2126.13 BOOL  ; NC433_6_U 7ST接料伺服偏差计数器复位输出/ 原点调整命令输出
2126.14 BOOL  ; NC433_6_U 7ST接料伺服激活Override
2126.15 BOOL  ; NC433_6_U 7ST接料伺服停止
2127.00 BOOL  ; NC433_6_U 7ST接料伺服预留
2127.01 BOOL  ; NC433_6_U 7ST接料伺服预留
2127.02 BOOL  ; NC433_6_U 7ST接料伺服预留
2127.03 BOOL  ; NC433_6_U 7ST接料伺服预留
2127.04 BOOL  ; NC433_6_U 7ST接料伺服预留
2127.05 BOOL  ; NC433_6_U 7ST接料伺服预留
2127.06 BOOL  ; NC433_6_U 7ST接料伺服预留
2127.07 BOOL  ; NC433_6_U 7ST接料伺服预留
2127.08 BOOL  ; NC433_6_U 7ST接料伺服强制中断
2127.09 BOOL  ; NC433_6_U 7ST接料伺服预留
2127.10 BOOL  ; NC433_6_U 7ST接料伺服预留
2127.11 BOOL  ; NC433_6_U 7ST接料伺服预留
2127.12 BOOL  ; NC433_6_U 7ST接料伺服数据写入
2127.13 BOOL  ; NC433_6_U 7ST接料伺服数据读出
2127.14 BOOL  ; NC433_6_U 7ST接料伺服数据保存
2127.15 BOOL  ; NC433_6_U 7ST接料伺服预留
2128.00 BOOL  ; NC433_6_X1#预留
2128.01 BOOL  ; NC433_6_X1#预留
2128.02 BOOL  ; NC433_6_X1#预留
2128.03 BOOL  ; NC433_6_X1#预留
2128.04 BOOL  ; NC433_6_X1#等待存储器操作
2128.05 BOOL  ; NC433_6_X1#定位完成标志位
2128.06 BOOL  ; NC433_6_X1#无原点标志位
2128.07 BOOL  ; NC433_6_X1#原点停止标志位
2128.08 BOOL  ; NC433_6_X1#0 区监测标志位
2128.09 BOOL  ; NC433_6_X1#1 区监测标志位
2128.10 BOOL  ; NC433_6_X1#2 区监测标志位
2128.11 BOOL  ; NC433_6_X1#示教完成
2128.12 BOOL  ; NC433_6_X1#错误标志
2128.13 BOOL  ; NC433_6_X1#忙标志
2128.14 BOOL  ; NC433_6_X1#数据传送标志位
2128.15 BOOL  ; NC433_6_X1#减速停止执行标志位
2129.00 BOOL  ; NC433_6_X1#预留
2129.01 BOOL  ; NC433_6_X1#预留
2129.02 BOOL  ; NC433_6_X1#预留
2129.03 BOOL  ; NC433_6_X1#预留
2129.04 BOOL  ; NC433_6_X1#预留
2129.05 BOOL  ; NC433_6_X1#预留
2129.06 BOOL  ; NC433_6_X1#预留
2129.07 BOOL  ; NC433_6_X1#预留
2129.08 BOOL  ; NC433_6_X1#CW极限输入信号
2129.09 BOOL  ; NC433_6_X1#CCW极限输入信号
2129.10 BOOL  ; NC433_6_X1#原点接近输入信号
2129.11 BOOL  ; NC433_6_X1#原点输入信号
2129.12 BOOL  ; NC433_6_X1#中断输入信号
2129.13 BOOL  ; NC433_6_X1#紧急输入信号
2129.14 BOOL  ; NC433_6_X1#定位完成输入信号
2129.15 BOOL  ; NC433_6_X1#偏差计数器复位输出/ 原点调整命令输出
2130.00 BOOL  ; NC433_6_X1#错误代码
2130.01 BOOL  ; NC433_6_X1#错误代码
2130.02 BOOL  ; NC433_6_X1#错误代码
2130.03 BOOL  ; NC433_6_X1#错误代码
2130.04 BOOL  ; NC433_6_X1#错误代码
2130.05 BOOL  ; NC433_6_X1#错误代码
2130.06 BOOL  ; NC433_6_X1#错误代码
2130.07 BOOL  ; NC433_6_X1#错误代码
2130.08 BOOL  ; NC433_6_X1#错误代码
2130.09 BOOL  ; NC433_6_X1#错误代码
2130.10 BOOL  ; NC433_6_X1#错误代码
2130.11 BOOL  ; NC433_6_X1#错误代码
2130.12 BOOL  ; NC433_6_X1#错误代码
2130.13 BOOL  ; NC433_6_X1#错误代码
2130.14 BOOL  ; NC433_6_X1#错误代码
2130.15 BOOL  ; NC433_6_X1#错误代码
2131.00 BOOL  ; NC433_6_Y 2#预留
2131.01 BOOL  ; NC433_6_Y 2#预留
2131.02 BOOL  ; NC433_6_Y 2#预留
2131.03 BOOL  ; NC433_6_Y 2#预留
2131.04 BOOL  ; NC433_6_Y 2#等待存储器操作
2131.05 BOOL  ; NC433_6_Y 2#定位完成标志位
2131.06 BOOL  ; NC433_6_Y 2#无原点标志位
2131.07 BOOL  ; NC433_6_Y 2#原点停止标志位
2131.08 BOOL  ; NC433_6_Y 2#0 区监测标志位
2131.09 BOOL  ; NC433_6_Y 2#1 区监测标志位
2131.10 BOOL  ; NC433_6_Y 2#2 区监测标志位
2131.11 BOOL  ; NC433_6_Y 2#示教完成
2131.12 BOOL  ; NC433_6_Y 2#错误标志
2131.13 BOOL  ; NC433_6_Y 2#忙标志
2131.14 BOOL  ; NC433_6_Y 2#数据传送标志位
2131.15 BOOL  ; NC433_6_Y 2#减速停止执行标志位
2132.00 BOOL  ; NC433_6_Y 2#预留
2132.01 BOOL  ; NC433_6_Y 2#预留
2132.02 BOOL  ; NC433_6_Y 2#预留
2132.03 BOOL  ; NC433_6_Y 2#预留
2132.04 BOOL  ; NC433_6_Y 2#预留
2132.05 BOOL  ; NC433_6_Y 2#预留
2132.06 BOOL  ; NC433_6_Y 2#预留
2132.07 BOOL  ; NC433_6_Y 2#预留
2132.08 BOOL  ; NC433_6_Y 2#CW极限输入信号
2132.09 BOOL  ; NC433_6_Y 2#CCW极限输入信号
2132.10 BOOL  ; NC433_6_Y 2#原点接近输入信号
2132.11 BOOL  ; NC433_6_Y 2#原点输入信号
2132.12 BOOL  ; NC433_6_Y 2#中断输入信号
2132.13 BOOL  ; NC433_6_Y 2#紧急输入信号
2132.14 BOOL  ; NC433_6_Y 2#定位完成输入信号
2132.15 BOOL  ; NC433_6_Y 2#偏差计数器复位输出/ 原点调整命令输出
2133.00 BOOL  ; NC433_6_Y 2#错误代码
2133.01 BOOL  ; NC433_6_Y 2#错误代码
2133.02 BOOL  ; NC433_6_Y 2#错误代码
2133.03 BOOL  ; NC433_6_Y 2#错误代码
2133.04 BOOL  ; NC433_6_Y 2#错误代码
2133.05 BOOL  ; NC433_6_Y 2#错误代码
2133.06 BOOL  ; NC433_6_Y 2#错误代码
2133.07 BOOL  ; NC433_6_Y 2#错误代码
2133.08 BOOL  ; NC433_6_Y 2#错误代码
2133.09 BOOL  ; NC433_6_Y 2#错误代码
2133.10 BOOL  ; NC433_6_Y 2#错误代码
2133.11 BOOL  ; NC433_6_Y 2#错误代码
2133.12 BOOL  ; NC433_6_Y 2#错误代码
2133.13 BOOL  ; NC433_6_Y 2#错误代码
2133.14 BOOL  ; NC433_6_Y 2#错误代码
2133.15 BOOL  ; NC433_6_Y 2#错误代码
2134.00 BOOL  ; NC433_6_Z 3#预留
2134.01 BOOL  ; NC433_6_Z 3#预留
2134.02 BOOL  ; NC433_6_Z 3#预留
2134.03 BOOL  ; NC433_6_Z 3#预留
2134.04 BOOL  ; NC433_6_Z 3#等待存储器操作
2134.05 BOOL  ; NC433_6_Z 3#定位完成标志位
2134.06 BOOL  ; NC433_6_Z 3#无原点标志位
2134.07 BOOL  ; NC433_6_Z 3#原点停止标志位
2134.08 BOOL  ; NC433_6_Z 3#0 区监测标志位
2134.09 BOOL  ; NC433_6_Z 3#1 区监测标志位
2134.10 BOOL  ; NC433_6_Z 3#2 区监测标志位
2134.11 BOOL  ; NC433_6_Z 3#示教完成
2134.12 BOOL  ; NC433_6_Z 3#错误标志
2134.13 BOOL  ; NC433_6_Z 3#忙标志
2134.14 BOOL  ; NC433_6_Z 3#数据传送标志位
2134.15 BOOL  ; NC433_6_Z 3#减速停止执行标志位
2135.00 BOOL  ; NC433_6_Z 3#预留
2135.01 BOOL  ; NC433_6_Z 3#预留
2135.02 BOOL  ; NC433_6_Z 3#预留
2135.03 BOOL  ; NC433_6_Z 3#预留
2135.04 BOOL  ; NC433_6_Z 3#预留
2135.05 BOOL  ; NC433_6_Z 3#预留
2135.06 BOOL  ; NC433_6_Z 3#预留
2135.07 BOOL  ; NC433_6_Z 3#预留
2135.08 BOOL  ; NC433_6_Z 3#CW极限输入信号
2135.09 BOOL  ; NC433_6_Z 3#CCW极限输入信号
2135.10 BOOL  ; NC433_6_Z 3#原点接近输入信号
2135.11 BOOL  ; NC433_6_Z 3#原点输入信号
2135.12 BOOL  ; NC433_6_Z 3#中断输入信号
2135.13 BOOL  ; NC433_6_Z 3#紧急输入信号
2135.14 BOOL  ; NC433_6_Z 3#定位完成输入信号
2135.15 BOOL  ; NC433_6_Z 3#偏差计数器复位输出/ 原点调整命令输出
2136.00 BOOL  ; NC433_6_Z 3#错误代码
2136.01 BOOL  ; NC433_6_Z 3#错误代码
2136.02 BOOL  ; NC433_6_Z 3#错误代码
2136.03 BOOL  ; NC433_6_Z 3#错误代码
2136.04 BOOL  ; NC433_6_Z 3#错误代码
2136.05 BOOL  ; NC433_6_Z 3#错误代码
2136.06 BOOL  ; NC433_6_Z 3#错误代码
2136.07 BOOL  ; NC433_6_Z 3#错误代码
2136.08 BOOL  ; NC433_6_Z 3#错误代码
2136.09 BOOL  ; NC433_6_Z 3#错误代码
2136.10 BOOL  ; NC433_6_Z 3#错误代码
2136.11 BOOL  ; NC433_6_Z 3#错误代码
2136.12 BOOL  ; NC433_6_Z 3#错误代码
2136.13 BOOL  ; NC433_6_Z 3#错误代码
2136.14 BOOL  ; NC433_6_Z 3#错误代码
2136.15 BOOL  ; NC433_6_Z 3#错误代码
2137.00 BOOL  ; NC433_6_U 7ST接料伺服预留
2137.01 BOOL  ; NC433_6_U 7ST接料伺服预留
2137.02 BOOL  ; NC433_6_U 7ST接料伺服预留
2137.03 BOOL  ; NC433_6_U 7ST接料伺服预留
2137.04 BOOL  ; NC433_6_U 7ST接料伺服等待存储器操作
2137.05 BOOL  ; NC433_6_U 7ST接料伺服定位完成标志位
2137.06 BOOL  ; NC433_6_U 7ST接料伺服无原点标志位
2137.07 BOOL  ; NC433_6_U 7ST接料伺服原点停止标志位
2137.08 BOOL  ; NC433_6_U 7ST接料伺服0 区监测标志位
2137.09 BOOL  ; NC433_6_U 7ST接料伺服1 区监测标志位
2137.10 BOOL  ; NC433_6_U 7ST接料伺服2 区监测标志位
2137.11 BOOL  ; NC433_6_U 7ST接料伺服示教完成
2137.12 BOOL  ; NC433_6_U 7ST接料伺服错误标志
2137.13 BOOL  ; NC433_6_U 7ST接料伺服忙标志
2137.14 BOOL  ; NC433_6_U 7ST接料伺服数据传送标志位
2137.15 BOOL  ; NC433_6_U 7ST接料伺服减速停止执行标志位
2138.00 BOOL  ; NC433_6_U 7ST接料伺服预留
2138.01 BOOL  ; NC433_6_U 7ST接料伺服预留
2138.02 BOOL  ; NC433_6_U 7ST接料伺服预留
2138.03 BOOL  ; NC433_6_U 7ST接料伺服预留
2138.04 BOOL  ; NC433_6_U 7ST接料伺服预留
2138.05 BOOL  ; NC433_6_U 7ST接料伺服预留
2138.06 BOOL  ; NC433_6_U 7ST接料伺服预留
2138.07 BOOL  ; NC433_6_U 7ST接料伺服预留
2138.08 BOOL  ; NC433_6_U 7ST接料伺服CW极限输入信号
2138.09 BOOL  ; NC433_6_U 7ST接料伺服CCW极限输入信号
2138.10 BOOL  ; NC433_6_U 7ST接料伺服原点接近输入信号
2138.11 BOOL  ; NC433_6_U 7ST接料伺服原点输入信号
2138.12 BOOL  ; NC433_6_U 7ST接料伺服中断输入信号
2138.13 BOOL  ; NC433_6_U 7ST接料伺服紧急输入信号
2138.14 BOOL  ; NC433_6_U 7ST接料伺服定位完成输入信号
2138.15 BOOL  ; NC433_6_U 7ST接料伺服偏差计数器复位输出/ 原点调整命令输出
2139.00 BOOL  ; NC433_6_U 7ST接料伺服错误代码
2139.01 BOOL  ; NC433_6_U 7ST接料伺服错误代码
2139.02 BOOL  ; NC433_6_U 7ST接料伺服错误代码
2139.03 BOOL  ; NC433_6_U 7ST接料伺服错误代码
2139.04 BOOL  ; NC433_6_U 7ST接料伺服错误代码
2139.05 BOOL  ; NC433_6_U 7ST接料伺服错误代码
2139.06 BOOL  ; NC433_6_U 7ST接料伺服错误代码
2139.07 BOOL  ; NC433_6_U 7ST接料伺服错误代码
2139.08 BOOL  ; NC433_6_U 7ST接料伺服错误代码
2139.09 BOOL  ; NC433_6_U 7ST接料伺服错误代码
2139.10 BOOL  ; NC433_6_U 7ST接料伺服错误代码
2139.11 BOOL  ; NC433_6_U 7ST接料伺服错误代码
2139.12 BOOL  ; NC433_6_U 7ST接料伺服错误代码
2139.13 BOOL  ; NC433_6_U 7ST接料伺服错误代码
2139.14 BOOL  ; NC433_6_U 7ST接料伺服错误代码
2139.15 BOOL  ; NC433_6_U 7ST接料伺服错误代码
2170 CHANNEL  ; DA08V_1 通道使能
2171 CHANNEL  ; DA08V_1 通道1 A1比例阀 转换值
2172 CHANNEL  ; DA08V_1 通道2 A2比例阀 转换值
2173 CHANNEL  ; DA08V_1 通道3 A3比例阀 转换值
2174 CHANNEL  ; DA08V_1 通道4 A4比例阀 转换值
2175 CHANNEL  ; DA08V_1 通道5 B1比例阀 转换值
2176 CHANNEL  ; DA08V_1 通道6 B2比例阀 转换值
2177 CHANNEL  ; DA08V_1 通道7 B3比例阀 转换值
2178 CHANNEL  ; DA08V_1 通道8 B4比例阀 转换值
2180 CHANNEL  ; DA08V_2 通道使能
2181 CHANNEL  ; DA08V_2 通道1DA 转换值
2182 CHANNEL  ; DA08V_2 通道2DA 转换值
2183 CHANNEL  ; DA08V_2 通道3DA 转换值
2184 CHANNEL  ; DA08V_2 通道4DA 转换值
2185 CHANNEL  ; DA08V_2 通道5DA 转换值
2186 CHANNEL  ; DA08V_2 通道6DA 转换值
2187 CHANNEL  ; DA08V_2 通道7DA 转换值
2188 CHANNEL  ; DA08V_2 通道8DA 转换值
2190 CHANNEL  ; DA08V_3 通道使能
2191 CHANNEL  ; DA08V_3 通道1DA 转换值
2192 CHANNEL  ; DA08V_3 通道2DA 转换值
2193 CHANNEL  ; DA08V_3 通道3DA 转换值
2194 CHANNEL  ; DA08V_3 通道4DA 转换值
2195 CHANNEL  ; DA08V_3 通道5DA 转换值
2196 CHANNEL  ; DA08V_3 通道6DA 转换值
2197 CHANNEL  ; DA08V_3 通道7DA 转换值
2198 CHANNEL  ; DA08V_3 通道8DA 转换值
21.00 BOOL  ; 热压C下层上板左加热启动
21.01 BOOL  ; 热压C下层上板中加热启动
21.02 BOOL  ; 热压C下层上板右加热启动
21.03 BOOL  ; 热压C下层下板左加热启动
21.04 BOOL  ; 热压C下层下板中加热启动
21.05 BOOL  ; 热压C下层下板右加热启动
2200 CHANNEL  ; DA08V_4 通道使能
2201 CHANNEL  ; DA08V_4 通道1DA 转换值
2202 CHANNEL  ; DA08V_4 通道2DA 转换值
2203 CHANNEL  ; DA08V_4 通道3DA 转换值
2204 CHANNEL  ; DA08V_4 通道4DA 转换值
2205 CHANNEL  ; DA08V_4 通道5DA 转换值
2206 CHANNEL  ; DA08V_4 通道6DA 转换值
2207 CHANNEL  ; DA08V_4 通道7DA 转换值
2208 CHANNEL  ; DA08V_4 通道8DA 转换值
221.00 BOOL  ; 进出料横移伺服A进料位手动(M)
221.01 BOOL  ; 进出料横移伺服热压A放料位手动(M)
221.02 BOOL  ; 进出料横移伺服热压A取料位手动(M)
221.03 BOOL  ; 进出料横移伺服热压B放料位手动(M)
221.04 BOOL  ; 横移伺服热压B取料位手动(M)
221.05 BOOL  ; 横移伺服热压C放料位手动(M)
221.06 BOOL  ; 横移伺服热压C取料位手动(M)
221.07 BOOL  ; 进出料横移伺服出料位手动(M)
222.00 BOOL  ; 进出料横移伺服A进料位(A)
222.01 BOOL  ; 进出料横移伺服热压A放料位(A)
222.02 BOOL  ; 进出料横移伺服热压A取料位(A)
222.03 BOOL  ; 进出料横移伺服热压B放料位(A)
222.04 BOOL  ; 横移伺服热压B取料位(A)
222.05 BOOL  ; 横移伺服热压C放料位(A)
222.06 BOOL  ; 横移伺服热压C取料位(A)
222.07 BOOL  ; 进出料横移伺服出料位(A)
223.00 BOOL  ; 进出料伸缩伺服等待位手动(M)
223.01 BOOL  ; 进出料伸缩伺服平台取料位手动(M)
223.02 BOOL  ; 进出料伸缩伺服A热压取放位手动(M)
224.00 BOOL  ; 进出料伸缩伺服等待位(A)
224.01 BOOL  ; 进出料伸缩伺服平台取料位(A)
224.02 BOOL  ; 进出料伸缩伺服A热压取放位(A)
2.00 BOOL  ; 进料定位下层有料感应
2.01 BOOL  ; 出料定位上层前后松开位
2.02 BOOL  ; 出料定位上层前后夹紧位
2.03 BOOL  ; 出料定位下层前后松开位
2.04 BOOL  ; 出料定位下层前后夹紧位
2.05 BOOL  ; 出料定位上层左右松开位
2.06 BOOL  ; 出料定位上层左右夹紧位
2.07 BOOL  ; 出料定位下层左右松开位
2.08 BOOL  ; 出料定位下层左右夹紧位
2.09 BOOL  ; 出料定位平台上层接料位
2.10 BOOL  ; 出料定位平台上层出料位
2.11 BOOL  ; 出料定位平台下层接料位
2.12 BOOL  ; 出料定位平台下层出料位
2.13 BOOL  ; 出料定位上层有料感应
2.14 BOOL  ; 出料定位下层有料感应
2.15 BOOL  ; 备用5
321.00 BOOL  ; 进出料横移伺服A进料位
321.01 BOOL  ; 进出料横移伺服热压A放料位
321.02 BOOL  ; 进出料横移伺服热压A取料位
321.03 BOOL  ; 进出料横移伺服热压B放料位
321.04 BOOL  ; 横移伺服热压B取料位
321.05 BOOL  ; 横移伺服热压C放料位
321.06 BOOL  ; 横移伺服热压C取料位
321.07 BOOL  ; 进出料横移伺服出料位
323.00 BOOL  ; 进出料伸缩伺服等待位
323.01 BOOL  ; 进出料伸缩伺服平台取料位
323.02 BOOL  ; 进出料伸缩伺服A热压取放位
3.00 BOOL  ; 进料夹爪张开位
3.01 BOOL  ; 进料夹爪夹紧位
3.02 BOOL  ; 进料爪上层左压紧上升位
3.03 BOOL  ; 进料爪上层右压紧上升位
3.04 BOOL  ; 进料爪下层左压紧上升位
3.05 BOOL  ; 进料爪下层右压紧上升位
3.06 BOOL  ; 进料爪上层中间压紧上升位
3.07 BOOL  ; 进料爪下层中间压紧上升位
3.08 BOOL  ; 进料夹爪上升位
3.09 BOOL  ; 进料夹爪下降位
3.10 BOOL  ; 进料爪上层有料感应
3.11 BOOL  ; 进料爪下层有料感应
3.12 BOOL  ; 出料夹爪张开位
3.13 BOOL  ; 出料夹爪夹紧位
3.14 BOOL  ; 出料爪上层左压紧上升位
3.15 BOOL  ; 出料爪上层右压紧上升位
42.04 BOOL  ; $?St$Bk?_#[5] / 上料定位A0度翻转 / $?St$Bk?_#[5]
42.05 BOOL  ; 上料定位A90度翻转
42.06 BOOL  ; 上料定位A1前后左右松开
42.07 BOOL  ; 上料定位A1前后左右夹紧
42.08 BOOL  ; 上料定位A2前后左右松开
42.09 BOOL  ; 上料定位A2前后左右夹紧
42.10 BOOL  ; 上料定位A3前后左右松开
42.11 BOOL  ; 上料定位A3前后左右夹紧
42.12 BOOL  ; 上料定位A4前后左右松开
42.13 BOOL  ; 上料定位A4前后左右夹紧
47.02 BOOL  ; 热压A上预压平移气缸缩回
47.03 BOOL  ; 热压A上预压平移气缸预压
47.06 BOOL  ; 热压A垫高气缸移出
47.07 BOOL  ; 热压A垫高气缸热压
47.08 BOOL  ; 热压A1HIP测试上升
47.09 BOOL  ; 热压A1HIP测试下降
48.00 BOOL  ; 热压A1顶升气缸缩回
48.01 BOOL  ; 热压A1顶升气缸伸出
48.02 BOOL  ; 热压A2顶升气缸左右缩回
48.03 BOOL  ; 热压A2顶升气缸左右伸出
48.04 BOOL  ; 热压A3顶升气缸左右缩回
48.05 BOOL  ; 热压A3顶升气缸左右伸出
48.06 BOOL  ; 热压A4顶升气缸左右缩回
48.07 BOOL  ; 热压A4顶升气缸左右伸出
48.14 BOOL  ; 热压A上吹气
48.15 BOOL  ; 热压A下板A吹气
49.00 BOOL  ; 热压A下板B吹气
49.01 BOOL  ; 热压B上预压平移气缸缩回
49.02 BOOL  ; 热压B上预压平移气缸预压
49.03 BOOL  ; 热压B下预压平移气缸缩回
49.04 BOOL  ; 热压B下预压平移气缸预压
49.05 BOOL  ; 热压B垫高气缸移出
49.06 BOOL  ; 热压B垫高气缸热压
49.07 BOOL  ; 热压B1HIP测试上升
49.08 BOOL  ; 热压B1HIP测试下降
49.15 BOOL  ; 热压B1顶升气缸缩回
4.00 BOOL  ; 出料爪下层左压紧上升位
4.01 BOOL  ; 出料爪下层右压紧上升位
4.02 BOOL  ; 出料夹爪上升位
4.03 BOOL  ; 出料夹爪下降位
4.04 BOOL  ; 出料爪上层有料感应
4.05 BOOL  ; 出料爪下层有料感应
4.06 BOOL  ; 备用6
4.07 BOOL  ; 备用7
4.08 BOOL  ; 热压A增压缸上升位
4.09 BOOL  ; 热压A增压缸下降位
4.10 BOOL  ; 热压A上层顶升气缸上升位
4.11 BOOL  ; 热压A上层顶升气缸下降位
4.12 BOOL  ; 热压A下层顶升气缸上升位
4.13 BOOL  ; 热压A下层顶升气缸下降位
4.14 BOOL  ; 热压A垫高气缸移出位
4.15 BOOL  ; 热压A垫高气缸热压位
50.00 BOOL  ; 热压B1顶升气缸伸出
50.01 BOOL  ; 热压B2顶升气缸左缩回
50.02 BOOL  ; 热压B2顶升气缸左伸出
50.03 BOOL  ; 热压B3顶升气缸左缩回
50.04 BOOL  ; 热压B3顶升气缸左伸出
50.05 BOOL  ; 热压B4顶升气缸左缩回
50.06 BOOL  ; 热压B4顶升气缸左伸出
50.13 BOOL  ; 热压B上吹气
50.14 BOOL  ; 热压B下板A吹气
50.15 BOOL  ; 热压B下板B吹气
5.00 BOOL  ; 热压A上层Hip测试气缸上升位
5.01 BOOL  ; 热压A上层Hip测试气缸下降位
5.02 BOOL  ; 热压A下层Hip测试气缸上升位
5.03 BOOL  ; 热压A下层Hip测试气缸下降位
5.04 BOOL  ; 热压A上层有料感应
5.05 BOOL  ; 热压A下层有料感应
5.06 BOOL  ; 热压A上层极耳检查输入
5.07 BOOL  ; 热压A下层极耳检查输入
5.08 BOOL  ; 备用8
5.09 BOOL  ; 热压B增压缸上升位
5.10 BOOL  ; 热压B增压缸下降位
5.11 BOOL  ; 热压B上层顶升气缸上升位
5.12 BOOL  ; 热压B上层顶升气缸下降位
5.13 BOOL  ; 热压B下层顶升气缸上升位
5.14 BOOL  ; 热压B下层顶升气缸下降位
5.15 BOOL  ; 热压B垫高气缸移出位
6.00 BOOL  ; 热压B垫高气缸热压位
6.01 BOOL  ; 热压B上层Hip测试气缸上升位
6.02 BOOL  ; 热压B上层Hip测试气缸下降位
6.03 BOOL  ; 热压B下层Hip测试气缸上升位
6.04 BOOL  ; 热压B下层Hip测试气缸下降位
6.05 BOOL  ; 热压B上层有料感应
6.06 BOOL  ; 热压B下层有料感应
6.07 BOOL  ; 热压B上层极耳检查输入
6.08 BOOL  ; 热压B下层极耳检查输入
6.09 BOOL  ; 备用9
6.10 BOOL  ; 热压C增压缸上升位
6.11 BOOL  ; 热压C增压缸下降位
6.12 BOOL  ; 热压C上层顶升气缸上升位
6.13 BOOL  ; 热压C上层顶升气缸下降位
6.14 BOOL  ; 热压C下层顶升气缸上升位
6.15 BOOL  ; 热压C下层顶升气缸下降位
711 CHANNEL  ; 机器人不在取料区域延时
713 CHANNEL  ; $?St$Bk?_#[6] / 机器人不在放料A区域 / $?St$Bk?_#[6]
7.00 BOOL  ; 热压C垫高气缸移出位
7.01 BOOL  ; 热压C垫高气缸热压位
7.02 BOOL  ; 热压C上层Hip测试气缸上升位
7.03 BOOL  ; 热压C上层Hip测试气缸下降位
7.04 BOOL  ; 热压C下层Hip测试气缸上升位
7.05 BOOL  ; 热压C下层Hip测试气缸下降位
7.06 BOOL  ; 热压C上层有料感应
7.07 BOOL  ; 热压C下层有料感应
7.08 BOOL  ; 热压C上层极耳检查输入
7.09 BOOL  ; 热压C下层极耳检查输入
7.10 BOOL  ; 备用10
7.11 BOOL  ; 进出料转移伺服准备好
7.12 BOOL  ; 进出料转移伺服报警
7.13 BOOL  ; 伸缩伺服准备好
7.14 BOOL  ; 伸缩伺服报警
7.15 BOOL  ; 备用11
8 CHANNEL  ; 副PLC 0CH输入映射
8.00 BOOL  ; 加热A跳闸
8.01 BOOL  ; 加热B跳闸
8.02 BOOL  ; 加热C跳闸
8.03 BOOL  ; 副PLC 0.03
8.04 BOOL  ; 副PLC 0.04
8.05 BOOL  ; 副PLC 0.05
8.06 BOOL  ; 副PLC 0.06
8.07 BOOL  ; 副PLC 0.07
8.08 BOOL  ; 副PLC 0.08
8.09 BOOL  ; 副PLC 0.09
8.10 BOOL  ; 副PLC 0.10
8.11 BOOL  ; 副PLC 0.11
9 CHANNEL  ; 副PLC输入点1CH 映射地址
9.00 BOOL  ; 副PLC 1.00
9.01 BOOL  ; 副PLC 1.01
9.02 BOOL  ; 副PLC 1.02
9.03 BOOL  ; 副PLC 1.03
9.04 BOOL  ; 副PLC 1.04
9.05 BOOL  ; 副PLC 1.05
9.06 BOOL  ; 副PLC 1.06
9.07 BOOL  ; 副PLC 1.07
9.08 BOOL  ; 副PLC 1.08
9.09 BOOL  ; 副PLC 1.09
9.10 BOOL  ; 副PLC 1.10
9.11 BOOL  ; 副PLC 1.11
A202.00 BOOL  ; 内部逻辑端口1网络通信可执行标志
A202.01 BOOL  ; 内部逻辑端口2网络通信可执行标志
A202.02 BOOL  ; 内部逻辑端口3网络通信可执行标志
A202.03 BOOL  ; 内部逻辑端口4网络通信可执行标志
A202.04 BOOL  ; 内部逻辑端口5网络通信可执行标志
A202.05 BOOL  ; 内部逻辑端口6网络通信可执行标志
A202.06 BOOL  ; 内部逻辑端口7网络通信可执行标志
A202.07 BOOL  ; 内部逻辑端口7网络通信可执行标志
D0.00 BOOL  ; 机器人安全位置
D0.01 BOOL  ; 移载安全位置
D1000.00 BOOL  ; 自动模式
D1000.01 BOOL  ; 手动模式
D1000.02 BOOL  ; 自动运行中
D1000.04 BOOL  ; 初始化中
D1000.05 BOOL  ; 清料停止中
D1000.06 BOOL  ; 自动停止中
D1000.07 BOOL  ; 蜂鸣器停止
D1001.00 BOOL  ; 自动停止完成
D1001.02 BOOL  ; 整机初始化完成
D1001.03 BOOL  ; 整机清料完成
D1001.04 BOOL  ; 整机物料感应为空
D1001.05 BOOL  ; 外部（工厂报警系统）→允许运行
D1001.09 BOOL  ; 气压异常（正常=1）
D1001.10 BOOL  ; 急停（正常=1）
D1001.11 BOOL  ; 安全装置（正常=1）
D1001.12 BOOL  ; 跳闸（正常=1）
D1001.13 BOOL  ; 整机错误（气压+急停+门+跳闸）
D1001.14 BOOL  ; 整机警报
D1001.15 BOOL  ; 整机+工站错误
D1002.00 BOOL  ; 清料停止[T]
D1002.09 BOOL  ; 复位（T）
D1002.10 BOOL  ; 整机启动[T]
D1002.11 BOOL  ; 整机自动停止[T]
D1002.12 BOOL  ; 整机初始化[T]
D1002.14 BOOL  ; 蜂鸣器消音（T）
D1002.15 BOOL  ; 任务停止
D1003.02 BOOL  ; 整机记忆清除（T）
D1003.15 BOOL  ; 模组B加热正常
D1005 CHANNEL  ; 屏幕状态
D10050 CHANNEL  ; ST5520_A 测试电压输入设定值(F)
D10060 CHANNEL  ; 字符串表现形式(0-小数点形式,1-指数形式)
D10061 CHANNEL  ; 全位数
D10062 CHANNEL  ; 小数位数
D1006.00 BOOL  ; 主屏使用
D1006.01 BOOL  ; 副屏使用
D1006.02 BOOL  ; 小屏使用
D1006.03 BOOL  ; 没有移动屏使用信号，小屏不能使用
D10070 CHANNEL  ; ST5520_A 测试电压输入设定值(ASCII)
D10080 CHANNEL  ; ST5520_A 测试时间输入设定值(F)
D10091 CHANNEL  ; 全位数
D10092 CHANNEL  ; 小数位数
D10100 CHANNEL  ; ST5520_A 测试时间输入设定值(ASC)
D1010.00 BOOL  ; 1St上料机器人工站错误
D1010.01 BOOL  ; 1St上料机器人工站警告
D1010.02 BOOL  ; 1St上料机器人工站运行
D1010.03 BOOL  ; $?St$Bk?_#[8] / 1St上料机器人"$?St$Bk?_#[8]
D1010.05 BOOL  ; $?St$Bk?_#[10] / 1St上料机器人"$?St$Bk?_#[10]
D1010.07 BOOL  ; $?St$Bk?_#[12] / 1St上料机器人"$?St$Bk?_#[12]
D1010.09 BOOL  ; $?St$Bk?_#[14] / 1St上料机器人"$?St$Bk?_#[14]
D1010.11 BOOL  ; $?St$Bk?_#[16] / 1St上料机器人"$?St$Bk?_#[16]
D1010.13 BOOL  ; $?St$Bk?_#[18] / 1St上料机器人"$?St$Bk?_#[18]
D1010.15 BOOL  ; $?St$Bk?_#[20] / 1St上料机器人"$?St$Bk?_#[20]
D1011.04 BOOL  ; $?St$Bk?_#[22] / 1St上料机器人"$?St$Bk?_#[22]
D1011.06 BOOL  ; $?St$Bk?_#[24] / 1St上料机器人"$?St$Bk?_#[24]
D1011.08 BOOL  ; $?St$Bk?_#[26] / 1St上料机器人"$?St$Bk?_#[26]
D1011.10 BOOL  ; $?St$Bk?_#[28] / 1St上料机器人"$?St$Bk?_#[28]
D1011.12 BOOL  ; $?St$Bk?_#[30] / 1St上料机器人"$?St$Bk?_#[30]
D1011.14 BOOL  ; $?St$Bk?_#[32] / 1St上料机器人"$?St$Bk?_#[32]
D10120 CHANNEL  ; 字符串表现形式(0-小数点形式,1-指数形式)
D10121 CHANNEL  ; 全位数
D10122 CHANNEL  ; 小数位数
D1012.00 BOOL  ; 1St上料机器人工站就绪
D1012.01 BOOL  ; 1St上料机器人 初始化中
D1012.02 BOOL  ; 1St上料机器人 自动停止中
D1012.03 BOOL  ; 1St上料机器人 自动停止完成
D1012.04 BOOL  ; 1St上料机器人 联锁
D1012.05 BOOL  ; 1St上料机器人 单步中
D1012.06 BOOL  ; 1St上料机器人 单周期中
D1012.07 BOOL  ; 1St上料机器人 周期完成
D1012.08 BOOL  ; 1St上料机器人 任务开始
D1012.09 BOOL  ; 1St上料机器人 任务递进条件
D1012.10 BOOL  ; 1St上料机器人 任务递进
D1012.11 BOOL  ; 1St上料机器人 工作完成
D1012.12 BOOL  ; 1St上料机器人 初始化[T]
D1012.13 BOOL  ; 1St上料机器人 单步[T]
D1012.14 BOOL  ; 1St上料机器人 单周期[T]
D1012.15 BOOL  ; 1St上料机器人 任务停止[T]
D10130 CHANNEL  ; ST5520_A 响应延时时间输入设定值(ASC)
D1013.00 BOOL  ; 1St上料机器人 工站完成置位[T]
D1013.01 BOOL  ; 1St上料机器人 工站完成复位[T]
D1013.02 BOOL  ; 1St上料机器人 数据清除[T]
D1013.03 BOOL  ; 1St上料机器人 工站屏蔽[T]
D1013.04 BOOL  ; $?St$Bk?_#[34] / 1St上料机器人"$?St$Bk?_#[34]
D1013.06 BOOL  ; $?St$Bk?_#[36] / 1St上料机器人"$?St$Bk?_#[36]
D1013.08 BOOL  ; $?St$Bk?_#[38] / 1St上料机器人"$?St$Bk?_#[38]
D1013.10 BOOL  ; $?St$Bk?_#[40] / 1St上料机器人"$?St$Bk?_#[40]
D1013.12 BOOL  ; $?St$Bk?_#[42] / 1St上料机器人"$?St$Bk?_#[42]
D1013.14 BOOL  ; $?St$Bk?_#[44] / 1St上料机器人"$?St$Bk?_#[44]
D10140 CHANNEL  ; ST5520_A 绝缘电阻上限输入设定值(Float)
D1014.00 BOOL  ; 1St上料机器人上游就绪-0
D1014.01 BOOL  ; 1St上料机器人使能上游-0
D1014.02 BOOL  ; 1St上料机器人上游就绪-1
D1014.03 BOOL  ; 1St上料机器人使能上游-1
D1014.04 BOOL  ; 1St上料机器人上游就绪-2
D1014.05 BOOL  ; 1St上料机器人使能上游-2
D1014.06 BOOL  ; 1St上料机器人上游就绪-3
D1014.07 BOOL  ; 1St上料机器人使能上游-3
D1014.08 BOOL  ; 1St上料机器人下游就绪-0
D1014.09 BOOL  ; 1St上料机器人使能下游-0
D1014.10 BOOL  ; 1St上料机器人下游就绪-1
D1014.11 BOOL  ; 1St上料机器人使能下游-1
D1014.12 BOOL  ; 1St上料机器人下游就绪-2
D1014.13 BOOL  ; 1St上料机器人使能下游-2
D1014.14 BOOL  ; 1St上料机器人下游就绪-3
D1014.15 BOOL  ; 1St上料机器人使能下游-3
D1015 CHANNEL  ; 1ST自动步存放字
D10150 CHANNEL  ; 字符串表现形式(0-小数点形式,1-指数形式)
D10151 CHANNEL  ; 全位数
D1015.00 BOOL  ; 1St上料机器人开始步
D1015.01 BOOL  ; 1St上料机器人到抓料上位
D1015.02 BOOL  ; 1St上料机器人到抓料位
D1015.03 BOOL  ; 1St上料机器人全部夹紧
D1015.04 BOOL  ; 1St上料机器人全部压紧
D1015.05 BOOL  ; 1St上料机器人到扫码NG上位
D1015.06 BOOL  ; 1St上料机器人有料判断步
D1015.07 BOOL  ; 1St上料机器人去NG位安全条件
D1015.08 BOOL  ; 1St上料机器人到NG位
D1015.09 BOOL  ; 1St上料机器人放NG料
D1015.10 BOOL  ; 1St上料机器人有料判断步
D1015.11 BOOL  ; 1St上料机器人去放料位
D1015.12 BOOL  ; 1St上料机器人全部松压
D1015.13 BOOL  ; 1St上料机器人全部松开
D1015.14 BOOL  ; 1St上料机器人去抓料上位
D1015.15 BOOL  ; 1St上料机器人结束步
D10160 CHANNEL  ; ST5520_A 绝缘电阻上限输入设定值(ASCII)
D1016.00 BOOL  ; 1St上料机器人步16
D1016.01 BOOL  ; 1St上料机器人步17
D1016.02 BOOL  ; 1St上料机器人步18
D1016.03 BOOL  ; 1St上料机器人步19
D1016.04 BOOL  ; 1St上料机器人步20
D1016.05 BOOL  ; 1St上料机器人步21
D1016.06 BOOL  ; 1St上料机器人步22
D1016.07 BOOL  ; 1St上料机器人步23
D1016.08 BOOL  ; 1St上料机器人步24
D1016.09 BOOL  ; 1St上料机器人步25
D1016.10 BOOL  ; 1St上料机器人步26
D1016.11 BOOL  ; 1St上料机器人步27
D1016.12 BOOL  ; 1St上料机器人步28
D1016.13 BOOL  ; 1St上料机器人步29
D1016.14 BOOL  ; 1St上料机器人步30
D1016.15 BOOL  ; 1St上料机器人步31
D10170 CHANNEL  ; ST5520_A 绝缘电阻下限输入设定值(F)
D1017.00 BOOL  ; 1St上料机器人初始化步号
D1017.01 BOOL  ; 1St上料机器人
D1017.02 BOOL  ; 1St上料机器人
D1017.03 BOOL  ; 1St上料机器人
D1017.04 BOOL  ; 1St上料机器人
D1017.05 BOOL  ; 1St上料机器人
D1017.06 BOOL  ; 1St上料机器人
D1017.07 BOOL  ; 1St上料机器人
D1017.08 BOOL  ; 1St上料机器人
D1017.09 BOOL  ; 1St上料机器人
D1017.10 BOOL  ; 1St上料机器人
D1017.11 BOOL  ; 1St上料机器人
D1017.12 BOOL  ; 1St上料机器人
D1017.13 BOOL  ; 1St上料机器人
D1017.14 BOOL  ; 1St上料机器人
D1017.15 BOOL  ; 1St上料机器人
D10180 CHANNEL  ; 字符串表现形式(0-小数点形式,1-指数形式)
D10181 CHANNEL  ; 全位数
D10182 CHANNEL  ; 小数位数
D1018.00 BOOL  ; 1St上料机器人初始化_1
D1018.01 BOOL  ; 1St上料机器人初始化_2
D1018.02 BOOL  ; 1St上料机器人初始化_3
D1018.03 BOOL  ; 1St上料机器人初始化_4
D1018.04 BOOL  ; 1St上料机器人初始化_5
D1018.05 BOOL  ; 1St上料机器人初始化_6
D1018.06 BOOL  ; 1St上料机器人初始化_7
D1018.07 BOOL  ; 1St上料机器人初始化_8
D1018.08 BOOL  ; 1St上料机器人初始化_9
D1018.09 BOOL  ; 1St上料机器人初始化_10
D1018.10 BOOL  ; 1St上料机器人初始化_11
D1018.11 BOOL  ; 1St上料机器人初始化_12
D1018.12 BOOL  ; 1St上料机器人初始化_13
D1018.13 BOOL  ; 1St上料机器人初始化_14
D1018.14 BOOL  ; 1St上料机器人初始化_15
D1018.15 BOOL  ; 1St上料机器人初始化_16
D10190 CHANNEL  ; 字符串表现形式(0-小数点形式,1-指数形式)
D1019.00 BOOL  ; 1St上料机器人初始化_17
D1019.01 BOOL  ; 1St上料机器人初始化_18
D1019.02 BOOL  ; 1St上料机器人初始化_19
D1019.03 BOOL  ; 1St上料机器人初始化_20
D1019.04 BOOL  ; 1St上料机器人初始化_21
D1019.05 BOOL  ; 1St上料机器人初始化_22
D1019.06 BOOL  ; 1St上料机器人初始化_23
D1019.07 BOOL  ; 1St上料机器人初始化_24
D1019.08 BOOL  ; 1St上料机器人初始化_25
D1019.09 BOOL  ; 1St上料机器人初始化_26
D1019.10 BOOL  ; 1St上料机器人初始化_27
D1019.11 BOOL  ; 1St上料机器人初始化_28
D1019.12 BOOL  ; 1St上料机器人初始化_29
D1019.13 BOOL  ; 1St上料机器人初始化_30
D1019.14 BOOL  ; 1St上料机器人初始化_31
D1019.15 BOOL  ; 1St上料机器人初始化_32
D1020.00 BOOL  ; 1St_进料定位工站错误
D1020.01 BOOL  ; 1St_进料定位工站警告
D1020.02 BOOL  ; 1St_进料定位工站运行
D1020.03 BOOL  ; $?St$Bk?_#[46] / 1St_进料定位"$?St$Bk?_#[46]
D1020.05 BOOL  ; $?St$Bk?_#[48] / 1St_进料定位"$?St$Bk?_#[48]
D1020.07 BOOL  ; $?St$Bk?_#[50] / 1St_进料定位"$?St$Bk?_#[50]
D1020.09 BOOL  ; $?St$Bk?_#[52] / 1St_进料定位"$?St$Bk?_#[52]
D1020.11 BOOL  ; $?St$Bk?_#[54] / 1St_进料定位"$?St$Bk?_#[54]
D1020.13 BOOL  ; $?St$Bk?_#[56] / 1St_进料定位"$?St$Bk?_#[56]
D1020.15 BOOL  ; $?St$Bk?_#[58] / 1St_进料定位"$?St$Bk?_#[58]
D1021.04 BOOL  ; $?St$Bk?_#[60] / 1St_进料定位"$?St$Bk?_#[60]
D1021.06 BOOL  ; $?St$Bk?_#[62] / 1St_进料定位"$?St$Bk?_#[62]
D1021.08 BOOL  ; $?St$Bk?_#[64] / 1St_进料定位"$?St$Bk?_#[64]
D1021.10 BOOL  ; $?St$Bk?_#[66] / 1St_进料定位"$?St$Bk?_#[66]
D1021.12 BOOL  ; $?St$Bk?_#[68] / 1St_进料定位"$?St$Bk?_#[68]
D1021.14 BOOL  ; $?St$Bk?_#[70] / 1St_进料定位"$?St$Bk?_#[70]
D1022.00 BOOL  ; 1St_进料定位工站就绪
D1022.01 BOOL  ; 1St_进料定位 初始化中
D1022.02 BOOL  ; 1St_进料定位 自动停止中
D1022.03 BOOL  ; 1St_进料定位 自动停止完成
D1022.04 BOOL  ; 1St_进料定位 联锁
D1022.05 BOOL  ; 1St_进料定位 单步中
D1022.06 BOOL  ; 1St_进料定位 单周期中
D1022.07 BOOL  ; 1St_进料定位 周期完成
D1022.08 BOOL  ; 1St_进料定位 任务开始
D1022.09 BOOL  ; 1St_进料定位 任务递进条件
D1022.10 BOOL  ; 1St_进料定位 任务递进
D1022.11 BOOL  ; 1St_进料定位 工作完成
D1022.12 BOOL  ; 1St_进料定位 初始化[T]
D1022.13 BOOL  ; 1St_进料定位 单步[T]
D1022.14 BOOL  ; 1St_进料定位 单周期[T]
D1022.15 BOOL  ; 1St_进料定位 任务停止[T]
D1023.00 BOOL  ; 1St_进料定位 工站完成置位[T]
D1023.01 BOOL  ; 1St_进料定位 工站完成复位[T]
D1023.02 BOOL  ; 1St_进料定位 数据清除[T]
D1023.03 BOOL  ; 1St_进料定位 工站屏蔽[T]
D1023.04 BOOL  ; $?St$Bk?_#[72] / 1St_进料定位"$?St$Bk?_#[72]
D1023.06 BOOL  ; $?St$Bk?_#[74] / 1St_进料定位"$?St$Bk?_#[74]
D1023.08 BOOL  ; $?St$Bk?_#[76] / 1St_进料定位"$?St$Bk?_#[76]
D1023.10 BOOL  ; $?St$Bk?_#[78] / 1St_进料定位"$?St$Bk?_#[78]
D1023.12 BOOL  ; $?St$Bk?_#[80] / 1St_进料定位"$?St$Bk?_#[80]
D1023.14 BOOL  ; $?St$Bk?_#[82] / 1St_进料定位"$?St$Bk?_#[82]
D1024.00 BOOL  ; 1St_进料定位上游就绪-0
D1024.01 BOOL  ; 1St_进料定位使能上游-0
D1024.02 BOOL  ; 1St_进料定位上游就绪-1
D1024.03 BOOL  ; 1St_进料定位使能上游-1
D1024.04 BOOL  ; 1St_进料定位上游就绪-2
D1024.05 BOOL  ; 1St_进料定位使能上游-2
D1024.06 BOOL  ; 1St_进料定位上游就绪-3
D1024.07 BOOL  ; 1St_进料定位使能上游-3
D1024.08 BOOL  ; 1St_进料定位下游就绪-0
D1024.09 BOOL  ; 1St_进料定位使能下游-0
D1024.10 BOOL  ; 1St_进料定位下游就绪-1
D1024.11 BOOL  ; 1St_进料定位使能下游-1
D1024.12 BOOL  ; 1St_进料定位下游就绪-2
D1024.13 BOOL  ; 1St_进料定位使能下游-2
D1024.14 BOOL  ; 1St_进料定位下游就绪-3
D1024.15 BOOL  ; 1St_进料定位使能下游-3
D1025.00 BOOL  ; 1St_进料定位递进启动
D1025.01 BOOL  ; 1St_进料定位步01 前后左右夹紧
D1025.02 BOOL  ; 1St_进料定位步02 等待前进
D1025.03 BOOL  ; 1St_进料定位步03 平台前进
D1025.04 BOOL  ; 1St_进料定位步04 全部松开
D1025.05 BOOL  ; 1St_进料定位步05 等待取料
D1025.06 BOOL  ; 1St_进料定位步06平台缩回
D1025.07 BOOL  ; 1St_进料定位步07
D1025.08 BOOL  ; 1St_进料定位步08
D1025.09 BOOL  ; 1St_进料定位步09
D1025.10 BOOL  ; 1St_进料定位步10
D1025.11 BOOL  ; 1St_进料定位步11
D1025.12 BOOL  ; 1St_进料定位步12
D1025.13 BOOL  ; 1St_进料定位步13
D1025.14 BOOL  ; 1St_进料定位步14
D1025.15 BOOL  ; 1St_进料定位步15
D1026.00 BOOL  ; 1St_进料定位步16
D1026.01 BOOL  ; 1St_进料定位步17
D1026.02 BOOL  ; 1St_进料定位步18
D1026.03 BOOL  ; 1St_进料定位步19
D1026.04 BOOL  ; 1St_进料定位步20
D1026.05 BOOL  ; 1St_进料定位步21
D1026.06 BOOL  ; 1St_进料定位步22
D1026.07 BOOL  ; 1St_进料定位步23
D1026.08 BOOL  ; 1St_进料定位步24
D1026.09 BOOL  ; 1St_进料定位步25
D1026.10 BOOL  ; 1St_进料定位步26
D1026.11 BOOL  ; 1St_进料定位步27
D1026.12 BOOL  ; 1St_进料定位步28
D1026.13 BOOL  ; 1St_进料定位步29
D1026.14 BOOL  ; 1St_进料定位步30
D1026.15 BOOL  ; 1St_进料定位步31
D1027.00 BOOL  ; 1St_进料定位初始化步号
D1027.01 BOOL  ; 1St_进料定位
D1027.02 BOOL  ; 1St_进料定位
D1027.03 BOOL  ; 1St_进料定位
D1027.04 BOOL  ; 1St_进料定位
D1027.05 BOOL  ; 1St_进料定位
D1027.06 BOOL  ; 1St_进料定位
D1027.07 BOOL  ; 1St_进料定位
D1027.08 BOOL  ; 1St_进料定位
D1027.09 BOOL  ; 1St_进料定位
D1027.10 BOOL  ; 1St_进料定位
D1027.11 BOOL  ; 1St_进料定位
D1027.12 BOOL  ; 1St_进料定位
D1027.13 BOOL  ; 1St_进料定位
D1027.14 BOOL  ; 1St_进料定位
D1027.15 BOOL  ; 1St_进料定位
D1028.00 BOOL  ; 1St_进料定位初始化_全部松开
D1028.01 BOOL  ; 1St_进料定位初始化_2
D1028.02 BOOL  ; 1St_进料定位初始化_3
D1028.03 BOOL  ; 1St_进料定位初始化_4
D1028.04 BOOL  ; 1St_进料定位初始化_5
D1028.05 BOOL  ; 1St_进料定位初始化_6
D1028.06 BOOL  ; 1St_进料定位初始化_7
D1028.07 BOOL  ; 1St_进料定位初始化_8
D1028.08 BOOL  ; 1St_进料定位初始化_9
D1028.09 BOOL  ; 1St_进料定位初始化_10
D1028.10 BOOL  ; 1St_进料定位初始化_11
D1028.11 BOOL  ; 1St_进料定位初始化_12
D1028.12 BOOL  ; 1St_进料定位初始化_13
D1028.13 BOOL  ; 1St_进料定位初始化_14
D1028.14 BOOL  ; 1St_进料定位初始化_15
D1028.15 BOOL  ; 1St_进料定位初始化_16
D1029.00 BOOL  ; 1St_进料定位初始化_17
D1029.01 BOOL  ; 1St_进料定位初始化_18
D1029.02 BOOL  ; 1St_进料定位初始化_19
D1029.03 BOOL  ; 1St_进料定位初始化_20
D1029.04 BOOL  ; 1St_进料定位初始化_21
D1029.05 BOOL  ; 1St_进料定位初始化_22
D1029.06 BOOL  ; 1St_进料定位初始化_23
D1029.07 BOOL  ; 1St_进料定位初始化_24
D1029.08 BOOL  ; 1St_进料定位初始化_25
D1029.09 BOOL  ; 1St_进料定位初始化_26
D1029.10 BOOL  ; 1St_进料定位初始化_27
D1029.11 BOOL  ; 1St_进料定位初始化_28
D1029.12 BOOL  ; 1St_进料定位初始化_29
D1029.13 BOOL  ; 1St_进料定位初始化_30
D1029.14 BOOL  ; 1St_进料定位初始化_31
D1029.15 BOOL  ; 1St_进料定位初始化_32
D1030.00 BOOL  ; 2St_出料定位工站错误
D1030.01 BOOL  ; 2St_出料定位工站警告
D1030.02 BOOL  ; 2St_出料定位工站运行
D1030.03 BOOL  ; $?St$Bk?_#[84] / 2St_出料定位"$?St$Bk?_#[84]
D1030.05 BOOL  ; $?St$Bk?_#[86] / 2St_出料定位"$?St$Bk?_#[86]
D1030.07 BOOL  ; $?St$Bk?_#[88] / 2St_出料定位"$?St$Bk?_#[88]
D1030.09 BOOL  ; $?St$Bk?_#[90] / 2St_出料定位"$?St$Bk?_#[90]
D1030.11 BOOL  ; $?St$Bk?_#[92] / 2St_出料定位"$?St$Bk?_#[92]
D1030.13 BOOL  ; $?St$Bk?_#[94] / 2St_出料定位"$?St$Bk?_#[94]
D1030.15 BOOL  ; $?St$Bk?_#[96] / 2St_出料定位"$?St$Bk?_#[96]
D1031.04 BOOL  ; $?St$Bk?_#[98] / 2St_出料定位"$?St$Bk?_#[98]
D1031.06 BOOL  ; $?St$Bk?_#[100] / 2St_出料定位"$?St$Bk?_#[100]
D1031.08 BOOL  ; $?St$Bk?_#[102] / 2St_出料定位"$?St$Bk?_#[102]
D1031.10 BOOL  ; $?St$Bk?_#[104] / 2St_出料定位"$?St$Bk?_#[104]
D1031.12 BOOL  ; $?St$Bk?_#[106] / 2St_出料定位"$?St$Bk?_#[106]
D1031.14 BOOL  ; $?St$Bk?_#[108] / 2St_出料定位"$?St$Bk?_#[108]
D1032.00 BOOL  ; 2St_出料定位工站就绪
D1032.01 BOOL  ; 2St_出料定位 初始化中
D1032.02 BOOL  ; 2St_出料定位 自动停止中
D1032.03 BOOL  ; 2St_出料定位 自动停止完成
D1032.04 BOOL  ; 2St_出料定位 联锁
D1032.05 BOOL  ; 2St_出料定位 单步中
D1032.06 BOOL  ; 2St_出料定位 单周期中
D1032.07 BOOL  ; 2St_出料定位 周期完成
D1032.08 BOOL  ; 2St_出料定位 任务开始
D1032.09 BOOL  ; 2St_出料定位 任务递进条件
D1032.10 BOOL  ; 2St_出料定位 任务递进
D1032.11 BOOL  ; 2St_出料定位 工作完成
D1032.12 BOOL  ; 2St_出料定位 初始化[T]
D1032.13 BOOL  ; 2St_出料定位 单步[T]
D1032.14 BOOL  ; 2St_出料定位 单周期[T]
D1032.15 BOOL  ; 2St_出料定位 任务停止[T]
D1033.00 BOOL  ; 2St_出料定位 工站完成置位[T]
D1033.01 BOOL  ; 2St_出料定位 工站完成复位[T]
D1033.02 BOOL  ; 2St_出料定位 数据清除[T]
D1033.03 BOOL  ; 2St_出料定位 工站屏蔽[T]
D1033.04 BOOL  ; $?St$Bk?_#[110] / 2St_出料定位"$?St$Bk?_#[110]
D1033.06 BOOL  ; $?St$Bk?_#[112] / 2St_出料定位"$?St$Bk?_#[112]
D1033.08 BOOL  ; $?St$Bk?_#[114] / 2St_出料定位"$?St$Bk?_#[114]
D1033.10 BOOL  ; $?St$Bk?_#[116] / 2St_出料定位"$?St$Bk?_#[116]
D1033.12 BOOL  ; $?St$Bk?_#[118] / 2St_出料定位"$?St$Bk?_#[118]
D1033.14 BOOL  ; $?St$Bk?_#[120] / 2St_出料定位"$?St$Bk?_#[120]
D1034.00 BOOL  ; 2St_出料定位上游就绪-0
D1034.01 BOOL  ; 2St_出料定位使能上游-0
D1034.02 BOOL  ; 2St_出料定位上游就绪-1
D1034.03 BOOL  ; 2St_出料定位使能上游-1
D1034.04 BOOL  ; 2St_出料定位上游就绪-2
D1034.05 BOOL  ; 2St_出料定位使能上游-2
D1034.06 BOOL  ; 2St_出料定位上游就绪-3
D1034.07 BOOL  ; 2St_出料定位使能上游-3
D1034.08 BOOL  ; 2St_出料定位下游就绪-0
D1034.09 BOOL  ; 2St_出料定位使能下游-0
D1034.10 BOOL  ; 2St_出料定位下游就绪-1
D1034.11 BOOL  ; 2St_出料定位使能下游-1
D1034.12 BOOL  ; 2St_出料定位下游就绪-2
D1034.13 BOOL  ; 2St_出料定位使能下游-2
D1034.14 BOOL  ; 2St_出料定位下游就绪-3
D1034.15 BOOL  ; 2St_出料定位使能下游-3
D1035 CHANNEL  ; 2ST_A 步序字
D1035.00 BOOL  ; 2St_出料定位递进启动
D1035.01 BOOL  ; 2St_出料定位步01前后左右夹紧
D1035.02 BOOL  ; 2St_出料定位步02 移动到出料位
D1035.03 BOOL  ; 2St_出料定位步03 全部松开
D1035.04 BOOL  ; 2St_出料定位步04 等待取料
D1035.05 BOOL  ; 2St_出料定位步05 回接料位
D1035.06 BOOL  ; 2St_出料定位步06
D1035.07 BOOL  ; 2St_出料定位步07
D1035.08 BOOL  ; 2St_出料定位步08
D1035.09 BOOL  ; 2St_出料定位步09
D1035.10 BOOL  ; 2St_出料定位步10
D1035.11 BOOL  ; 2St_出料定位步11
D1035.12 BOOL  ; 2St_出料定位步12
D1035.13 BOOL  ; 2St_出料定位步13
D1035.14 BOOL  ; 2St_出料定位步14
D1035.15 BOOL  ; 2St_出料定位步15
D1036.00 BOOL  ; 2St_出料定位步16
D1036.01 BOOL  ; 2St_出料定位步17
D1036.02 BOOL  ; 2St_出料定位步18
D1036.03 BOOL  ; 2St_出料定位步19
D1036.04 BOOL  ; 2St_出料定位步20
D1036.05 BOOL  ; 2St_出料定位步21
D1036.06 BOOL  ; 2St_出料定位步22
D1036.07 BOOL  ; 2St_出料定位步23
D1036.08 BOOL  ; 2St_出料定位步24
D1036.09 BOOL  ; 2St_出料定位步25
D1036.10 BOOL  ; 2St_出料定位步26
D1036.11 BOOL  ; 2St_出料定位步27
D1036.12 BOOL  ; 2St_出料定位步28
D1036.13 BOOL  ; 2St_出料定位步29
D1036.14 BOOL  ; 2St_出料定位步30
D1036.15 BOOL  ; 2St_出料定位步31
D1037.00 BOOL  ; 2St_出料定位初始化步号
D1037.01 BOOL  ; 2St_出料定位
D1037.02 BOOL  ; 2St_出料定位
D1037.03 BOOL  ; 2St_出料定位
D1037.04 BOOL  ; 2St_出料定位
D1037.05 BOOL  ; 2St_出料定位
D1037.06 BOOL  ; 2St_出料定位
D1037.07 BOOL  ; 2St_出料定位
D1037.08 BOOL  ; 2St_出料定位
D1037.09 BOOL  ; 2St_出料定位
D1037.10 BOOL  ; 2St_出料定位
D1037.11 BOOL  ; 2St_出料定位
D1037.12 BOOL  ; 2St_出料定位
D1037.13 BOOL  ; 2St_出料定位
D1037.14 BOOL  ; 2St_出料定位
D1037.15 BOOL  ; 2St_出料定位
D1038.00 BOOL  ; 2St_出料定位初始化_1全部回位
D1038.01 BOOL  ; 2St_出料定位初始化_2
D1038.02 BOOL  ; 2St_出料定位初始化_3
D1038.03 BOOL  ; 2St_出料定位初始化_4
D1038.04 BOOL  ; 2St_出料定位初始化_5
D1038.05 BOOL  ; 2St_出料定位初始化_6
D1038.06 BOOL  ; 2St_出料定位初始化_7
D1038.07 BOOL  ; 2St_出料定位初始化_8
D1038.08 BOOL  ; 2St_出料定位初始化_9
D1038.09 BOOL  ; 2St_出料定位初始化_10
D1038.10 BOOL  ; 2St_出料定位初始化_11
D1038.11 BOOL  ; 2St_出料定位初始化_12
D1038.12 BOOL  ; 2St_出料定位初始化_13
D1038.13 BOOL  ; 2St_出料定位初始化_14
D1038.14 BOOL  ; 2St_出料定位初始化_15
D1038.15 BOOL  ; 2St_出料定位初始化_16
D1039.00 BOOL  ; 2St_出料定位初始化_17
D1039.01 BOOL  ; 2St_出料定位初始化_18
D1039.02 BOOL  ; 2St_出料定位初始化_19
D1039.03 BOOL  ; 2St_出料定位初始化_20
D1039.04 BOOL  ; 2St_出料定位初始化_21
D1039.05 BOOL  ; 2St_出料定位初始化_22
D1039.06 BOOL  ; 2St_出料定位初始化_23
D1039.07 BOOL  ; 2St_出料定位初始化_24
D1039.08 BOOL  ; 2St_出料定位初始化_25
D1039.09 BOOL  ; 2St_出料定位初始化_26
D1039.10 BOOL  ; 2St_出料定位初始化_27
D1039.11 BOOL  ; 2St_出料定位初始化_28
D1039.12 BOOL  ; 2St_出料定位初始化_29
D1039.13 BOOL  ; 2St_出料定位初始化_30
D1039.14 BOOL  ; 2St_出料定位初始化_31
D1039.15 BOOL  ; 2St_出料定位初始化_32
D10400 CHANNEL  ; ST5520_A1 绝缘测试仪测试时间读取值(ASC)
D10401 CHANNEL  ; ST5520_A1 绝缘测试仪测试时间读取值
D1040.00 BOOL  ; 3St_进出料转移工站错误
D1040.01 BOOL  ; 3St_进出料转移工站警告
D1040.02 BOOL  ; 3St_进出料转移工站运行
D1040.03 BOOL  ; $?St$Bk?_#[122] / 3St_进出料转移"$?St$Bk?_#[122]
D1040.05 BOOL  ; $?St$Bk?_#[124] / 3St_进出料转移"$?St$Bk?_#[124]
D1040.07 BOOL  ; $?St$Bk?_#[126] / 3St_进出料转移"$?St$Bk?_#[126]
D1040.09 BOOL  ; $?St$Bk?_#[128] / 3St_进出料转移"$?St$Bk?_#[128]
D1040.11 BOOL  ; $?St$Bk?_#[130] / 3St_进出料转移"$?St$Bk?_#[130]
D1040.13 BOOL  ; $?St$Bk?_#[132] / 3St_进出料转移"$?St$Bk?_#[132]
D1040.15 BOOL  ; $?St$Bk?_#[134] / 3St_进出料转移"$?St$Bk?_#[134]
D1041.04 BOOL  ; $?St$Bk?_#[136] / 3St_进出料转移"$?St$Bk?_#[136]
D1041.06 BOOL  ; $?St$Bk?_#[138] / 3St_进出料转移"$?St$Bk?_#[138]
D1041.08 BOOL  ; $?St$Bk?_#[140] / 3St_进出料转移"$?St$Bk?_#[140]
D1041.10 BOOL  ; $?St$Bk?_#[142] / 3St_进出料转移"$?St$Bk?_#[142]
D1041.12 BOOL  ; $?St$Bk?_#[144] / 3St_进出料转移"$?St$Bk?_#[144]
D1041.14 BOOL  ; $?St$Bk?_#[146] / 3St_进出料转移"$?St$Bk?_#[146]
D1042.00 BOOL  ; 3St_进出料转移工站就绪
D1042.01 BOOL  ; 3St_进出料转移 初始化中
D1042.02 BOOL  ; 3St_进出料转移 自动停止中
D1042.03 BOOL  ; 3St_进出料转移 自动停止完成
D1042.04 BOOL  ; 3St_进出料转移 联锁
D1042.05 BOOL  ; 3St_进出料转移 单步中
D1042.06 BOOL  ; 3St_进出料转移 单周期中
D1042.07 BOOL  ; 3St_进出料转移 周期完成
D1042.08 BOOL  ; 3St_进出料转移 任务开始
D1042.09 BOOL  ; 3St_进出料转移 任务递进条件
D1042.10 BOOL  ; 3St_进出料转移 任务递进
D1042.11 BOOL  ; 3St_进出料转移 工作完成
D1042.12 BOOL  ; 3St_进出料转移 初始化[T]
D1042.13 BOOL  ; 3St_进出料转移 单步[T]
D1042.14 BOOL  ; 3St_进出料转移 单周期[T]
D1042.15 BOOL  ; 3St_进出料转移 任务停止[T]
D1043.00 BOOL  ; 3St_进出料转移伸缩伺服回平台取料位条件
D1043.01 BOOL  ; 3St_进出料转移进料平台取料
D1043.02 BOOL  ; 3St_进出料转移出料平台放料
D1043.03 BOOL  ; 3St_进出料转移 工站屏蔽[T]
D1043.04 BOOL  ; $?St$Bk?_#[148] / 3St_进出料转移"$?St$Bk?_#[148]
D1043.06 BOOL  ; $?St$Bk?_#[150] / 3St_进出料转移"$?St$Bk?_#[150]
D1043.08 BOOL  ; $?St$Bk?_#[152] / 3St_进出料转移"$?St$Bk?_#[152]
D1043.10 BOOL  ; $?St$Bk?_#[154] / 3St_进出料转移"$?St$Bk?_#[154]
D1043.12 BOOL  ; $?St$Bk?_#[156] / 3St_进出料转移"$?St$Bk?_#[156]
D1043.14 BOOL  ; $?St$Bk?_#[158] / 3St_进出料转移"$?St$Bk?_#[158]
D1044.00 BOOL  ; 3St_进出料转移上游就绪-0
D1044.01 BOOL  ; 3St_进出料转移使能上游-0
D1044.02 BOOL  ; 3St_进出料转移上游就绪-1
D1044.03 BOOL  ; 3St_进出料转移使能上游-1
D1044.04 BOOL  ; 3St_进出料转移上游就绪-2
D1044.05 BOOL  ; 3St_进出料转移使能上游-2
D1044.06 BOOL  ; 3St_进出料转移上游就绪-3
D1044.07 BOOL  ; 3St_进出料转移使能上游-3
D1044.08 BOOL  ; 3St_进出料转移下游就绪-0
D1044.09 BOOL  ; 3St_进出料转移使能下游-0
D1044.10 BOOL  ; 3St_进出料转移下游就绪-1
D1044.11 BOOL  ; 3St_进出料转移使能下游-1
D1044.12 BOOL  ; 3St_进出料转移下游就绪-2
D1044.13 BOOL  ; 3St_进出料转移使能下游-2
D1044.14 BOOL  ; 3St_进出料转移下游就绪-3
D1044.15 BOOL  ; 3St_进出料转移使能下游-3
D1045 CHANNEL  ; 1ST自动步存放字
D1045.00 BOOL  ; 3St_进出料转移递进启动
D1045.01 BOOL  ; 3St_进出料转移步01 伸缩伺服平台取料位
D1045.02 BOOL  ; 3St_进出料转移步01 伸缩伺服平台回待料位
D1045.03 BOOL  ; 3St_进出料转移步03 进料夹爪两边夹紧
D1045.04 BOOL  ; 3St_进出料转移步04 进料夹爪左右下压|夹爪上升
D1045.05 BOOL  ; 3St_进出料转移步05 伸缩伺服回初始位
D1045.06 BOOL  ; 3St_进出料转移步06 取放位选择
D1045.07 BOOL  ; 3St_进出料转移步07 横移伺服到取料位
D1045.08 BOOL  ; 3St_进出料转移步08 伸缩伺服到热压取料位
D1045.09 BOOL  ; 3St_进出料转移步09 出料夹爪下降
D1045.10 BOOL  ; 3St_进出料转移步10 出料夹爪夹紧
D1045.11 BOOL  ; 3St_进出料转移步11 出料夹爪左右压紧|上升
D1045.12 BOOL  ; 3St_进出料转移步12 横移到放料位
D1045.13 BOOL  ; 3St_进出料转移步13 进料夹爪下降
D1045.14 BOOL  ; 3St_进出料转移步14 进料夹爪中间下降|左右上升
D1045.15 BOOL  ; 3St_进出料转移步15 进料夹爪左右松开|中间上升
D1046 CHANNEL  ; 3ST_A自动步存放字
D1046.00 BOOL  ; 3St_进出料转移步16
D1046.01 BOOL  ; 3St_进出料转移步17
D1046.02 BOOL  ; 3St_进出料转移步18
D1046.03 BOOL  ; 3St_进出料转移步19
D1046.04 BOOL  ; 3St_进出料转移步20
D1046.05 BOOL  ; 3St_进出料转移步21
D1046.06 BOOL  ; 3St_进出料转移步22
D1046.07 BOOL  ; 3St_进出料转移步23
D1046.08 BOOL  ; 3St_进出料转移步24
D1046.09 BOOL  ; 3St_进出料转移步25
D1046.10 BOOL  ; 3St_进出料转移步26
D1046.11 BOOL  ; 3St_进出料转移步27
D1046.12 BOOL  ; 3St_进出料转移步28
D1046.13 BOOL  ; 3St_进出料转移步29
D1046.14 BOOL  ; 3St_进出料转移步30
D1046.15 BOOL  ; 3St_进出料转移步31
D1047.00 BOOL  ; 3St_进出料转移初始化步号
D1047.01 BOOL  ; 3St_进出料转移
D1047.02 BOOL  ; 3St_进出料转移
D1047.03 BOOL  ; 3St_进出料转移
D1047.04 BOOL  ; 3St_进出料转移
D1047.05 BOOL  ; 3St_进出料转移
D1047.06 BOOL  ; 3St_进出料转移
D1047.07 BOOL  ; 3St_进出料转移
D1047.08 BOOL  ; 3St_进出料转移
D1047.09 BOOL  ; 3St_进出料转移
D1047.10 BOOL  ; 3St_进出料转移
D1047.11 BOOL  ; 3St_进出料转移
D1047.12 BOOL  ; 3St_进出料转移
D1047.13 BOOL  ; 3St_进出料转移
D1047.14 BOOL  ; 3St_进出料转移
D1047.15 BOOL  ; 3St_进出料转移
D1048.00 BOOL  ; 3St_进出料转移初始化_1
D1048.01 BOOL  ; 3St_进出料转移初始化_2
D1048.02 BOOL  ; 3St_进出料转移初始化_3
D1048.03 BOOL  ; 3St_进出料转移初始化_4
D1048.04 BOOL  ; 3St_进出料转移初始化_5
D1048.05 BOOL  ; 3St_进出料转移初始化_6
D1048.06 BOOL  ; 3St_进出料转移初始化_7
D1048.07 BOOL  ; 3St_进出料转移初始化_8
D1048.08 BOOL  ; 3St_进出料转移初始化_9
D1048.09 BOOL  ; 3St_进出料转移初始化_10
D1048.10 BOOL  ; 3St_进出料转移初始化_11
D1048.11 BOOL  ; 3St_进出料转移初始化_12
D1048.12 BOOL  ; 3St_进出料转移初始化_13
D1048.13 BOOL  ; 3St_进出料转移初始化_14
D1048.14 BOOL  ; 3St_进出料转移初始化_15
D1048.15 BOOL  ; 3St_进出料转移初始化_16
D1049.00 BOOL  ; 3St_进出料转移初始化_17
D1049.01 BOOL  ; 3St_进出料转移初始化_18
D1049.02 BOOL  ; 3St_进出料转移初始化_19
D1049.03 BOOL  ; 3St_进出料转移初始化_20
D1049.04 BOOL  ; 3St_进出料转移初始化_21
D1049.05 BOOL  ; 3St_进出料转移初始化_22
D1049.06 BOOL  ; 3St_进出料转移初始化_23
D1049.07 BOOL  ; 3St_进出料转移初始化_24
D1049.08 BOOL  ; 3St_进出料转移初始化_25
D1049.09 BOOL  ; 3St_进出料转移初始化_26
D1049.10 BOOL  ; 3St_进出料转移初始化_27
D1049.11 BOOL  ; 3St_进出料转移初始化_28
D1049.12 BOOL  ; 3St_进出料转移初始化_29
D1049.13 BOOL  ; 3St_进出料转移初始化_30
D1049.14 BOOL  ; 3St_进出料转移初始化_31
D1049.15 BOOL  ; 3St_进出料转移初始化_32
D1050.00 BOOL  ; 4St_1热压A工站错误
D1050.01 BOOL  ; 4St_1热压A工站警告
D1050.02 BOOL  ; 4St_1热压A工站运行
D1050.03 BOOL  ; $?St$Bk?_#[160] / 4St_1热压A"$?St$Bk?_#[160]
D1050.05 BOOL  ; $?St$Bk?_#[162] / 4St_1热压A"$?St$Bk?_#[162]
D1050.07 BOOL  ; $?St$Bk?_#[164] / 4St_1热压A"$?St$Bk?_#[164]
D1050.09 BOOL  ; $?St$Bk?_#[166] / 4St_1热压A"$?St$Bk?_#[166]
D1050.11 BOOL  ; $?St$Bk?_#[168] / 4St_1热压A"$?St$Bk?_#[168]
D1050.13 BOOL  ; $?St$Bk?_#[170] / 4St_1热压A"$?St$Bk?_#[170]
D1050.15 BOOL  ; $?St$Bk?_#[172] / 4St_1热压A"$?St$Bk?_#[172]
D1051.04 BOOL  ; $?St$Bk?_#[174] / 4St_1热压A"$?St$Bk?_#[174]
D1051.06 BOOL  ; $?St$Bk?_#[176] / 4St_1热压A"$?St$Bk?_#[176]
D1051.08 BOOL  ; $?St$Bk?_#[178] / 4St_1热压A"$?St$Bk?_#[178]
D1051.10 BOOL  ; $?St$Bk?_#[180] / 4St_1热压A"$?St$Bk?_#[180]
D1051.12 BOOL  ; $?St$Bk?_#[182] / 4St_1热压A"$?St$Bk?_#[182]
D1051.14 BOOL  ; $?St$Bk?_#[184] / 4St_1热压A"$?St$Bk?_#[184]
D1052.00 BOOL  ; 4St_1热压A工站就绪
D1052.01 BOOL  ; 4St_1热压A 初始化中
D1052.02 BOOL  ; 4St_1热压A 自动停止中
D1052.03 BOOL  ; 4St_1热压A 自动停止完成
D1052.04 BOOL  ; 4St_1热压A 联锁
D1052.05 BOOL  ; 4St_1热压A 单步中
D1052.06 BOOL  ; 4St_1热压A 单周期中
D1052.07 BOOL  ; 4St_1热压A 周期完成
D1052.08 BOOL  ; 4St_1热压A 任务开始
D1052.09 BOOL  ; 4St_1热压A 任务递进条件
D1052.10 BOOL  ; 4St_1热压A 任务递进
D1052.11 BOOL  ; 4St_1热压A 工作完成
D1052.12 BOOL  ; 4St_1热压A 初始化[T]
D1052.13 BOOL  ; 4St_1热压A 单步[T]
D1052.14 BOOL  ; 4St_1热压A 单周期[T]
D1052.15 BOOL  ; 4St_1热压A 任务停止[T]
D1053.00 BOOL  ; 4St_1热压A 工站完成置位[T]
D1053.01 BOOL  ; 4St_1热压A 工站完成复位[T]
D1053.02 BOOL  ; 4St_1热压A 数据清除[T]
D1053.03 BOOL  ; 4St_1热压A 工站屏蔽[T]
D1053.04 BOOL  ; $?St$Bk?_#[186] / 4St_1热压A"$?St$Bk?_#[186]
D1053.06 BOOL  ; $?St$Bk?_#[188] / 4St_1热压A"$?St$Bk?_#[188]
D1053.08 BOOL  ; $?St$Bk?_#[190] / 4St_1热压A"$?St$Bk?_#[190]
D1053.10 BOOL  ; $?St$Bk?_#[192] / 4St_1热压A"$?St$Bk?_#[192]
D1053.12 BOOL  ; $?St$Bk?_#[194] / 4St_1热压A"$?St$Bk?_#[194]
D1053.14 BOOL  ; $?St$Bk?_#[196] / 4St_1热压A"$?St$Bk?_#[196]
D1054.00 BOOL  ; 4St_1热压A上游就绪-0
D1054.01 BOOL  ; 4St_1热压A使能上游-0
D1054.02 BOOL  ; 4St_1热压A上游就绪-1
D1054.03 BOOL  ; 4St_1热压A使能上游-1
D1054.04 BOOL  ; 4St_1热压A上游就绪-2
D1054.05 BOOL  ; 4St_1热压A使能上游-2
D1054.06 BOOL  ; 4St_1热压A上游就绪-3
D1054.07 BOOL  ; 4St_1热压A使能上游-3
D1054.08 BOOL  ; 4St_1热压A下游就绪-0
D1054.09 BOOL  ; 4St_1热压A使能下游-0
D1054.10 BOOL  ; 4St_1热压A下游就绪-1
D1054.11 BOOL  ; 4St_1热压A使能下游-1
D1054.12 BOOL  ; 4St_1热压A下游就绪-2
D1054.13 BOOL  ; 4St_1热压A使能下游-2
D1054.14 BOOL  ; 4St_1热压A下游就绪-3
D1054.15 BOOL  ; 4St_1热压A使能下游-3
D1055 CHANNEL  ; 3ST_B进出料移栽自动步序
D1055.00 BOOL  ; 4St_1热压A递进启动
D1055.01 BOOL  ; 4St_1热压A步01
D1055.02 BOOL  ; 4St_1热压A步02
D1055.03 BOOL  ; 4St_1热压A步03
D1055.04 BOOL  ; 4St_1热压A步04
D1055.05 BOOL  ; 4St_1热压A步05
D1055.06 BOOL  ; 4St_1热压A步06
D1055.07 BOOL  ; 4St_1热压A步07
D1055.08 BOOL  ; 4St_1热压A步08
D1055.09 BOOL  ; 4St_1热压A步09
D1055.10 BOOL  ; 4St_1热压A步10
D1055.11 BOOL  ; 4St_1热压A步11
D1055.12 BOOL  ; 4St_1热压A步12
D1055.13 BOOL  ; 4St_1热压A步13
D1055.14 BOOL  ; 4St_1热压A步14
D1055.15 BOOL  ; 4St_1热压A步15
D1056 CHANNEL  ; 3ST_B进出料移栽自动步序
D1056.00 BOOL  ; 4St_1热压A步16
D1056.01 BOOL  ; 4St_1热压A步17
D1056.02 BOOL  ; 4St_1热压A步18
D1056.03 BOOL  ; 4St_1热压A步19
D1056.04 BOOL  ; 4St_1热压A步20
D1056.05 BOOL  ; 4St_1热压A步21
D1056.06 BOOL  ; 4St_1热压A步22
D1056.07 BOOL  ; 4St_1热压A步23
D1056.08 BOOL  ; 4St_1热压A步24
D1056.09 BOOL  ; 4St_1热压A步25
D1056.10 BOOL  ; 4St_1热压A步26
D1056.11 BOOL  ; 4St_1热压A步27
D1056.12 BOOL  ; 4St_1热压A步28
D1056.13 BOOL  ; 4St_1热压A步29
D1056.14 BOOL  ; 4St_1热压A步30
D1056.15 BOOL  ; 4St_1热压A步31
D1057.00 BOOL  ; 4St_1热压A初始化步号
D1057.01 BOOL  ; 4St_1热压A
D1057.02 BOOL  ; 4St_1热压A
D1057.03 BOOL  ; 4St_1热压A
D1057.04 BOOL  ; 4St_1热压A
D1057.05 BOOL  ; 4St_1热压A
D1057.06 BOOL  ; 4St_1热压A
D1057.07 BOOL  ; 4St_1热压A
D1057.08 BOOL  ; 4St_1热压A
D1057.09 BOOL  ; 4St_1热压A
D1057.10 BOOL  ; 4St_1热压A
D1057.11 BOOL  ; 4St_1热压A
D1057.12 BOOL  ; 4St_1热压A
D1057.13 BOOL  ; 4St_1热压A
D1057.14 BOOL  ; 4St_1热压A
D1057.15 BOOL  ; 4St_1热压A
D1058.00 BOOL  ; 4St_1热压A初始化_1
D1058.01 BOOL  ; 4St_1热压A初始化_2
D1058.02 BOOL  ; 4St_1热压A初始化_3
D1058.03 BOOL  ; 4St_1热压A初始化_4
D1058.04 BOOL  ; 4St_1热压A初始化_5
D1058.05 BOOL  ; 4St_1热压A初始化_6
D1058.06 BOOL  ; 4St_1热压A初始化_7
D1058.07 BOOL  ; 4St_1热压A初始化_8
D1058.08 BOOL  ; 4St_1热压A初始化_9
D1058.09 BOOL  ; 4St_1热压A初始化_10
D1058.10 BOOL  ; 4St_1热压A初始化_11
D1058.11 BOOL  ; 4St_1热压A初始化_12
D1058.12 BOOL  ; 4St_1热压A初始化_13
D1058.13 BOOL  ; 4St_1热压A初始化_14
D1058.14 BOOL  ; 4St_1热压A初始化_15
D1058.15 BOOL  ; 4St_1热压A初始化_16
D1059.00 BOOL  ; 4St_1热压A初始化_17
D1059.01 BOOL  ; 4St_1热压A初始化_18
D1059.02 BOOL  ; 4St_1热压A初始化_19
D1059.03 BOOL  ; 4St_1热压A初始化_20
D1059.04 BOOL  ; 4St_1热压A初始化_21
D1059.05 BOOL  ; 4St_1热压A初始化_22
D1059.06 BOOL  ; 4St_1热压A初始化_23
D1059.07 BOOL  ; 4St_1热压A初始化_24
D1059.08 BOOL  ; 4St_1热压A初始化_25
D1059.09 BOOL  ; 4St_1热压A初始化_26
D1059.10 BOOL  ; 4St_1热压A初始化_27
D1059.11 BOOL  ; 4St_1热压A初始化_28
D1059.12 BOOL  ; 4St_1热压A初始化_29
D1059.13 BOOL  ; 4St_1热压A初始化_30
D1059.14 BOOL  ; 4St_1热压A初始化_31
D1059.15 BOOL  ; 4St_1热压A初始化_32
D10600 CHANNEL  ; $?St$Bk?_#[197] / String "AUTO"$?St$Bk?_#[197]
D1060.00 BOOL  ; 4St_2热压B工站错误
D1060.01 BOOL  ; 4St_2热压B工站警告
D1060.02 BOOL  ; 4St_2热压B工站运行
D1060.03 BOOL  ; $?St$Bk?_#[199] / 4St_2热压B"$?St$Bk?_#[199]
D1060.05 BOOL  ; $?St$Bk?_#[201] / 4St_2热压B"$?St$Bk?_#[201]
D1060.07 BOOL  ; $?St$Bk?_#[203] / 4St_2热压B"$?St$Bk?_#[203]
D1060.09 BOOL  ; $?St$Bk?_#[205] / 4St_2热压B"$?St$Bk?_#[205]
D1060.11 BOOL  ; $?St$Bk?_#[207] / 4St_2热压B"$?St$Bk?_#[207]
D1060.13 BOOL  ; $?St$Bk?_#[209] / 4St_2热压B"$?St$Bk?_#[209]
D1060.15 BOOL  ; $?St$Bk?_#[212] / 4St_2热压B"$?St$Bk?_#[212]
D1061.04 BOOL  ; $?St$Bk?_#[214] / 4St_2热压B"$?St$Bk?_#[214]
D1061.06 BOOL  ; $?St$Bk?_#[216] / 4St_2热压B"$?St$Bk?_#[216]
D1061.08 BOOL  ; $?St$Bk?_#[218] / 4St_2热压B"$?St$Bk?_#[218]
D1061.10 BOOL  ; $?St$Bk?_#[220] / 4St_2热压B"$?St$Bk?_#[220]
D1061.12 BOOL  ; $?St$Bk?_#[222] / 4St_2热压B"$?St$Bk?_#[222]
D1061.14 BOOL  ; $?St$Bk?_#[224] / 4St_2热压B"$?St$Bk?_#[224]
D10620 CHANNEL  ; $?St$Bk?_#[225] / String "20M"$?St$Bk?_#[225]
D1062.00 BOOL  ; 4St_2热压B工站就绪
D1062.01 BOOL  ; 4St_2热压B 初始化中
D1062.02 BOOL  ; 4St_2热压B 自动停止中
D1062.03 BOOL  ; 4St_2热压B 自动停止完成
D1062.04 BOOL  ; 4St_2热压B 联锁
D1062.05 BOOL  ; 4St_2热压B 单步中
D1062.06 BOOL  ; 4St_2热压B 单周期中
D1062.07 BOOL  ; 4St_2热压B 周期完成
D1062.08 BOOL  ; 4St_2热压B 任务开始
D1062.09 BOOL  ; 4St_2热压B 任务递进条件
D1062.10 BOOL  ; 4St_2热压B 任务递进
D1062.11 BOOL  ; 4St_2热压B 工作完成
D1062.12 BOOL  ; 4St_2热压B 初始化[T]
D1062.13 BOOL  ; 4St_2热压B 单步[T]
D1062.14 BOOL  ; 4St_2热压B 单周期[T]
D1062.15 BOOL  ; 4St_2热压B 任务停止[T]
D10630 CHANNEL  ; $?St$Bk?_#[226] / String "200M"$?St$Bk?_#[226]
D1063.00 BOOL  ; 4St_2热压B 工站完成置位[T]
D1063.01 BOOL  ; 4St_2热压B 工站完成复位[T]
D1063.02 BOOL  ; 4St_2热压B 数据清除[T]
D1063.03 BOOL  ; 4St_2热压B 工站屏蔽[T]
D1063.04 BOOL  ; $?St$Bk?_#[228] / 4St_2热压B"$?St$Bk?_#[228]
D1063.06 BOOL  ; $?St$Bk?_#[230] / 4St_2热压B"$?St$Bk?_#[230]
D1063.08 BOOL  ; $?St$Bk?_#[232] / 4St_2热压B"$?St$Bk?_#[232]
D1063.10 BOOL  ; $?St$Bk?_#[234] / 4St_2热压B"$?St$Bk?_#[234]
D1063.12 BOOL  ; $?St$Bk?_#[236] / 4St_2热压B"$?St$Bk?_#[236]
D1063.14 BOOL  ; $?St$Bk?_#[238] / 4St_2热压B"$?St$Bk?_#[238]
D10640 CHANNEL  ; $?St$Bk?_#[239] / String "2000M"$?St$Bk?_#[239]
D1064.00 BOOL  ; 4St_2热压B上游就绪-0
D1064.01 BOOL  ; 4St_2热压B使能上游-0
D1064.02 BOOL  ; 4St_2热压B上游就绪-1
D1064.03 BOOL  ; 4St_2热压B使能上游-1
D1064.04 BOOL  ; 4St_2热压B上游就绪-2
D1064.05 BOOL  ; 4St_2热压B使能上游-2
D1064.06 BOOL  ; 4St_2热压B上游就绪-3
D1064.07 BOOL  ; 4St_2热压B使能上游-3
D1064.08 BOOL  ; 4St_2热压B下游就绪-0
D1064.09 BOOL  ; 4St_2热压B使能下游-0
D1064.10 BOOL  ; 4St_2热压B下游就绪-1
D1064.11 BOOL  ; 4St_2热压B使能下游-1
D1064.12 BOOL  ; 4St_2热压B下游就绪-2
D1064.13 BOOL  ; 4St_2热压B使能下游-2
D1064.14 BOOL  ; 4St_2热压B下游就绪-3
D1064.15 BOOL  ; 4St_2热压B使能下游-3
D1065 CHANNEL  ; 4ST_A 热压A步序字
D10650 CHANNEL  ; $?St$Bk?_#[240] / String "4000M"$?St$Bk?_#[240]
D1065.00 BOOL  ; 4St_2热压B递进启动
D1065.01 BOOL  ; 4St_2热压B步01
D1065.02 BOOL  ; 4St_2热压B步02
D1065.03 BOOL  ; 4St_2热压B步03
D1065.04 BOOL  ; 4St_2热压B步04
D1065.05 BOOL  ; 4St_2热压B步05
D1065.06 BOOL  ; 4St_2热压B步06
D1065.07 BOOL  ; 4St_2热压B步07
D1065.08 BOOL  ; 4St_2热压B步08
D1065.09 BOOL  ; 4St_2热压B步09
D1065.10 BOOL  ; 4St_2热压B步10
D1065.11 BOOL  ; 4St_2热压B步11
D1065.12 BOOL  ; 4St_2热压B步12
D1065.13 BOOL  ; 4St_2热压B步13
D1065.14 BOOL  ; 4St_2热压B步14
D1065.15 BOOL  ; 4St_2热压B步15
D10660 CHANNEL  ; $?St$Bk?_#[241] / "FAST"$?St$Bk?_#[241]
D1066.00 BOOL  ; 4St_2热压B步16
D1066.01 BOOL  ; 4St_2热压B步17
D1066.02 BOOL  ; 4St_2热压B步18
D1066.03 BOOL  ; 4St_2热压B步19
D1066.04 BOOL  ; 4St_2热压B步20
D1066.05 BOOL  ; 4St_2热压B步21
D1066.06 BOOL  ; 4St_2热压B步22
D1066.07 BOOL  ; 4St_2热压B步23
D1066.08 BOOL  ; 4St_2热压B步24
D1066.09 BOOL  ; 4St_2热压B步25
D1066.10 BOOL  ; 4St_2热压B步26
D1066.11 BOOL  ; 4St_2热压B步27
D1066.12 BOOL  ; 4St_2热压B步28
D1066.13 BOOL  ; 4St_2热压B步29
D1066.14 BOOL  ; 4St_2热压B步30
D1066.15 BOOL  ; 4St_2热压B步31
D10670 CHANNEL  ; $?St$Bk?_#[242] / "SLOW"$?St$Bk?_#[242]
D1067.00 BOOL  ; 4St_2热压B初始化步号
D1067.01 BOOL  ; 4St_2热压B
D1067.02 BOOL  ; 4St_2热压B
D1067.03 BOOL  ; 4St_2热压B
D1067.04 BOOL  ; 4St_2热压B
D1067.05 BOOL  ; 4St_2热压B
D1067.06 BOOL  ; 4St_2热压B
D1067.07 BOOL  ; 4St_2热压B
D1067.08 BOOL  ; 4St_2热压B
D1067.09 BOOL  ; 4St_2热压B
D1067.10 BOOL  ; 4St_2热压B
D1067.11 BOOL  ; 4St_2热压B
D1067.12 BOOL  ; 4St_2热压B
D1067.13 BOOL  ; 4St_2热压B
D1067.14 BOOL  ; 4St_2热压B
D1067.15 BOOL  ; 4St_2热压B
D1068.00 BOOL  ; 4St_2热压B初始化_1
D1068.01 BOOL  ; 4St_2热压B初始化_2
D1068.02 BOOL  ; 4St_2热压B初始化_3
D1068.03 BOOL  ; 4St_2热压B初始化_4
D1068.04 BOOL  ; 4St_2热压B初始化_5
D1068.05 BOOL  ; 4St_2热压B初始化_6
D1068.06 BOOL  ; 4St_2热压B初始化_7
D1068.07 BOOL  ; 4St_2热压B初始化_8
D1068.08 BOOL  ; 4St_2热压B初始化_9
D1068.09 BOOL  ; 4St_2热压B初始化_10
D1068.10 BOOL  ; 4St_2热压B初始化_11
D1068.11 BOOL  ; 4St_2热压B初始化_12
D1068.12 BOOL  ; 4St_2热压B初始化_13
D1068.13 BOOL  ; 4St_2热压B初始化_14
D1068.14 BOOL  ; 4St_2热压B初始化_15
D1068.15 BOOL  ; 4St_2热压B初始化_16
D1069.00 BOOL  ; 4St_2热压B初始化_17
D1069.01 BOOL  ; 4St_2热压B初始化_18
D1069.02 BOOL  ; 4St_2热压B初始化_19
D1069.03 BOOL  ; 4St_2热压B初始化_20
D1069.04 BOOL  ; 4St_2热压B初始化_21
D1069.05 BOOL  ; 4St_2热压B初始化_22
D1069.06 BOOL  ; 4St_2热压B初始化_23
D1069.07 BOOL  ; 4St_2热压B初始化_24
D1069.08 BOOL  ; 4St_2热压B初始化_25
D1069.09 BOOL  ; 4St_2热压B初始化_26
D1069.10 BOOL  ; 4St_2热压B初始化_27
D1069.11 BOOL  ; 4St_2热压B初始化_28
D1069.12 BOOL  ; 4St_2热压B初始化_29
D1069.13 BOOL  ; 4St_2热压B初始化_30
D1069.14 BOOL  ; 4St_2热压B初始化_31
D1069.15 BOOL  ; 4St_2热压B初始化_32
D10700 CHANNEL  ; $?St$Bk?_#[243] / String "CONTINUE"$?St$Bk?_#[243]
D10701 CHANNEL  ; $?St$Bk?_#[244] / String "CONTINUE"$?St$Bk?_#[244]
D10702 CHANNEL  ; $?St$Bk?_#[245] / String "CONTINUE"$?St$Bk?_#[245]
D10703 CHANNEL  ; $?St$Bk?_#[246] / String "CONTINUE"$?St$Bk?_#[246]
D1070.00 BOOL  ; 4St_3热压C工站错误
D1070.01 BOOL  ; 4St_3热压C工站警告
D1070.02 BOOL  ; 4St_3热压C工站运行
D1070.03 BOOL  ; $?St$Bk?_#[248] / 4St_3热压C"$?St$Bk?_#[248]
D1070.05 BOOL  ; $?St$Bk?_#[250] / 4St_3热压C"$?St$Bk?_#[250]
D1070.07 BOOL  ; $?St$Bk?_#[252] / 4St_3热压C"$?St$Bk?_#[252]
D1070.09 BOOL  ; $?St$Bk?_#[254] / 4St_3热压C"$?St$Bk?_#[254]
D1070.11 BOOL  ; $?St$Bk?_#[256] / 4St_3热压C"$?St$Bk?_#[256]
D1070.13 BOOL  ; $?St$Bk?_#[258] / 4St_3热压C"$?St$Bk?_#[258]
D1070.15 BOOL  ; $?St$Bk?_#[264] / 4St_3热压C"$?St$Bk?_#[264]
D1071.04 BOOL  ; $?St$Bk?_#[266] / 4St_3热压C"$?St$Bk?_#[266]
D1071.06 BOOL  ; $?St$Bk?_#[268] / 4St_3热压C"$?St$Bk?_#[268]
D1071.08 BOOL  ; $?St$Bk?_#[270] / 4St_3热压C"$?St$Bk?_#[270]
D1071.10 BOOL  ; $?St$Bk?_#[272] / 4St_3热压C"$?St$Bk?_#[272]
D1071.12 BOOL  ; $?St$Bk?_#[274] / 4St_3热压C"$?St$Bk?_#[274]
D1071.14 BOOL  ; $?St$Bk?_#[276] / 4St_3热压C"$?St$Bk?_#[276]
D10720 CHANNEL  ; $?St$Bk?_#[277] / String "FAILSTOP"$?St$Bk?_#[277]
D10721 CHANNEL  ; $?St$Bk?_#[278] / String "FAILSTOP"$?St$Bk?_#[278]
D10722 CHANNEL  ; $?St$Bk?_#[279] / String "FAILSTOP"$?St$Bk?_#[279]
D10723 CHANNEL  ; $?St$Bk?_#[280] / String "FAILSTOP"$?St$Bk?_#[280]
D1072.00 BOOL  ; 4St_3热压C工站就绪
D1072.01 BOOL  ; 4St_3热压C 初始化中
D1072.02 BOOL  ; 4St_3热压C 自动停止中
D1072.03 BOOL  ; 4St_3热压C 自动停止完成
D1072.04 BOOL  ; 4St_3热压C 联锁
D1072.05 BOOL  ; 4St_3热压C 单步中
D1072.06 BOOL  ; 4St_3热压C 单周期中
D1072.07 BOOL  ; 4St_3热压C 周期完成
D1072.08 BOOL  ; 4St_3热压C 任务开始
D1072.09 BOOL  ; 4St_3热压C 任务递进条件
D1072.10 BOOL  ; 4St_3热压C 任务递进
D1072.11 BOOL  ; 4St_3热压C 工作完成
D1072.12 BOOL  ; 4St_3热压C 初始化[T]
D1072.13 BOOL  ; 4St_3热压C 单步[T]
D1072.14 BOOL  ; 4St_3热压C 单周期[T]
D1072.15 BOOL  ; 4St_3热压C 任务停止[T]
D10730 CHANNEL  ; $?St$Bk?_#[281] / String "SEQUENCE"$?St$Bk?_#[281]
D10731 CHANNEL  ; $?St$Bk?_#[282] / String "SEQUENCE"$?St$Bk?_#[282]
D10732 CHANNEL  ; $?St$Bk?_#[283] / String "SEQUENCE"$?St$Bk?_#[283]
D10733 CHANNEL  ; $?St$Bk?_#[284] / String "SEQUENCE"$?St$Bk?_#[284]
D1073.00 BOOL  ; 4St_3热压C 工站完成置位[T]
D1073.01 BOOL  ; 4St_3热压C 工站完成复位[T]
D1073.02 BOOL  ; 4St_3热压C 数据清除[T]
D1073.03 BOOL  ; 4St_3热压C 工站屏蔽[T]
D1073.04 BOOL  ; $?St$Bk?_#[286] / 4St_3热压C"$?St$Bk?_#[286]
D1073.06 BOOL  ; $?St$Bk?_#[288] / 4St_3热压C"$?St$Bk?_#[288]
D1073.08 BOOL  ; $?St$Bk?_#[290] / 4St_3热压C"$?St$Bk?_#[290]
D1073.10 BOOL  ; $?St$Bk?_#[292] / 4St_3热压C"$?St$Bk?_#[292]
D1073.12 BOOL  ; $?St$Bk?_#[294] / 4St_3热压C"$?St$Bk?_#[294]
D1073.14 BOOL  ; $?St$Bk?_#[296] / 4St_3热压C"$?St$Bk?_#[296]
D1074.00 BOOL  ; 4St_3热压C上游就绪-0
D1074.01 BOOL  ; 4St_3热压C使能上游-0
D1074.02 BOOL  ; 4St_3热压C上游就绪-1
D1074.03 BOOL  ; 4St_3热压C使能上游-1
D1074.04 BOOL  ; 4St_3热压C上游就绪-2
D1074.05 BOOL  ; 4St_3热压C使能上游-2
D1074.06 BOOL  ; 4St_3热压C上游就绪-3
D1074.07 BOOL  ; 4St_3热压C使能上游-3
D1074.08 BOOL  ; 4St_3热压C下游就绪-0
D1074.09 BOOL  ; 4St_3热压C使能下游-0
D1074.10 BOOL  ; 4St_3热压C下游就绪-1
D1074.11 BOOL  ; 4St_3热压C使能下游-1
D1074.12 BOOL  ; 4St_3热压C下游就绪-2
D1074.13 BOOL  ; 4St_3热压C使能下游-2
D1074.14 BOOL  ; 4St_3热压C下游就绪-3
D1074.15 BOOL  ; 4St_3热压C使能下游-3
D1075 CHANNEL  ; 4ST_B 自动步存放字
D1075.00 BOOL  ; 4St_3热压C递进启动
D1075.01 BOOL  ; 4St_3热压C步01
D1075.02 BOOL  ; 4St_3热压C步02
D1075.03 BOOL  ; 4St_3热压C步03
D1075.04 BOOL  ; 4St_3热压C步04
D1075.05 BOOL  ; 4St_3热压C步05
D1075.06 BOOL  ; 4St_3热压C步06
D1075.07 BOOL  ; 4St_3热压C步07
D1075.08 BOOL  ; 4St_3热压C步08
D1075.09 BOOL  ; 4St_3热压C步09
D1075.10 BOOL  ; 4St_3热压C步10
D1075.11 BOOL  ; 4St_3热压C步11
D1075.12 BOOL  ; 4St_3热压C步12
D1075.13 BOOL  ; 4St_3热压C步13
D1075.14 BOOL  ; 4St_3热压C步14
D1075.15 BOOL  ; 4St_3热压C步15
D1076.00 BOOL  ; 4St_3热压C步16
D1076.01 BOOL  ; 4St_3热压C步17
D1076.02 BOOL  ; 4St_3热压C步18
D1076.03 BOOL  ; 4St_3热压C步19
D1076.04 BOOL  ; 4St_3热压C步20
D1076.05 BOOL  ; 4St_3热压C步21
D1076.06 BOOL  ; 4St_3热压C步22
D1076.07 BOOL  ; 4St_3热压C步23
D1076.08 BOOL  ; 4St_3热压C步24
D1076.09 BOOL  ; 4St_3热压C步25
D1076.10 BOOL  ; 4St_3热压C步26
D1076.11 BOOL  ; 4St_3热压C步27
D1076.12 BOOL  ; 4St_3热压C步28
D1076.13 BOOL  ; 4St_3热压C步29
D1076.14 BOOL  ; 4St_3热压C步30
D1076.15 BOOL  ; 4St_3热压C步31
D1077.00 BOOL  ; 4St_3热压C初始化步号
D1077.01 BOOL  ; 4St_3热压C
D1077.02 BOOL  ; 4St_3热压C
D1077.03 BOOL  ; 4St_3热压C
D1077.04 BOOL  ; 4St_3热压C
D1077.05 BOOL  ; 4St_3热压C
D1077.06 BOOL  ; 4St_3热压C
D1077.07 BOOL  ; 4St_3热压C
D1077.08 BOOL  ; 4St_3热压C
D1077.09 BOOL  ; 4St_3热压C
D1077.10 BOOL  ; 4St_3热压C
D1077.11 BOOL  ; 4St_3热压C
D1077.12 BOOL  ; 4St_3热压C
D1077.13 BOOL  ; 4St_3热压C
D1077.14 BOOL  ; 4St_3热压C
D1077.15 BOOL  ; 4St_3热压C
D1078.00 BOOL  ; 4St_3热压C初始化_1
D1078.01 BOOL  ; 4St_3热压C初始化_2
D1078.02 BOOL  ; 4St_3热压C初始化_3
D1078.03 BOOL  ; 4St_3热压C初始化_4
D1078.04 BOOL  ; 4St_3热压C初始化_5
D1078.05 BOOL  ; 4St_3热压C初始化_6
D1078.06 BOOL  ; 4St_3热压C初始化_7
D1078.07 BOOL  ; 4St_3热压C初始化_8
D1078.08 BOOL  ; 4St_3热压C初始化_9
D1078.09 BOOL  ; 4St_3热压C初始化_10
D1078.10 BOOL  ; 4St_3热压C初始化_11
D1078.11 BOOL  ; 4St_3热压C初始化_12
D1078.12 BOOL  ; 4St_3热压C初始化_13
D1078.13 BOOL  ; 4St_3热压C初始化_14
D1078.14 BOOL  ; 4St_3热压C初始化_15
D1078.15 BOOL  ; 4St_3热压C初始化_16
D1079.00 BOOL  ; 4St_3热压C初始化_17
D1079.01 BOOL  ; 4St_3热压C初始化_18
D1079.02 BOOL  ; 4St_3热压C初始化_19
D1079.03 BOOL  ; 4St_3热压C初始化_20
D1079.04 BOOL  ; 4St_3热压C初始化_21
D1079.05 BOOL  ; 4St_3热压C初始化_22
D1079.06 BOOL  ; 4St_3热压C初始化_23
D1079.07 BOOL  ; 4St_3热压C初始化_24
D1079.08 BOOL  ; 4St_3热压C初始化_25
D1079.09 BOOL  ; 4St_3热压C初始化_26
D1079.10 BOOL  ; 4St_3热压C初始化_27
D1079.11 BOOL  ; 4St_3热压C初始化_28
D1079.12 BOOL  ; 4St_3热压C初始化_29
D1079.13 BOOL  ; 4St_3热压C初始化_30
D1079.14 BOOL  ; 4St_3热压C初始化_31
D1079.15 BOOL  ; 4St_3热压C初始化_32
D1080.00 BOOL  ; 5St_A出料定位A工站错误
D1080.01 BOOL  ; 5St_A出料定位A工站警告
D1080.02 BOOL  ; 5St_A出料定位A工站运行
D1080.03 BOOL  ; $?St$Bk?_#[298] / 5St_A出料定位A"$?St$Bk?_#[298]
D1080.05 BOOL  ; $?St$Bk?_#[300] / 5St_A出料定位A"$?St$Bk?_#[300]
D1080.07 BOOL  ; $?St$Bk?_#[302] / 5St_A出料定位A"$?St$Bk?_#[302]
D1080.09 BOOL  ; $?St$Bk?_#[304] / 5St_A出料定位A"$?St$Bk?_#[304]
D1080.11 BOOL  ; $?St$Bk?_#[306] / 5St_A出料定位A"$?St$Bk?_#[306]
D1080.13 BOOL  ; $?St$Bk?_#[308] / 5St_A出料定位A"$?St$Bk?_#[308]
D1080.15 BOOL  ; $?St$Bk?_#[310] / 5St_A出料定位A"$?St$Bk?_#[310]
D1081.04 BOOL  ; $?St$Bk?_#[312] / 5St_A出料定位A"$?St$Bk?_#[312]
D1081.06 BOOL  ; $?St$Bk?_#[314] / 5St_A出料定位A"$?St$Bk?_#[314]
D1081.08 BOOL  ; $?St$Bk?_#[316] / 5St_A出料定位A"$?St$Bk?_#[316]
D1081.10 BOOL  ; $?St$Bk?_#[318] / 5St_A出料定位A"$?St$Bk?_#[318]
D1081.12 BOOL  ; $?St$Bk?_#[320] / 5St_A出料定位A"$?St$Bk?_#[320]
D1081.14 BOOL  ; $?St$Bk?_#[322] / 5St_A出料定位A"$?St$Bk?_#[322]
D1082.00 BOOL  ; 5St_A出料定位A工站就绪
D1082.01 BOOL  ; 5St_A出料定位A 初始化中
D1082.02 BOOL  ; 5St_A出料定位A 自动停止中
D1082.03 BOOL  ; 5St_A出料定位A 自动停止完成
D1082.04 BOOL  ; 5St_A出料定位A 联锁
D1082.05 BOOL  ; 5St_A出料定位A 单步中
D1082.06 BOOL  ; 5St_A出料定位A 单周期中
D1082.07 BOOL  ; 5St_A出料定位A 周期完成
D1082.08 BOOL  ; 5St_A出料定位A 任务开始
D1082.09 BOOL  ; 5St_A出料定位A 任务递进条件
D1082.10 BOOL  ; 5St_A出料定位A 任务递进
D1082.11 BOOL  ; 5St_A出料定位A 工作完成
D1082.12 BOOL  ; 5St_A出料定位A 初始化[T]
D1082.13 BOOL  ; 5St_A出料定位A 单步[T]
D1082.14 BOOL  ; 5St_A出料定位A 单周期[T]
D1082.15 BOOL  ; 5St_A出料定位A 任务停止[T]
D1083.00 BOOL  ; 5St_A出料定位A 工站完成置位[T]
D1083.01 BOOL  ; 5St_A出料定位A 工站完成复位[T]
D1083.02 BOOL  ; 5St_A出料定位A 数据清除[T]
D1083.03 BOOL  ; 5St_A出料定位A 工站屏蔽[T]
D1083.04 BOOL  ; $?St$Bk?_#[324] / 5St_A出料定位A"$?St$Bk?_#[324]
D1083.06 BOOL  ; $?St$Bk?_#[326] / 5St_A出料定位A"$?St$Bk?_#[326]
D1083.08 BOOL  ; $?St$Bk?_#[328] / 5St_A出料定位A"$?St$Bk?_#[328]
D1083.10 BOOL  ; $?St$Bk?_#[330] / 5St_A出料定位A"$?St$Bk?_#[330]
D1083.12 BOOL  ; $?St$Bk?_#[332] / 5St_A出料定位A"$?St$Bk?_#[332]
D1083.14 BOOL  ; $?St$Bk?_#[334] / 5St_A出料定位A"$?St$Bk?_#[334]
D1084.00 BOOL  ; 5St_A出料定位A上游就绪-0
D1084.01 BOOL  ; 5St_A出料定位A使能上游-0
D1084.02 BOOL  ; 5St_A出料定位A上游就绪-1
D1084.03 BOOL  ; 5St_A出料定位A使能上游-1
D1084.04 BOOL  ; 5St_A出料定位A上游就绪-2
D1084.05 BOOL  ; 5St_A出料定位A使能上游-2
D1084.06 BOOL  ; 5St_A出料定位A上游就绪-3
D1084.07 BOOL  ; 5St_A出料定位A使能上游-3
D1084.08 BOOL  ; 5St_A出料定位A下游就绪-0
D1084.09 BOOL  ; 5St_A出料定位A使能下游-0
D1084.10 BOOL  ; 5St_A出料定位A下游就绪-1
D1084.11 BOOL  ; 5St_A出料定位A使能下游-1
D1084.12 BOOL  ; 5St_A出料定位A下游就绪-2
D1084.13 BOOL  ; 5St_A出料定位A使能下游-2
D1084.14 BOOL  ; 5St_A出料定位A下游就绪-3
D1084.15 BOOL  ; 5St_A出料定位A使能下游-3
D1085.00 BOOL  ; 5St_A出料定位A递进启动
D1085.01 BOOL  ; 5St_A出料定位A步01
D1085.02 BOOL  ; 5St_A出料定位A步02
D1085.03 BOOL  ; 5St_A出料定位A步03
D1085.04 BOOL  ; 5St_A出料定位A步04
D1085.05 BOOL  ; 5St_A出料定位A步05
D1085.06 BOOL  ; 5St_A出料定位A步06
D1085.07 BOOL  ; 5St_A出料定位A步07
D1085.08 BOOL  ; 5St_A出料定位A步08
D1085.09 BOOL  ; 5St_A出料定位A步09
D1085.10 BOOL  ; 5St_A出料定位A步10
D1085.11 BOOL  ; 5St_A出料定位A步11
D1085.12 BOOL  ; 5St_A出料定位A步12
D1085.13 BOOL  ; 5St_A出料定位A步13
D1085.14 BOOL  ; 5St_A出料定位A步14
D1085.15 BOOL  ; 5St_A出料定位A步15
D1086.00 BOOL  ; 5St_A出料定位A步16
D1086.01 BOOL  ; 5St_A出料定位A步17
D1086.02 BOOL  ; 5St_A出料定位A步18
D1086.03 BOOL  ; 5St_A出料定位A步19
D1086.04 BOOL  ; 5St_A出料定位A步20
D1086.05 BOOL  ; 5St_A出料定位A步21
D1086.06 BOOL  ; 5St_A出料定位A步22
D1086.07 BOOL  ; 5St_A出料定位A步23
D1086.08 BOOL  ; 5St_A出料定位A步24
D1086.09 BOOL  ; 5St_A出料定位A步25
D1086.10 BOOL  ; 5St_A出料定位A步26
D1086.11 BOOL  ; 5St_A出料定位A步27
D1086.12 BOOL  ; 5St_A出料定位A步28
D1086.13 BOOL  ; 5St_A出料定位A步29
D1086.14 BOOL  ; 5St_A出料定位A步30
D1086.15 BOOL  ; 5St_A出料定位A步31
D1087.00 BOOL  ; 5St_A出料定位A初始化步号
D1087.01 BOOL  ; 5St_A出料定位A
D1087.02 BOOL  ; 5St_A出料定位A
D1087.03 BOOL  ; 5St_A出料定位A
D1087.04 BOOL  ; 5St_A出料定位A
D1087.05 BOOL  ; 5St_A出料定位A
D1087.06 BOOL  ; 5St_A出料定位A
D1087.07 BOOL  ; 5St_A出料定位A
D1087.08 BOOL  ; 5St_A出料定位A
D1087.09 BOOL  ; 5St_A出料定位A
D1087.10 BOOL  ; 5St_A出料定位A
D1087.11 BOOL  ; 5St_A出料定位A
D1087.12 BOOL  ; 5St_A出料定位A
D1087.13 BOOL  ; 5St_A出料定位A
D1087.14 BOOL  ; 5St_A出料定位A
D1087.15 BOOL  ; 5St_A出料定位A
D1088.00 BOOL  ; 5St_A出料定位A初始化_1
D1088.01 BOOL  ; 5St_A出料定位A初始化_2
D1088.02 BOOL  ; 5St_A出料定位A初始化_3
D1088.03 BOOL  ; 5St_A出料定位A初始化_4
D1088.04 BOOL  ; 5St_A出料定位A初始化_5
D1088.05 BOOL  ; 5St_A出料定位A初始化_6
D1088.06 BOOL  ; 5St_A出料定位A初始化_7
D1088.07 BOOL  ; 5St_A出料定位A初始化_8
D1088.08 BOOL  ; 5St_A出料定位A初始化_9
D1088.09 BOOL  ; 5St_A出料定位A初始化_10
D1088.10 BOOL  ; 5St_A出料定位A初始化_11
D1088.11 BOOL  ; 5St_A出料定位A初始化_12
D1088.12 BOOL  ; 5St_A出料定位A初始化_13
D1088.13 BOOL  ; 5St_A出料定位A初始化_14
D1088.14 BOOL  ; 5St_A出料定位A初始化_15
D1088.15 BOOL  ; 5St_A出料定位A初始化_16
D1089.00 BOOL  ; 5St_A出料定位A初始化_17
D1089.01 BOOL  ; 5St_A出料定位A初始化_18
D1089.02 BOOL  ; 5St_A出料定位A初始化_19
D1089.03 BOOL  ; 5St_A出料定位A初始化_20
D1089.04 BOOL  ; 5St_A出料定位A初始化_21
D1089.05 BOOL  ; 5St_A出料定位A初始化_22
D1089.06 BOOL  ; 5St_A出料定位A初始化_23
D1089.07 BOOL  ; 5St_A出料定位A初始化_24
D1089.08 BOOL  ; 5St_A出料定位A初始化_25
D1089.09 BOOL  ; 5St_A出料定位A初始化_26
D1089.10 BOOL  ; 5St_A出料定位A初始化_27
D1089.11 BOOL  ; 5St_A出料定位A初始化_28
D1089.12 BOOL  ; 5St_A出料定位A初始化_29
D1089.13 BOOL  ; 5St_A出料定位A初始化_30
D1089.14 BOOL  ; 5St_A出料定位A初始化_31
D1089.15 BOOL  ; 5St_A出料定位A初始化_32
D1090.00 BOOL  ; 5St_B出料定位B工站错误
D1090.01 BOOL  ; 5St_B出料定位B工站警告
D1090.02 BOOL  ; 5St_B出料定位B工站运行
D1090.03 BOOL  ; $?St$Bk?_#[336] / 5St_B出料定位B"$?St$Bk?_#[336]
D1090.05 BOOL  ; $?St$Bk?_#[338] / 5St_B出料定位B"$?St$Bk?_#[338]
D1090.07 BOOL  ; $?St$Bk?_#[340] / 5St_B出料定位B"$?St$Bk?_#[340]
D1090.09 BOOL  ; $?St$Bk?_#[342] / 5St_B出料定位B"$?St$Bk?_#[342]
D1090.11 BOOL  ; $?St$Bk?_#[344] / 5St_B出料定位B"$?St$Bk?_#[344]
D1090.13 BOOL  ; $?St$Bk?_#[346] / 5St_B出料定位B"$?St$Bk?_#[346]
D1090.15 BOOL  ; $?St$Bk?_#[348] / 5St_B出料定位B"$?St$Bk?_#[348]
D1091.04 BOOL  ; $?St$Bk?_#[350] / 5St_B出料定位B"$?St$Bk?_#[350]
D1091.06 BOOL  ; $?St$Bk?_#[352] / 5St_B出料定位B"$?St$Bk?_#[352]
D1091.08 BOOL  ; $?St$Bk?_#[354] / 5St_B出料定位B"$?St$Bk?_#[354]
D1091.10 BOOL  ; $?St$Bk?_#[356] / 5St_B出料定位B"$?St$Bk?_#[356]
D1091.12 BOOL  ; $?St$Bk?_#[358] / 5St_B出料定位B"$?St$Bk?_#[358]
D1091.14 BOOL  ; $?St$Bk?_#[360] / 5St_B出料定位B"$?St$Bk?_#[360]
D1092.00 BOOL  ; 5St_B出料定位B工站就绪
D1092.01 BOOL  ; 5St_B出料定位B 初始化中
D1092.02 BOOL  ; 5St_B出料定位B 自动停止中
D1092.03 BOOL  ; 5St_B出料定位B 自动停止完成
D1092.04 BOOL  ; 5St_B出料定位B 联锁
D1092.05 BOOL  ; 5St_B出料定位B 单步中
D1092.06 BOOL  ; 5St_B出料定位B 单周期中
D1092.07 BOOL  ; 5St_B出料定位B 周期完成
D1092.08 BOOL  ; 5St_B出料定位B 任务开始
D1092.09 BOOL  ; 5St_B出料定位B 任务递进条件
D1092.10 BOOL  ; 5St_B出料定位B 任务递进
D1092.11 BOOL  ; 5St_B出料定位B 工作完成
D1092.12 BOOL  ; 5St_B出料定位B 初始化[T]
D1092.13 BOOL  ; 5St_B出料定位B 单步[T]
D1092.14 BOOL  ; 5St_B出料定位B 单周期[T]
D1092.15 BOOL  ; 5St_B出料定位B 任务停止[T]
D1093.00 BOOL  ; 5St_B出料定位B 工站完成置位[T]
D1093.01 BOOL  ; 5St_B出料定位B 工站完成复位[T]
D1093.02 BOOL  ; 5St_B出料定位B 数据清除[T]
D1093.03 BOOL  ; 5St_B出料定位B 工站屏蔽[T]
D1093.04 BOOL  ; $?St$Bk?_#[362] / 5St_B出料定位B"$?St$Bk?_#[362]
D1093.06 BOOL  ; $?St$Bk?_#[364] / 5St_B出料定位B"$?St$Bk?_#[364]
D1093.08 BOOL  ; $?St$Bk?_#[366] / 5St_B出料定位B"$?St$Bk?_#[366]
D1093.10 BOOL  ; $?St$Bk?_#[368] / 5St_B出料定位B"$?St$Bk?_#[368]
D1093.12 BOOL  ; $?St$Bk?_#[370] / 5St_B出料定位B"$?St$Bk?_#[370]
D1093.14 BOOL  ; $?St$Bk?_#[372] / 5St_B出料定位B"$?St$Bk?_#[372]
D1094.00 BOOL  ; 5St_B出料定位B上游就绪-0
D1094.01 BOOL  ; 5St_B出料定位B使能上游-0
D1094.02 BOOL  ; 5St_B出料定位B上游就绪-1
D1094.03 BOOL  ; 5St_B出料定位B使能上游-1
D1094.04 BOOL  ; 5St_B出料定位B上游就绪-2
D1094.05 BOOL  ; 5St_B出料定位B使能上游-2
D1094.06 BOOL  ; 5St_B出料定位B上游就绪-3
D1094.07 BOOL  ; 5St_B出料定位B使能上游-3
D1094.08 BOOL  ; 5St_B出料定位B下游就绪-0
D1094.09 BOOL  ; 5St_B出料定位B使能下游-0
D1094.10 BOOL  ; 5St_B出料定位B下游就绪-1
D1094.11 BOOL  ; 5St_B出料定位B使能下游-1
D1094.12 BOOL  ; 5St_B出料定位B下游就绪-2
D1094.13 BOOL  ; 5St_B出料定位B使能下游-2
D1094.14 BOOL  ; 5St_B出料定位B下游就绪-3
D1094.15 BOOL  ; 5St_B出料定位B使能下游-3
D1095.00 BOOL  ; 5St_B出料定位B递进启动
D1095.01 BOOL  ; 5St_B出料定位B步01
D1095.02 BOOL  ; 5St_B出料定位B步02
D1095.03 BOOL  ; 5St_B出料定位B步03
D1095.04 BOOL  ; 5St_B出料定位B步04
D1095.05 BOOL  ; 5St_B出料定位B步05
D1095.06 BOOL  ; 5St_B出料定位B步06
D1095.07 BOOL  ; 5St_B出料定位B步07
D1095.08 BOOL  ; 5St_B出料定位B步08
D1095.09 BOOL  ; 5St_B出料定位B步09
D1095.10 BOOL  ; 5St_B出料定位B步10
D1095.11 BOOL  ; 5St_B出料定位B步11
D1095.12 BOOL  ; 5St_B出料定位B步12
D1095.13 BOOL  ; 5St_B出料定位B步13
D1095.14 BOOL  ; 5St_B出料定位B步14
D1095.15 BOOL  ; 5St_B出料定位B步15
D1096.00 BOOL  ; 5St_B出料定位B步16
D1096.01 BOOL  ; 5St_B出料定位B步17
D1096.02 BOOL  ; 5St_B出料定位B步18
D1096.03 BOOL  ; 5St_B出料定位B步19
D1096.04 BOOL  ; 5St_B出料定位B步20
D1096.05 BOOL  ; 5St_B出料定位B步21
D1096.06 BOOL  ; 5St_B出料定位B步22
D1096.07 BOOL  ; 5St_B出料定位B步23
D1096.08 BOOL  ; 5St_B出料定位B步24
D1096.09 BOOL  ; 5St_B出料定位B步25
D1096.10 BOOL  ; 5St_B出料定位B步26
D1096.11 BOOL  ; 5St_B出料定位B步27
D1096.12 BOOL  ; 5St_B出料定位B步28
D1096.13 BOOL  ; 5St_B出料定位B步29
D1096.14 BOOL  ; 5St_B出料定位B步30
D1096.15 BOOL  ; 5St_B出料定位B步31
D1097.00 BOOL  ; 5St_B出料定位B初始化步号
D1097.01 BOOL  ; 5St_B出料定位B
D1097.02 BOOL  ; 5St_B出料定位B
D1097.03 BOOL  ; 5St_B出料定位B
D1097.04 BOOL  ; 5St_B出料定位B
D1097.05 BOOL  ; 5St_B出料定位B
D1097.06 BOOL  ; 5St_B出料定位B
D1097.07 BOOL  ; 5St_B出料定位B
D1097.08 BOOL  ; 5St_B出料定位B
D1097.09 BOOL  ; 5St_B出料定位B
D1097.10 BOOL  ; 5St_B出料定位B
D1097.11 BOOL  ; 5St_B出料定位B
D1097.12 BOOL  ; 5St_B出料定位B
D1097.13 BOOL  ; 5St_B出料定位B
D1097.14 BOOL  ; 5St_B出料定位B
D1097.15 BOOL  ; 5St_B出料定位B
D1098.00 BOOL  ; 5St_B出料定位B初始化_1
D1098.01 BOOL  ; 5St_B出料定位B初始化_2
D1098.02 BOOL  ; 5St_B出料定位B初始化_3
D1098.03 BOOL  ; 5St_B出料定位B初始化_4
D1098.04 BOOL  ; 5St_B出料定位B初始化_5
D1098.05 BOOL  ; 5St_B出料定位B初始化_6
D1098.06 BOOL  ; 5St_B出料定位B初始化_7
D1098.07 BOOL  ; 5St_B出料定位B初始化_8
D1098.08 BOOL  ; 5St_B出料定位B初始化_9
D1098.09 BOOL  ; 5St_B出料定位B初始化_10
D1098.10 BOOL  ; 5St_B出料定位B初始化_11
D1098.11 BOOL  ; 5St_B出料定位B初始化_12
D1098.12 BOOL  ; 5St_B出料定位B初始化_13
D1098.13 BOOL  ; 5St_B出料定位B初始化_14
D1098.14 BOOL  ; 5St_B出料定位B初始化_15
D1098.15 BOOL  ; 5St_B出料定位B初始化_16
D1099.00 BOOL  ; 5St_B出料定位B初始化_17
D1099.01 BOOL  ; 5St_B出料定位B初始化_18
D1099.02 BOOL  ; 5St_B出料定位B初始化_19
D1099.03 BOOL  ; 5St_B出料定位B初始化_20
D1099.04 BOOL  ; 5St_B出料定位B初始化_21
D1099.05 BOOL  ; 5St_B出料定位B初始化_22
D1099.06 BOOL  ; 5St_B出料定位B初始化_23
D1099.07 BOOL  ; 5St_B出料定位B初始化_24
D1099.08 BOOL  ; 5St_B出料定位B初始化_25
D1099.09 BOOL  ; 5St_B出料定位B初始化_26
D1099.10 BOOL  ; 5St_B出料定位B初始化_27
D1099.11 BOOL  ; 5St_B出料定位B初始化_28
D1099.12 BOOL  ; 5St_B出料定位B初始化_29
D1099.13 BOOL  ; 5St_B出料定位B初始化_30
D1099.14 BOOL  ; 5St_B出料定位B初始化_31
D1099.15 BOOL  ; 5St_B出料定位B初始化_32
D1100.00 BOOL  ; 6St下料机器人工站错误
D1100.01 BOOL  ; 6St下料机器人工站警告
D1100.02 BOOL  ; 6St下料机器人工站运行
D1100.03 BOOL  ; $?St$Bk?_#[374] / 6St下料机器人"$?St$Bk?_#[374]
D1100.05 BOOL  ; $?St$Bk?_#[376] / 6St下料机器人"$?St$Bk?_#[376]
D1100.07 BOOL  ; $?St$Bk?_#[378] / 6St下料机器人"$?St$Bk?_#[378]
D1100.09 BOOL  ; $?St$Bk?_#[380] / 6St下料机器人"$?St$Bk?_#[380]
D1100.11 BOOL  ; $?St$Bk?_#[382] / 6St下料机器人"$?St$Bk?_#[382]
D1100.13 BOOL  ; $?St$Bk?_#[384] / 6St下料机器人"$?St$Bk?_#[384]
D1100.15 BOOL  ; $?St$Bk?_#[386] / 6St下料机器人"$?St$Bk?_#[386]
D1101.04 BOOL  ; $?St$Bk?_#[388] / 6St下料机器人"$?St$Bk?_#[388]
D1101.06 BOOL  ; $?St$Bk?_#[390] / 6St下料机器人"$?St$Bk?_#[390]
D1101.08 BOOL  ; $?St$Bk?_#[392] / 6St下料机器人"$?St$Bk?_#[392]
D1101.10 BOOL  ; $?St$Bk?_#[394] / 6St下料机器人"$?St$Bk?_#[394]
D1101.12 BOOL  ; $?St$Bk?_#[396] / 6St下料机器人"$?St$Bk?_#[396]
D1101.14 BOOL  ; $?St$Bk?_#[398] / 6St下料机器人"$?St$Bk?_#[398]
D1102.00 BOOL  ; 6St下料机器人工站就绪
D1102.01 BOOL  ; 6St下料机器人 初始化中
D1102.02 BOOL  ; 6St下料机器人 自动停止中
D1102.03 BOOL  ; 6St下料机器人 自动停止完成
D1102.04 BOOL  ; 6St下料机器人 联锁
D1102.05 BOOL  ; 6St下料机器人 单步中
D1102.06 BOOL  ; 6St下料机器人 单周期中
D1102.07 BOOL  ; 6St下料机器人 周期完成
D1102.08 BOOL  ; 6St下料机器人 任务开始
D1102.09 BOOL  ; 6St下料机器人 任务递进条件
D1102.10 BOOL  ; 6St下料机器人 任务递进
D1102.11 BOOL  ; 6St下料机器人 工作完成
D1102.12 BOOL  ; 6St下料机器人 初始化[T]
D1102.13 BOOL  ; 6St下料机器人 单步[T]
D1102.14 BOOL  ; 6St下料机器人 单周期[T]
D1102.15 BOOL  ; 6St下料机器人 任务停止[T]
D1103.00 BOOL  ; 6St下料机器人 工站完成置位[T]
D1103.01 BOOL  ; 6St下料机器人 工站完成复位[T]
D1103.02 BOOL  ; 6St下料机器人 数据清除[T]
D1103.03 BOOL  ; 6St下料机器人 工站屏蔽[T]
D1103.04 BOOL  ; $?St$Bk?_#[400] / 6St下料机器人"$?St$Bk?_#[400]
D1103.06 BOOL  ; $?St$Bk?_#[402] / 6St下料机器人"$?St$Bk?_#[402]
D1103.08 BOOL  ; $?St$Bk?_#[404] / 6St下料机器人"$?St$Bk?_#[404]
D1103.10 BOOL  ; $?St$Bk?_#[406] / 6St下料机器人"$?St$Bk?_#[406]
D1103.12 BOOL  ; $?St$Bk?_#[408] / 6St下料机器人"$?St$Bk?_#[408]
D1103.14 BOOL  ; $?St$Bk?_#[410] / 6St下料机器人"$?St$Bk?_#[410]
D1104.00 BOOL  ; 6St下料机器人上游就绪-0
D1104.01 BOOL  ; 6St下料机器人使能上游-0
D1104.02 BOOL  ; 6St下料机器人上游就绪-1
D1104.03 BOOL  ; 6St下料机器人使能上游-1
D1104.04 BOOL  ; 6St下料机器人上游就绪-2
D1104.05 BOOL  ; 6St下料机器人使能上游-2
D1104.06 BOOL  ; 6St下料机器人上游就绪-3
D1104.07 BOOL  ; 6St下料机器人使能上游-3
D1104.08 BOOL  ; 6St下料机器人下游就绪-0
D1104.09 BOOL  ; 6St下料机器人使能下游-0
D1104.10 BOOL  ; 6St下料机器人下游就绪-1
D1104.11 BOOL  ; 6St下料机器人使能下游-1
D1104.12 BOOL  ; 6St下料机器人下游就绪-2
D1104.13 BOOL  ; 6St下料机器人使能下游-2
D1104.14 BOOL  ; 6St下料机器人下游就绪-3
D1104.15 BOOL  ; 6St下料机器人使能下游-3
D1105 CHANNEL  ; 1ST自动步存放字
D1105.00 BOOL  ; 6St下料机器人开始步
D1105.01 BOOL  ; 6St下料机器人去抓料上位
D1105.02 BOOL  ; 6St下料机器人去抓料位
D1105.03 BOOL  ; 6St下料机器人全部夹紧
D1105.04 BOOL  ; 6St下料机器人全部压紧
D1105.05 BOOL  ; 6St下料机器人判断跳转步
D1105.06 BOOL  ; 6St下料机器人去工艺NG位安全条件
D1105.07 BOOL  ; 6St下料机器人去工艺NG位
D1105.08 BOOL  ; 6St下料机器人放工艺NG物料及判断步
D1105.09 BOOL  ; 6St下料机器人去HipotNG上位
D1105.10 BOOL  ; 6St下料机器人去HipotNG位安全条件
D1105.11 BOOL  ; 6St下料机器人去HipotNG位安全条件
D1105.12 BOOL  ; 6St下料机器人放HipotNG物料及判断步
D1105.13 BOOL  ; 6St下料机器人去放料上位
D1105.14 BOOL  ; 6St下料机器人拉带可放料
D1105.15 BOOL  ; 6St下料机器人去放料位
D1106.00 BOOL  ; 6St下料机器人全部松压
D1106.01 BOOL  ; 6St下料机器人全部松夹
D1106.02 BOOL  ; 6St下料机器人去放料上位
D1106.03 BOOL  ; 6St下料机器人结束步
D1106.04 BOOL  ; 6St下料机器人步20
D1106.05 BOOL  ; 6St下料机器人步21
D1106.06 BOOL  ; 6St下料机器人步22
D1106.07 BOOL  ; 6St下料机器人步23
D1106.08 BOOL  ; 6St下料机器人步24
D1106.09 BOOL  ; 6St下料机器人步25
D1106.10 BOOL  ; 6St下料机器人步26
D1106.11 BOOL  ; 6St下料机器人步27
D1106.12 BOOL  ; 6St下料机器人步28
D1106.13 BOOL  ; 6St下料机器人步29
D1106.14 BOOL  ; 6St下料机器人步30
D1106.15 BOOL  ; 6St下料机器人步31
D1107.00 BOOL  ; 6St下料机器人初始化步号
D1107.01 BOOL  ; 6St下料机器人
D1107.02 BOOL  ; 6St下料机器人
D1107.03 BOOL  ; 6St下料机器人
D1107.04 BOOL  ; 6St下料机器人
D1107.05 BOOL  ; 6St下料机器人
D1107.06 BOOL  ; 6St下料机器人
D1107.07 BOOL  ; 6St下料机器人
D1107.08 BOOL  ; 6St下料机器人
D1107.09 BOOL  ; 6St下料机器人
D1107.10 BOOL  ; 6St下料机器人
D1107.11 BOOL  ; 6St下料机器人
D1107.12 BOOL  ; 6St下料机器人
D1107.13 BOOL  ; 6St下料机器人
D1107.14 BOOL  ; 6St下料机器人
D1107.15 BOOL  ; 6St下料机器人
D1108.00 BOOL  ; 6St下料机器人初始化_1
D1108.01 BOOL  ; 6St下料机器人初始化_2
D1108.02 BOOL  ; 6St下料机器人初始化_3
D1108.03 BOOL  ; 6St下料机器人初始化_4
D1108.04 BOOL  ; 6St下料机器人初始化_5
D1108.05 BOOL  ; 6St下料机器人初始化_6
D1108.06 BOOL  ; 6St下料机器人初始化_7
D1108.07 BOOL  ; 6St下料机器人初始化_8
D1108.08 BOOL  ; 6St下料机器人初始化_9
D1108.09 BOOL  ; 6St下料机器人初始化_10
D1108.10 BOOL  ; 6St下料机器人初始化_11
D1108.11 BOOL  ; 6St下料机器人初始化_12
D1108.12 BOOL  ; 6St下料机器人初始化_13
D1108.13 BOOL  ; 6St下料机器人初始化_14
D1108.14 BOOL  ; 6St下料机器人初始化_15
D1108.15 BOOL  ; 6St下料机器人初始化_16
D1109.00 BOOL  ; 6St下料机器人初始化_17
D1109.01 BOOL  ; 6St下料机器人初始化_18
D1109.02 BOOL  ; 6St下料机器人初始化_19
D1109.03 BOOL  ; 6St下料机器人初始化_20
D1109.04 BOOL  ; 6St下料机器人初始化_21
D1109.05 BOOL  ; 6St下料机器人初始化_22
D1109.06 BOOL  ; 6St下料机器人初始化_23
D1109.07 BOOL  ; 6St下料机器人初始化_24
D1109.08 BOOL  ; 6St下料机器人初始化_25
D1109.09 BOOL  ; 6St下料机器人初始化_26
D1109.10 BOOL  ; 6St下料机器人初始化_27
D1109.11 BOOL  ; 6St下料机器人初始化_28
D1109.12 BOOL  ; 6St下料机器人初始化_29
D1109.13 BOOL  ; 6St下料机器人初始化_30
D1109.14 BOOL  ; 6St下料机器人初始化_31
D1109.15 BOOL  ; 6St下料机器人初始化_32
D1110.00 BOOL  ; 7St接料及扫码工站错误
D1110.01 BOOL  ; 7St接料及扫码工站警告
D1110.02 BOOL  ; 7St接料及扫码工站运行
D1110.03 BOOL  ; $?St$Bk?_#[412] / 7St接料及扫码"$?St$Bk?_#[412]
D1110.05 BOOL  ; $?St$Bk?_#[414] / 7St接料及扫码"$?St$Bk?_#[414]
D1110.07 BOOL  ; $?St$Bk?_#[416] / 7St接料及扫码"$?St$Bk?_#[416]
D1110.09 BOOL  ; $?St$Bk?_#[418] / 7St接料及扫码"$?St$Bk?_#[418]
D1110.11 BOOL  ; $?St$Bk?_#[420] / 7St接料及扫码"$?St$Bk?_#[420]
D1110.13 BOOL  ; $?St$Bk?_#[422] / 7St接料及扫码"$?St$Bk?_#[422]
D1110.15 BOOL  ; $?St$Bk?_#[424] / 7St接料及扫码"$?St$Bk?_#[424]
D1111.04 BOOL  ; $?St$Bk?_#[426] / 7St接料及扫码"$?St$Bk?_#[426]
D1111.06 BOOL  ; $?St$Bk?_#[428] / 7St接料及扫码"$?St$Bk?_#[428]
D1111.08 BOOL  ; $?St$Bk?_#[430] / 7St接料及扫码"$?St$Bk?_#[430]
D1111.10 BOOL  ; $?St$Bk?_#[432] / 7St接料及扫码"$?St$Bk?_#[432]
D1111.12 BOOL  ; $?St$Bk?_#[434] / 7St接料及扫码"$?St$Bk?_#[434]
D1111.14 BOOL  ; $?St$Bk?_#[436] / 7St接料及扫码"$?St$Bk?_#[436]
D1112.00 BOOL  ; 7St接料及扫码工站就绪
D1112.01 BOOL  ; 7St接料及扫码 初始化中
D1112.02 BOOL  ; 7St接料及扫码 自动停止中
D1112.03 BOOL  ; 7St接料及扫码 自动停止完成
D1112.04 BOOL  ; 7St接料及扫码 联锁
D1112.05 BOOL  ; 7St接料及扫码 单步中
D1112.06 BOOL  ; 7St接料及扫码 单周期中
D1112.07 BOOL  ; 7St接料及扫码 周期完成
D1112.08 BOOL  ; 7St接料及扫码 任务开始
D1112.09 BOOL  ; 7St接料及扫码 任务递进条件
D1112.10 BOOL  ; 7St接料及扫码 任务递进
D1112.11 BOOL  ; 7St接料及扫码 工作完成
D1112.12 BOOL  ; 7St接料及扫码 初始化[T]
D1112.13 BOOL  ; 7St接料及扫码 单步[T]
D1112.14 BOOL  ; 7St接料及扫码 单周期[T]
D1112.15 BOOL  ; 7St接料及扫码 任务停止[T]
D1113.00 BOOL  ; 7St接料及扫码 工站完成置位[T]
D1113.01 BOOL  ; 7St接料及扫码 工站完成复位[T]
D1113.02 BOOL  ; 7St接料及扫码 数据清除[T]
D1113.03 BOOL  ; 7St接料及扫码 工站屏蔽[T]
D1113.04 BOOL  ; $?St$Bk?_#[438] / 7St接料及扫码"$?St$Bk?_#[438]
D1113.06 BOOL  ; $?St$Bk?_#[440] / 7St接料及扫码"$?St$Bk?_#[440]
D1113.08 BOOL  ; $?St$Bk?_#[442] / 7St接料及扫码"$?St$Bk?_#[442]
D1113.10 BOOL  ; $?St$Bk?_#[444] / 7St接料及扫码"$?St$Bk?_#[444]
D1113.12 BOOL  ; $?St$Bk?_#[446] / 7St接料及扫码"$?St$Bk?_#[446]
D1113.14 BOOL  ; $?St$Bk?_#[448] / 7St接料及扫码"$?St$Bk?_#[448]
D1114.00 BOOL  ; 7St接料及扫码上游就绪-0
D1114.01 BOOL  ; 7St接料及扫码使能上游-0
D1114.02 BOOL  ; 7St接料及扫码上游就绪-1
D1114.03 BOOL  ; 7St接料及扫码使能上游-1
D1114.04 BOOL  ; 7St接料及扫码上游就绪-2
D1114.05 BOOL  ; 7St接料及扫码使能上游-2
D1114.06 BOOL  ; 7St接料及扫码上游就绪-3
D1114.07 BOOL  ; 7St接料及扫码使能上游-3
D1114.08 BOOL  ; 7St接料及扫码下游就绪-0
D1114.09 BOOL  ; 7St接料及扫码使能下游-0
D1114.10 BOOL  ; 7St接料及扫码下游就绪-1
D1114.11 BOOL  ; 7St接料及扫码使能下游-1
D1114.12 BOOL  ; 7St接料及扫码下游就绪-2
D1114.13 BOOL  ; 7St接料及扫码使能下游-2
D1114.14 BOOL  ; 7St接料及扫码下游就绪-3
D1114.15 BOOL  ; 7St接料及扫码使能下游-3
D1115.00 BOOL  ; 7St扫码开始步
D1115.01 BOOL  ; 扫码判断步
D1115.02 BOOL  ; A1扫码未完成
D1115.03 BOOL  ; 一层扫码左位
D1115.04 BOOL  ; 一层扫码前进
D1115.05 BOOL  ; 一层A1开始扫码
D1115.06 BOOL  ; 一层A1扫码完成
D1115.07 BOOL  ; 一层扫码后退
D1115.08 BOOL  ; B1扫码未完成
D1115.09 BOOL  ; 一层扫码右位
D1115.10 BOOL  ; 一层扫码前进
D1115.11 BOOL  ; 一层B1开始扫码
D1115.12 BOOL  ; 一层B1扫码完成
D1115.13 BOOL  ; 一层扫码后退
D1115.14 BOOL  ; A2扫码未完成
D1115.15 BOOL  ; 二层扫码左位
D1116.00 BOOL  ; 二层扫码前进
D1116.01 BOOL  ; 二层A2开始扫码
D1116.02 BOOL  ; 二层A2扫码完成
D1116.03 BOOL  ; 二层扫码后退
D1116.04 BOOL  ; B2扫码未完成
D1116.05 BOOL  ; 二层扫码左位
D1116.06 BOOL  ; 二层扫码前进
D1116.07 BOOL  ; 二层B2开始扫码
D1116.08 BOOL  ; 二层B2扫码完成
D1116.09 BOOL  ; 二层扫码后退
D1116.10 BOOL  ; 7St扫码结束步
D1116.11 BOOL  ; 7St接料及扫码步27
D1116.12 BOOL  ; 7St接料及扫码步28
D1116.13 BOOL  ; 7St接料及扫码步29
D1116.14 BOOL  ; 7St接料及扫码步30
D1116.15 BOOL  ; 7St接料及扫码步31
D1117.00 BOOL  ; 7St接料及扫码初始化步号
D1117.01 BOOL  ; 7St接料及扫码
D1117.02 BOOL  ; 7St接料及扫码
D1117.03 BOOL  ; 7St接料及扫码
D1117.04 BOOL  ; 7St接料及扫码
D1117.05 BOOL  ; 7St接料及扫码
D1117.06 BOOL  ; 7St接料及扫码
D1117.07 BOOL  ; 7St接料及扫码
D1117.08 BOOL  ; 7St接料及扫码
D1117.09 BOOL  ; 7St接料及扫码
D1117.10 BOOL  ; 7St接料及扫码
D1117.11 BOOL  ; 7St接料及扫码
D1117.12 BOOL  ; 7St接料及扫码
D1117.13 BOOL  ; 7St接料及扫码
D1117.14 BOOL  ; 7St接料及扫码
D1117.15 BOOL  ; 7St接料及扫码
D1118.00 BOOL  ; 7St接料及扫码初始化_1
D1118.01 BOOL  ; 7St接料及扫码初始化_2
D1118.02 BOOL  ; 7St接料及扫码初始化_3
D1118.03 BOOL  ; 7St接料及扫码初始化_4
D1118.04 BOOL  ; 7St接料及扫码初始化_5
D1118.05 BOOL  ; 7St接料及扫码初始化_6
D1118.06 BOOL  ; 7St接料及扫码初始化_7
D1118.07 BOOL  ; 7St接料及扫码初始化_8
D1118.08 BOOL  ; 7St接料及扫码初始化_9
D1118.09 BOOL  ; 7St接料及扫码初始化_10
D1118.10 BOOL  ; 7St接料及扫码初始化_11
D1118.11 BOOL  ; 7St接料及扫码初始化_12
D1118.12 BOOL  ; 7St接料及扫码初始化_13
D1118.13 BOOL  ; 7St接料及扫码初始化_14
D1118.14 BOOL  ; 7St接料及扫码初始化_15
D1118.15 BOOL  ; 7St接料及扫码初始化_16
D1119.00 BOOL  ; 7St接料及扫码初始化_17
D1119.01 BOOL  ; 7St接料及扫码初始化_18
D1119.02 BOOL  ; 7St接料及扫码初始化_19
D1119.03 BOOL  ; 7St接料及扫码初始化_20
D1119.04 BOOL  ; 7St接料及扫码初始化_21
D1119.05 BOOL  ; 7St接料及扫码初始化_22
D1119.06 BOOL  ; 7St接料及扫码初始化_23
D1119.07 BOOL  ; 7St接料及扫码初始化_24
D1119.08 BOOL  ; 7St接料及扫码初始化_25
D1119.09 BOOL  ; 7St接料及扫码初始化_26
D1119.10 BOOL  ; 7St接料及扫码初始化_27
D1119.11 BOOL  ; 7St接料及扫码初始化_28
D1119.12 BOOL  ; 7St接料及扫码初始化_29
D1119.13 BOOL  ; 7St接料及扫码初始化_30
D1119.14 BOOL  ; 7St接料及扫码初始化_31
D1119.15 BOOL  ; 7St接料及扫码初始化_32
D114.13 BOOL  ; 100-1St_电芯进料 回待机位
D12600 CHANNEL  ; ST5520_A 测试电压读取返回数据(ASC)
D12601 CHANNEL  ; ST5520_A 测试电压读取值(ASC)
D12620 CHANNEL  ; ST5520_A1 绝缘测试仪测试写入时间读取值(ASC)
D12640 CHANNEL  ; ST5520_A 绝缘测试仪延时时间读取返回数据(ASC)
D12641 CHANNEL  ; ST5520_A 绝缘测试仪延时时间读取值(ASC)
D12660 CHANNEL  ; ST5520_A 读取绝缘电阻上下限返回值
D12700 CHANNEL  ; ST5520_A 读取的测试档位返回数据
D12701 CHANNEL  ; ST5520_A 读取的测试档位返回数据
D12720 CHANNEL  ; ST5520_A 读取测试速度返回数据
D12721 CHANNEL  ; ST5520_A 读取测试速度返回数据(ASC)
D12740 CHANNEL  ; ST5520_A 读取比较器的测试模式数据
D12741 CHANNEL  ; ST5520_A 读取比较器的测试模式数据
D12800 CHANNEL  ; ST5520_A 读取绝缘电阻上限返回值
D12810 CHANNEL  ; ST5520_A 绝缘电阻上限读取值(欧)
D12820 CHANNEL  ; ST5520_A 绝缘电阻上限读取值(兆欧)
D12840 CHANNEL  ; ST5520_A 读取绝缘电阻下限返回值
D12850 CHANNEL  ; ST5520_A 绝缘电阻下限读取值(欧)
D12860 CHANNEL  ; ST5520_A 绝缘电阻下限读取值(兆欧)
D12900 CHANNEL  ; $?St$Bk?_#[449] / "PASS"$?St$Bk?_#[449]
D12910 CHANNEL  ; $?St$Bk?_#[450] / "LFAIL"$?St$Bk?_#[450]
D12920 CHANNEL  ; $?St$Bk?_#[451] / "UFAIL"$?St$Bk?_#[451]
D12930 CHANNEL  ; $?St$Bk?_#[452] / "ULFAIL"$?St$Bk?_#[452]
D12940 CHANNEL  ; $?St$Bk?_#[453] / "NOCOMP"$?St$Bk?_#[453]
D12950 CHANNEL  ; 空格
D12952 CHANNEL  ; 字符“O.F.”
D12960 CHANNEL  ; $?St$Bk?_#[454] / "O."$?St$Bk?_#[454]
D12961 CHANNEL  ; 'U.'
D12962 CHANNEL  ; 'C.'
D12963 CHANNEL  ; 'Sh'
D1400.00 BOOL  ; 初始位(15)到取料A1安全位(02)(HMI)
D1400.01 BOOL  ; 初始位(15)到取料A2安全位(03)(HMI)
D1400.02 BOOL  ; 初始位(15)到取料B1安全位(04)(HMI)
D1400.03 BOOL  ; 初始位(15)到取料B2安全位(05)(HMI)
D1400.04 BOOL  ; 取料A1安全位(01)到取料A1位(02)(HMI)
D1400.05 BOOL  ; 取料A2安全位(03)到取料A2位(04)(HMI)
D1400.06 BOOL  ; 取料B1安全位(05)到取料B1位(06)(HMI)
D1400.07 BOOL  ; 取料B2安全位(07)到取料B2位(08)(HMI)
D1400.08 BOOL  ; 取料A1位(02)到放料A安全位(11)(HMI)
D1400.09 BOOL  ; 取料A2位(04)到放料A安全位(11)(HMI)
D1400.10 BOOL  ; 取料B1位(06)到放料A安全位(11)(HMI)
D1400.11 BOOL  ; 取料B2位(08)到放料A安全位(11)(HMI)
D1400.12 BOOL  ; 取料A1位(02)到放料B安全位(13)(HMI)
D1400.13 BOOL  ; 取料A2位(04)到放料B安全位(13)(HMI)
D1400.14 BOOL  ; 取料B1位(06)到放料B安全位(13)(HMI)
D1400.15 BOOL  ; 取料B2位(08)到放料B安全位(13)(HMI)
D1401.00 BOOL  ; 放料A安全位(11)到放料A位(12)(HMI)
D1401.01 BOOL  ; 放料B安全位(13)到放料B位(14)(HMI)
D1401.02 BOOL  ; 放料A位(12)到初始位(15)(HMI)
D1401.03 BOOL  ; 放料B位(14)到初始位(15)(HMI)
D1401.04 BOOL  ; 取料A1位(02)到初始位(15)(HMI)
D1401.05 BOOL  ; 取料A2位(04)到初始位(15)(HMI)
D1401.06 BOOL  ; 取料B1位(06)到初始位(15)(HMI)
D1401.07 BOOL  ; 取料B2位(08)到初始位(15)(HMI)
D1401.08 BOOL  ; 扫码安全位(09)到扫码位(10)(HMI)
D1401.09 BOOL  ; 扫码位(10)到初始位(15)(HMI)
D1401.10 BOOL  ; 初始位(15)到扫码安全位(09)(HMI)
D1401.11 BOOL  ; 初始位(15)到放料A安全位(11)(HMI)
D1401.12 BOOL  ; 初始位(15)到放料B安全位(13)(HMI)
D1401.13 BOOL  ; 取料A1安全位(01)到初始位(15)(HMI)
D1401.14 BOOL  ; 取料A2安全位(03)到初始位(15)(HMI)
D1401.15 BOOL  ; 取料B1安全位(05)到初始位(15)(HMI)
D1402.00 BOOL  ; 取料B2安全位(07)到初始位(15)(HMI)
D1402.01 BOOL  ; 扫码安全位(09)到初始位(15)(HMI)
D1402.02 BOOL  ; 放料A安全位(11)到初始位(15)(HMI)
D1402.03 BOOL  ; 放料B安全位(13)到初始位(15)(HMI)
D1402.04 BOOL  ; 取料A1位(02)到取料A1安全位(01)(HMI)
D1402.05 BOOL  ; 取料A2位(04)到取料A2安全位(03)(HMI)
D1402.06 BOOL  ; 取料B1位(06)到取料B1安全位(05)(HMI)
D1402.07 BOOL  ; 取料B2位(08)到取料B2安全位(07)(HMI)
D1402.08 BOOL  ; 扫码位(10)到扫码安全位(09)(HMI)
D1402.09 BOOL  ; 放料A位(12)到放料A安全位(11)(HMI)
D1402.10 BOOL  ; 放料B位(14)到放料B安全位(13)(HMI)
D1402.11 BOOL  ; 扫码位(10)到放料A位(12)(HMI)
D1402.12 BOOL  ; 扫码位(10)到放料B位(14)(HMI)
D1402.13 BOOL  ; 初始位(15)到放料A位(12)(HMI)
D1402.14 BOOL  ; 初始位(15)到放料B位(14)(HMI）
D1403.00 BOOL  ; 初始位(15)到取料A1安全位(02)(M)
D1403.01 BOOL  ; 初始位(15)到取料A2安全位(03)(M)
D1403.02 BOOL  ; 初始位(15)到取料B1安全位(04)(M)
D1403.03 BOOL  ; 初始位(15)到取料B2安全位(05)(M)
D1403.04 BOOL  ; 取料A1安全位(01)到取料A1位(02)(M)
D1403.05 BOOL  ; 取料A2安全位(03)到取料A2位(04)(M)
D1403.06 BOOL  ; 取料B1安全位(05)到取料B1位(06)(M)
D1403.07 BOOL  ; 取料B2安全位(07)到取料B2位(08)(M)
D1403.08 BOOL  ; 取料A1位(02)到放料A安全位(11)(M)
D1403.09 BOOL  ; 取料A2位(04)到放料A安全位(11)(M)
D1403.10 BOOL  ; 取料B1位(06)到放料A安全位(11)(M)
D1403.11 BOOL  ; 取料B2位(08)到放料A安全位(11)(M)
D1403.12 BOOL  ; 取料A1位(02)到放料B安全位(13)(M)
D1403.13 BOOL  ; 取料A2位(04)到放料B安全位(13)(M)
D1403.14 BOOL  ; 取料B1位(06)到放料B安全位(13)(M)
D1403.15 BOOL  ; 取料B2位(08)到放料B安全位(13)(M)
D1404.00 BOOL  ; 放料A安全位(11)到放料A位(12)(M)
D1404.01 BOOL  ; 放料B安全位(13)到放料B位(14)(M)
D1404.02 BOOL  ; 放料A位(12)到初始位(15)(M)
D1404.03 BOOL  ; 放料B位(14)到初始位(15)(M)
D1404.04 BOOL  ; 取料A1位(02)到初始位(15)(M)
D1404.05 BOOL  ; 取料A2位(04)到初始位(15)(M)
D1404.06 BOOL  ; 取料B1位(06)到初始位(15)(M)
D1404.07 BOOL  ; 取料B2位(08)到初始位(15)(M)
D1404.08 BOOL  ; 扫码安全位(09)到扫码位(10)(M)
D1404.09 BOOL  ; 扫码位(10)到初始位(15)(M)
D1404.10 BOOL  ; 初始位(15)到扫码安全位(09)(M)
D1404.11 BOOL  ; 初始位(15)到放料A安全位(11)(M)
D1404.12 BOOL  ; 初始位(15)到放料B安全位(13)(M)
D1404.13 BOOL  ; 取料A1安全位(01)到初始位(15)(M)
D1404.14 BOOL  ; 取料A2安全位(03)到初始位(15)(M)
D1404.15 BOOL  ; 取料B1安全位(05)到初始位(15)(M)
D1405.00 BOOL  ; 取料B2安全位(07)到初始位(15)(M)
D1405.01 BOOL  ; 扫码安全位(09)到初始位(15)(M)
D1405.02 BOOL  ; 放料A安全位(11)到初始位(15)(M)
D1405.03 BOOL  ; 放料B安全位(13)到初始位(15)(M)
D1405.04 BOOL  ; 取料A1位(02)到取料A1安全位(01)(M)
D1405.05 BOOL  ; 取料A2位(04)到取料A2安全位(03)(M)
D1405.06 BOOL  ; 取料B1位(06)到取料B1安全位(05)(M)
D1405.07 BOOL  ; 取料B2位(08)到取料B2安全位(07)(M)
D1405.08 BOOL  ; 扫码位(10)到扫码安全位(09)(M)
D1405.09 BOOL  ; 放料A位(12)到放料A安全位(11)(M)
D1405.10 BOOL  ; 放料B位(14)到放料B安全位(13)(M)
D1405.11 BOOL  ; 扫码位(10)到放料A位(12)(M)
D1405.12 BOOL  ; 扫码位(10)到放料B位(14)(M)
D1405.13 BOOL  ; 初始位(15)到放料A位(12)(M)
D1405.14 BOOL  ; 初始位(15)到放料B位(14)(M）
D1406.00 BOOL  ; 初始位(15)到取料A1安全位(02)(A)
D1406.01 BOOL  ; 初始位(15)到取料A2安全位(03)(A)
D1406.02 BOOL  ; 初始位(15)到取料B1安全位(04)(A)
D1406.03 BOOL  ; 初始位(15)到取料B2安全位(05)(A)
D1406.04 BOOL  ; 取料A1安全位(01)到取料A1位(02)(A)
D1406.05 BOOL  ; 取料A2安全位(03)到取料A2位(04)(A)
D1406.06 BOOL  ; 取料B1安全位(05)到取料B1位(06)(A)
D1406.07 BOOL  ; 取料B2安全位(07)到取料B2位(08)(A)
D1406.08 BOOL  ; 取料A1位(02)到放料A安全位(11)(A)
D1406.09 BOOL  ; 取料A2位(04)到放料A安全位(11)(A)
D1406.10 BOOL  ; 取料B1位(06)到放料A安全位(11)(A)
D1406.11 BOOL  ; 取料B2位(08)到放料A安全位(11)(A)
D1406.12 BOOL  ; 取料A1位(02)到放料B安全位(13)(A)
D1406.13 BOOL  ; 取料A2位(04)到放料B安全位(13)(A)
D1406.14 BOOL  ; 取料B1位(06)到放料B安全位(13)(A)
D1406.15 BOOL  ; 取料B2位(08)到放料B安全位(13)(A)
D1407.00 BOOL  ; 放料A安全位(11)到放料A位(12)(A)
D1407.01 BOOL  ; 放料B安全位(13)到放料B位(14)(A)
D1407.02 BOOL  ; 放料A位(12)到初始位(15)(A)
D1407.03 BOOL  ; 放料B位(14)到初始位(15)(A)
D1407.04 BOOL  ; 取料A1位(02)到初始位(15)(A)
D1407.05 BOOL  ; 取料A2位(04)到初始位(15)(A)
D1407.06 BOOL  ; 取料B1位(06)到初始位(15)(A)
D1407.07 BOOL  ; 取料B2位(08)到初始位(15)(A)
D1407.08 BOOL  ; 扫码安全位(09)到扫码位(10)(A)
D1407.09 BOOL  ; 扫码位(10)到初始位(15)(A)
D1407.10 BOOL  ; 初始位(15)到扫码安全位(09)(A)
D1407.11 BOOL  ; 初始位(15)到放料A安全位(11)(A)
D1407.12 BOOL  ; 初始位(15)到放料B安全位(13)(A)
D1407.13 BOOL  ; 取料A1安全位(01)到初始位(15)(A)
D1407.14 BOOL  ; 取料A2安全位(03)到初始位(15)(A)
D1407.15 BOOL  ; 取料B1安全位(05)到初始位(15)(A)
D1408.00 BOOL  ; 取料B2安全位(07)到初始位(15)(A)
D1408.01 BOOL  ; 扫码安全位(09)到初始位(15)(A)
D1408.02 BOOL  ; 放料A安全位(11)到初始位(15)(A)
D1408.03 BOOL  ; 放料B安全位(13)到初始位(15)(A)
D1408.04 BOOL  ; 取料A1位(02)到取料A1安全位(01)(A)
D1408.05 BOOL  ; 取料A2位(04)到取料A2安全位(03)(A)
D1408.06 BOOL  ; 取料B1位(06)到取料B1安全位(05)(A)
D1408.07 BOOL  ; 取料B2位(08)到取料B2安全位(07)(A)
D1408.08 BOOL  ; 扫码位(10)到扫码安全位(09)(A)
D1408.09 BOOL  ; 放料A位(12)到放料A安全位(11)(A)
D1408.10 BOOL  ; 放料B位(14)到放料B安全位(13)(A)
D1408.11 BOOL  ; 扫码位(10)到放料A位(12)(A)
D1408.12 BOOL  ; 扫码位(10)到放料B位(14)(A)
D1408.13 BOOL  ; 初始位(15)到放料A位(12)(A)
D1408.14 BOOL  ; 初始位(15)到放料B位(14)(A）
D1409.00 BOOL  ; 初始位(15)到取料A1安全位(02)(中间输出)
D1409.01 BOOL  ; 初始位(15)到取料A2安全位(03)(中间输出)
D1409.02 BOOL  ; 初始位(15)到取料B1安全位(04)(中间输出)
D1409.03 BOOL  ; 初始位(15)到取料B2安全位(05)(中间输出)
D1409.04 BOOL  ; 取料A1安全位(01)到取料A1位(02)(中间输出)
D1409.05 BOOL  ; 取料A2安全位(03)到取料A2位(04)(中间输出)
D1409.06 BOOL  ; 取料B1安全位(05)到取料B1位(06)(中间输出)
D1409.07 BOOL  ; 取料B2安全位(07)到取料B2位(08)(中间输出)
D1409.08 BOOL  ; 取料A1位(02)到放料A安全位(11)(中间输出)
D1409.09 BOOL  ; 取料A2位(04)到放料A安全位(11)(中间输出)
D1409.10 BOOL  ; 取料B1位(06)到放料A安全位(11)(中间输出)
D1409.11 BOOL  ; 取料B2位(08)到放料A安全位(11)(中间输出)
D1409.12 BOOL  ; 取料A1位(02)到放料B安全位(13)(中间输出)
D1409.13 BOOL  ; 取料A2位(04)到放料B安全位(13)(中间输出)
D1409.14 BOOL  ; 取料B1位(06)到放料B安全位(13)(中间输出)
D1409.15 BOOL  ; 取料B2位(08)到放料B安全位(13)(中间输出)
D1410.00 BOOL  ; 放料A安全位(11)到放料A位(12)(中间输出)
D1410.01 BOOL  ; 放料B安全位(13)到放料B位(14)(中间输出)
D1410.02 BOOL  ; 放料A位(12)到初始位(15)(中间输出)
D1410.03 BOOL  ; 放料B位(14)到初始位(15)(中间输出)
D1410.04 BOOL  ; 取料A1位(02)到初始位(15)(中间输出)
D1410.05 BOOL  ; 取料A2位(04)到初始位(15)(中间输出)
D1410.06 BOOL  ; 取料B1位(06)到初始位(15)(中间输出)
D1410.07 BOOL  ; 取料B2位(08)到初始位(15)(中间输出)
D1410.08 BOOL  ; 扫码安全位(09)到扫码位(10)(中间输出)
D1410.09 BOOL  ; 扫码位(10)到初始位(15)(中间输出)
D1410.10 BOOL  ; 初始位(15)到扫码安全位(09)(中间输出)
D1410.11 BOOL  ; 初始位(15)到放料A安全位(11)(中间输出)
D1410.12 BOOL  ; 初始位(15)到放料B安全位(13)(中间输出)
D1410.13 BOOL  ; 取料A1安全位(01)到初始位(15)(中间输出)
D1410.14 BOOL  ; 取料A2安全位(03)到初始位(15)(中间输出)
D1410.15 BOOL  ; 取料B1安全位(05)到初始位(15)(中间输出)
D1411.00 BOOL  ; 取料B2安全位(07)到初始位(15)(中间输出)
D1411.01 BOOL  ; 扫码安全位(09)到初始位(15)(中间输出)
D1411.02 BOOL  ; 放料A安全位(11)到初始位(15)(中间输出)
D1411.03 BOOL  ; 放料B安全位(13)到初始位(15)(中间输出)
D1411.04 BOOL  ; 取料A1位(02)到取料A1安全位(01)(中间输出)
D1411.05 BOOL  ; 取料A2位(04)到取料A2安全位(03)(中间输出)
D1411.06 BOOL  ; 取料B1位(06)到取料B1安全位(05)(中间输出)
D1411.07 BOOL  ; 取料B2位(08)到取料B2安全位(07)(中间输出)
D1411.08 BOOL  ; 扫码位(10)到扫码安全位(09)(中间输出)
D1411.09 BOOL  ; 放料A位(12)到放料A安全位(11)(中间输出)
D1411.10 BOOL  ; 放料B位(14)到放料B安全位(13)(中间输出)
D1411.11 BOOL  ; 放料A位(12)到放料A安全位(11)(中间输出)
D1411.12 BOOL  ; 放料B位(14)到放料B安全位(13)(中间输出)
D1411.13 BOOL  ; 初始位(15)到放料A位(12)(中间输出)
D1411.14 BOOL  ; 初始位(15)到放料B位(14)(中间输出）
D1412.00 BOOL  ; 速度切换-低速
D1412.01 BOOL  ; 速度切换-中低速
D1412.02 BOOL  ; 速度切换-中高速
D1412.03 BOOL  ; 速度切换-高速
D1412.05 BOOL  ; 初始化(HMI)
D1412.06 BOOL  ; 初始化(复位)
D1412.07 BOOL  ; 初始化中
D1412.08 BOOL  ; 初始化1：终止程序
D1412.09 BOOL  ; 初始化2：报警复位
D1412.10 BOOL  ; 初始化3：程序确认
D1412.11 BOOL  ; 初始化4：程序启动
D1413.00 BOOL  ; A1压板全部松起
D1413.01 BOOL  ; A1压板全部压紧
D1413.02 BOOL  ; A2压板全部松起
D1413.03 BOOL  ; A2压板全部压紧
D1413.04 BOOL  ; A3压板全部松起
D1413.05 BOOL  ; A3压板全部压紧
D1413.06 BOOL  ; A4压板全部松起
D1413.07 BOOL  ; A4压板全部压紧
D1413.08 BOOL  ; A5压板全部松起
D1413.09 BOOL  ; A5压板全部压紧
D1414.00 BOOL  ; A1全部松开
D1414.01 BOOL  ; A1全部夹紧
D1414.02 BOOL  ; A2全部松开
D1414.03 BOOL  ; A2全部夹紧
D1414.04 BOOL  ; A3全部松开
D1414.05 BOOL  ; A3全部夹紧
D1414.06 BOOL  ; A4全部松开
D1414.07 BOOL  ; A4全部夹紧
D1414.08 BOOL  ; A5全部松开
D1414.09 BOOL  ; A5全部夹紧
D1450 CHANNEL  ; 上料A吹气时间
D1500 CHANNEL  ; 上料B吹气时间
D1550 CHANNEL  ; A边无来料计时
D1551 CHANNEL  ; B边无来料计时
D1552 CHANNEL  ; 3ST_A A测取料允许计时
D1553 CHANNEL  ; 3ST_B A测取料允许计时
D1602 CHANNEL  ; 3ST_A B测取料允许计时
D1603 CHANNEL  ; 3ST_B B测取料允许计时
D1652 CHANNEL  ; 物料个数
D1654 CHANNEL  ; A工位无料层数
D1656 CHANNEL  ; A工位减速位补偿距离
D1662 CHANNEL  ; B工位热压电芯个数
D1664 CHANNEL  ; B工位无料个数
D1666 CHANNEL  ; B工位减速位补偿值
D1750 CHANNEL  ; 下料A吹气时间
D1760.00 BOOL  ; 数据传递至PC抓取区域
D1760.01 BOOL  ; PLC出站请求A
D1760.02 BOOL  ; 待PC与MES校验
D1760.03 BOOL  ; $?St$Bk?_#[455] / 接收MES出站校验 / $?St$Bk?_#[455]
D1760.04 BOOL  ; $?St$Bk?_#[456] / A记忆判断完成 / $?St$Bk?_#[456]
D1760.05 BOOL  ; $?St$Bk?_#[457] / B记忆判断完成 / $?St$Bk?_#[457]
D1760.06 BOOL  ; $?St$Bk?_#[458] / A面请求PC交互 / $?St$Bk?_#[458]
D1760.07 BOOL  ; $?St$Bk?_#[459] / A面PC交互完成 / $?St$Bk?_#[459]
D1760.08 BOOL  ; $?St$Bk?_#[460] / B面请求PC交互 / $?St$Bk?_#[460]
D1760.09 BOOL  ; $?St$Bk?_#[461] / B面PC交互完成 / $?St$Bk?_#[461]
D1800 CHANNEL  ; 下料B吹气时间
D1850.00 BOOL  ; 取料上位A(01)到取料位A(02)(HMI)
D1850.01 BOOL  ; 取料上位B(03)到取料位B(04)(HMI)
D1850.04 BOOL  ; 放料上位(05)到放料位(06)(HMI)
D1850.09 BOOL  ; 工艺NG上位(20)到工艺NG位(21)(HMI)
D1850.10 BOOL  ; HipotNG上位(30)到HipotNG位(31)(HMI)
D1851.03 BOOL  ; 任意上位到取料上位A(01)(HMI)
D1851.04 BOOL  ; 任意上位到取料上位B(03)(HMI)
D1851.05 BOOL  ; 任意上位到放料上位(05)(HMI)
D1851.06 BOOL  ; 任意上位到工艺NG上位(20)(HMI)
D1851.07 BOOL  ; 任意上位到HipotNG上位(30)(HMI)
D1851.08 BOOL  ; 取料位A(02)到取料上位A(01)(HMI)
D1851.09 BOOL  ; 取料位B(04)到取料上位B(03)(HMI)
D1851.10 BOOL  ; 放料位(06)到放料上位(05)(HMI)
D1851.11 BOOL  ; 工艺NG位(21)到工艺NG上位(20)(HMI)
D1851.12 BOOL  ; HipotNG位(31)到HipotNG上位(30)(HMI)
D1852.00 BOOL  ; 取料上位A(01)到取料位A(02)(M)
D1852.01 BOOL  ; 取料上位B(03)到取料位B(04)(M)
D1852.04 BOOL  ; 放料上位(05)到放料位(06)(M)
D1852.09 BOOL  ; 工艺NG上位(20)到工艺NG位(21)(M)
D1852.10 BOOL  ; HipotNG上位(30)到HipotNG位(31)(M)
D1853.03 BOOL  ; 任意上位到取料上位A(01)(M)
D1853.04 BOOL  ; 任意上位到取料上位B(03)(M)
D1853.05 BOOL  ; 任意上位到放料上位(05)(M)
D1853.06 BOOL  ; 任意上位到工艺NG上位(20)(M)
D1853.07 BOOL  ; 任意上位到HipotNG上位(30)(M)
D1853.08 BOOL  ; 取料位A(02)到取料上位A(01)(M)
D1853.09 BOOL  ; 取料位B(04)到取料上位B(03)(M)
D1853.10 BOOL  ; 放料位(06)到放料上位(05)(M)
D1853.11 BOOL  ; 工艺NG位(21)到工艺NG上位(20)(M)
D1853.12 BOOL  ; HipotNG位(31)到HipotNG上位(30)(M)
D1854.00 BOOL  ; 取料上位A(01)到取料位A(02)(A)
D1854.01 BOOL  ; 取料上位B(03)到取料位B(04)(A)
D1854.02 BOOL  ; 取料位A(02)到放料上位(05)(A)
D1854.03 BOOL  ; 取料位B(04)到放料上位(05)(A)
D1854.04 BOOL  ; 放料上位(05)到放料位(06)(A)
D1854.05 BOOL  ; 取料位A(02)到工艺NG上位(20)(A)
D1854.06 BOOL  ; 取料位B(04)到工艺NG上位(20)(A)
D1854.07 BOOL  ; 取料位A(02)到HipotNG上位(30)(A)
D1854.08 BOOL  ; 取料位B(04)到HipotNG上位(30)(A)
D1854.09 BOOL  ; 工艺NG上位(20)到工艺NG位(21)(A)
D1854.10 BOOL  ; HipotNG上位(30)到HipotNG位(31)(A)
D1854.11 BOOL  ; 工艺NG位(21)到取料上位A(01)(A)
D1854.12 BOOL  ; 工艺NG位(21)到取料上位B(03)(A)
D1854.13 BOOL  ; HipotNG位(31)到取料上位A(01)(A)
D1854.14 BOOL  ; HipotNG位(31)到取料上位B(03)(A)
D1854.15 BOOL  ; 工艺NG位(21)到HipotNG位(31)(A)
D1855.00 BOOL  ; HipotNG位(31)到工艺NG位(21)(A)
D1855.01 BOOL  ; 工艺NG位(21)到放料上位(05)(A)
D1855.02 BOOL  ; HipotNG位(31)到放料上位(05)(A)
D1855.03 BOOL  ; 任意上位到取料上位A(01)(A)
D1855.04 BOOL  ; 任意上位到取料上位B(03)(A)
D1855.05 BOOL  ; 任意上位到放料上位(05)(A)
D1855.06 BOOL  ; 任意上位到工艺NG上位(20)(A)
D1855.07 BOOL  ; 任意上位到HipotNG上位(30)(A)
D1855.08 BOOL  ; 取料位A(02)到取料上位A(01)(A)
D1855.09 BOOL  ; 取料位B(04)到取料上位B(03)(A)
D1855.10 BOOL  ; 放料位(06)到放料上位(05)(A)
D1855.11 BOOL  ; 工艺NG位(21)到工艺NG上位(20)(A)
D1855.12 BOOL  ; HipotNG位(31)到HipotNG上位(30)(A)
D1856.00 BOOL  ; 取料上位A(01)到取料位A(02)
D1856.01 BOOL  ; 取料上位B(03)到取料位B(04)
D1856.02 BOOL  ; 取料位A(02)到放料上位(05)
D1856.03 BOOL  ; 取料位B(04)到放料上位(05)
D1856.04 BOOL  ; 放料上位(05)到放料位(06)
D1856.05 BOOL  ; 取料位A(02)到工艺NG上位(20)
D1856.06 BOOL  ; 取料位B(04)到工艺NG上位(20)
D1856.07 BOOL  ; 取料位A(02)到HipotNG上位(30)
D1856.08 BOOL  ; 取料位B(04)到HipotNG上位(30)
D1856.09 BOOL  ; 工艺NG上位(20)到工艺NG位(21)
D1856.10 BOOL  ; HipotNG上位(30)到HipotNG位(31)
D1856.11 BOOL  ; 工艺NG位(21)到取料上位A(01)
D1856.12 BOOL  ; 工艺NG位(21)到取料上位B(03)
D1856.13 BOOL  ; HipotNG位(31)到取料上位A(01)
D1856.14 BOOL  ; HipotNG位(31)到取料上位B(03)
D1856.15 BOOL  ; 工艺NG位(21)到HipotNG位(31)
D1857.00 BOOL  ; HipotNG位(31)到工艺NG位(21)
D1857.01 BOOL  ; 工艺NG位(21)到放料上位(05)
D1857.02 BOOL  ; HipotNG位(31)到放料上位(05)
D1857.03 BOOL  ; 任意上位到取料上位A(01)
D1857.04 BOOL  ; 任意上位到取料上位B(03)
D1857.05 BOOL  ; 任意上位到放料上位(05)
D1857.06 BOOL  ; 任意上位到工艺NG上位(20)
D1857.07 BOOL  ; 任意上位到HipotNG上位(30)
D1857.08 BOOL  ; 取料位A(02)到取料上位A(01)
D1857.09 BOOL  ; 取料位B(04)到取料上位B(03)
D1857.10 BOOL  ; 放料位(06)到放料上位(05)
D1857.11 BOOL  ; 工艺NG位(21)到工艺NG上位(20)
D1857.12 BOOL  ; HipotNG位(31)到HipotNG上位(30)
D1863.00 BOOL  ; $?St$Bk?_#[462] / 机器人低速 / $?St$Bk?_#[462]
D1863.01 BOOL  ; $?St$Bk?_#[463] / 机器人中低速 / $?St$Bk?_#[463]
D1863.02 BOOL  ; $?St$Bk?_#[464] / 机器人中高速 / $?St$Bk?_#[464]
D1863.03 BOOL  ; $?St$Bk?_#[465] / 机器人高速 / $?St$Bk?_#[465]
D1864.00 BOOL  ; 下料机器人夹爪压板1全部松开
D1864.01 BOOL  ; 下料机器人夹爪压板1全部夹紧
D1864.02 BOOL  ; 下料机器人夹爪压板2全部松开
D1864.03 BOOL  ; 下料机器人夹爪压板2全部夹紧
D1864.04 BOOL  ; 下料机器人夹爪压板3全部松开
D1864.05 BOOL  ; 下料机器人夹爪压板3全部夹紧
D1864.06 BOOL  ; 下料机器人夹爪压板4全部松开
D1864.07 BOOL  ; 下料机器人夹爪压板4全部夹紧
D1864.08 BOOL  ; 下料机器人夹爪压板5全部松开
D1864.09 BOOL  ; 下料机器人夹爪压板5全部夹紧
D1864.10 BOOL  ; 下料机器人压板1全部松开
D1864.11 BOOL  ; 下料机器人压板2全部松开
D1864.12 BOOL  ; 下料机器人压板3全部松开
D1864.13 BOOL  ; 下料机器人压板4全部松开
D1864.14 BOOL  ; 下料机器人压板5全部松开
D1900.00 BOOL  ; 待PC扫码完成后，PLC确认信息
D1900.01 BOOL  ; 待PC收到确认信息后，PLC清除确认信息
D1900.02 BOOL  ; 待PC与MES校验
D1900.03 BOOL  ; 校验后，清除入站请求
D1900.04 BOOL  ; 根据PC反馈的MES信息设置记忆
D1900.05 BOOL  ; PLC判断MES完成
D1900.06 BOOL  ; 一层5个入站通知清除标志
D1900.07 BOOL  ; 二层5个入站通知清除标志
D1901 CHANNEL  ; 扫码数据1长度
D1902 CHANNEL  ; 扫码数据2长度
D1903 CHANNEL  ; 扫码数据3长度
D1904 CHANNEL  ; 扫码数据4长度
D1905 CHANNEL  ; 扫码数据5长度
D1906 CHANNEL  ; 扫码数据6长度
D1907 CHANNEL  ; 扫码数据7长度
D1908 CHANNEL  ; 扫码数据8长度
D1909 CHANNEL  ; 扫码数据9长度
D1910 CHANNEL  ; 扫码数据10长度
D1911 CHANNEL  ; 扫码数据设定位数
D20014 CHANNEL  ; NC433_0_X轴 原点偏移
D20025 CHANNEL  ; NC433_0_X 轴负软限位
D20027 CHANNEL  ; NC433_0_X 轴正软限位
D30 CHANNEL  ; 当前测试通道
D3000 CHANNEL  ; 发送字数
D3001 CHANNEL  ; 目标网络号
D3002 CHANNEL  ; 目标PLC节点号
D3003 CHANNEL  ; 内部逻辑端口号
D3004 CHANNEL  ; 反馈监控时间(0.1-6553.5s)
D3010 CHANNEL  ; 接收字数
D3011 CHANNEL  ; 网络号
D3012 CHANNEL  ; 节点地址
D3013 CHANNEL  ; 逻辑端口
D3014 CHANNEL  ; 监视时间
D3020 CHANNEL  ; 发送字数
D3021 CHANNEL  ; 目标网络号
D3022 CHANNEL  ; 目标PLC节点号
D3023 CHANNEL  ; 内部逻辑端口号
D3024 CHANNEL  ; 反馈监控时间(0.1-6553.5s)
D3030 CHANNEL  ; 发送字数
D3031 CHANNEL  ; 目标网络号
D3032 CHANNEL  ; 目标PLC节点号
D3033 CHANNEL  ; 内部逻辑端口号
D3034 CHANNEL  ; 反馈监控时间(0.1-6553.5s)
D3040 CHANNEL  ; 发送字数
D3041 CHANNEL  ; 目标网络号
D3042 CHANNEL  ; 目标PLC节点号
D3043 CHANNEL  ; 内部逻辑端口号
D3044 CHANNEL  ; 反馈监控时间(0.1-6553.5s)
D3050 CHANNEL  ; 接收字数
D3051 CHANNEL  ; 网络号
D3052 CHANNEL  ; 节点地址
D3053 CHANNEL  ; 逻辑端口
D3054 CHANNEL  ; 监视时间
D3060 CHANNEL  ; 接收字数
D3061 CHANNEL  ; 网络号
D3062 CHANNEL  ; 节点地址
D3063 CHANNEL  ; 逻辑端口
D3064 CHANNEL  ; 监视时间
D3070 CHANNEL  ; 接收字数
D3071 CHANNEL  ; 网络号
D3072 CHANNEL  ; 节点地址
D3073 CHANNEL  ; 逻辑端口
D3074 CHANNEL  ; 反馈监控时间(0.1-6553.5s)
D31 CHANNEL  ; 当前测试通讯按钮
D3100 CHANNEL  ; 发送字数
D3101 CHANNEL  ; 目标网络号
D3102 CHANNEL  ; 目标PLC节点号
D3103 CHANNEL  ; 内部逻辑端口号
D3104 CHANNEL  ; 反馈监控时间(0.1-6553.5s)
D3110 CHANNEL  ; 接收字数
D3111 CHANNEL  ; 网络号
D3112 CHANNEL  ; 节点地址
D3113 CHANNEL  ; 逻辑端口
D3114 CHANNEL  ; 监视时间
D3120 CHANNEL  ; 发送字数
D3121 CHANNEL  ; 目标网络号
D3122 CHANNEL  ; 目标PLC节点号
D3123 CHANNEL  ; 内部逻辑端口号
D3124 CHANNEL  ; 反馈监控时间(0.1-6553.5s)
D3130 CHANNEL  ; 发送字数
D3131 CHANNEL  ; 目标网络号
D3132 CHANNEL  ; 目标PLC节点号
D3133 CHANNEL  ; 内部逻辑端口号
D3134 CHANNEL  ; 反馈监控时间(0.1-6553.5s)
D3140 CHANNEL  ; 发送字数
D3141 CHANNEL  ; 目标网络号
D3142 CHANNEL  ; 目标PLC节点号
D3143 CHANNEL  ; 内部逻辑端口号
D3144 CHANNEL  ; 反馈监控时间(0.1-6553.5s)
D3150 CHANNEL  ; 接收字数
D3151 CHANNEL  ; 网络号
D3153 CHANNEL  ; 逻辑端口
D3154 CHANNEL  ; 监视时间
D3160 CHANNEL  ; 接收字数
D3161 CHANNEL  ; 网络号
D3162 CHANNEL  ; 节点地址
D3163 CHANNEL  ; 逻辑端口
D3164 CHANNEL  ; 监视时间
D3170 CHANNEL  ; 发送字数
D3171 CHANNEL  ; 目标网络号
D3172 CHANNEL  ; 目标PLC节点号
D3173 CHANNEL  ; 内部逻辑端口号
D3174 CHANNEL  ; 反馈监控时间(0.1-6553.5s)
D3180 CHANNEL  ; 接收字数
D3181 CHANNEL  ; 网络号
D3182 CHANNEL  ; 节点地址
D3183 CHANNEL  ; 逻辑端口
D3184 CHANNEL  ; 监视时间
D32 CHANNEL  ; 偏移
D3200 CHANNEL  ; 发送字数
D3201 CHANNEL  ; 目标网络号
D3202 CHANNEL  ; 目标PLC节点号
D3203 CHANNEL  ; 内部逻辑端口号
D3204 CHANNEL  ; 反馈监控时间(0.1-6553.5s)
D3210 CHANNEL  ; 接收字数
D3211 CHANNEL  ; 网络号
D3212 CHANNEL  ; 节点地址
D3213 CHANNEL  ; 逻辑端口
D3214 CHANNEL  ; 监视时间
D3220 CHANNEL  ; 发送字数
D3221 CHANNEL  ; 目标网络号
D3222 CHANNEL  ; 目标PLC节点号
D3223 CHANNEL  ; 内部逻辑端口号
D3224 CHANNEL  ; 反馈监控时间(0.1-6553.5s)
D3230 CHANNEL  ; 发送字数
D3231 CHANNEL  ; 目标网络号
D3232 CHANNEL  ; 目标PLC节点号
D3233 CHANNEL  ; 内部逻辑端口号
D3234 CHANNEL  ; 反馈监控时间(0.1-6553.5s)
D3240 CHANNEL  ; 发送字数
D3241 CHANNEL  ; 目标网络号
D3242 CHANNEL  ; 目标PLC节点号
D3243 CHANNEL  ; 内部逻辑端口号
D3244 CHANNEL  ; 反馈监控时间(0.1-6553.5s)
D3250 CHANNEL  ; 接收字数
D3251 CHANNEL  ; 网络号
D3252 CHANNEL  ; 节点地址
D3253 CHANNEL  ; 逻辑端口
D3254 CHANNEL  ; 监视时间
D3260 CHANNEL  ; 接收字数
D3261 CHANNEL  ; 网络号
D3262 CHANNEL  ; 节点地址
D3263 CHANNEL  ; 逻辑端口
D3264 CHANNEL  ; 监视时间
D3270 CHANNEL  ; 发送字数
D3271 CHANNEL  ; 目标网络号
D3272 CHANNEL  ; 目标PLC节点号
D3273 CHANNEL  ; 内部逻辑端口号
D3274 CHANNEL  ; 反馈监控时间(0.1-6553.5s)
D3280 CHANNEL  ; 接收字数
D3281 CHANNEL  ; 网络号
D3282 CHANNEL  ; 节点地址
D3283 CHANNEL  ; 逻辑端口
D3284 CHANNEL  ; 监视时间
D33 CHANNEL  ; 寄存器偏移
D3400 CHANNEL  ; 1#副PLC网络地址
D3401 CHANNEL  ; 2#副PLC网络地址
D3402 CHANNEL  ; 3#副PLC网络地址
D35 CHANNEL  ; 端口控制字
D3500 CHANNEL  ; 上压力（设定）
D3502 CHANNEL  ; 侧压力（设定）
D3504 CHANNEL  ; 上压偏差
D3506 CHANNEL  ; 侧压偏差
D3508 CHANNEL  ; 宽度
D3519 CHANNEL  ; 时间偏差
D3520 CHANNEL  ; 预压时间SV1
D3521 CHANNEL  ; 预压时间SV2
D3522 CHANNEL  ; 预压时间SV3
D3523 CHANNEL  ; 冷却时间1阀值
D3524 CHANNEL  ; 冷却时间2阀值
D3525 CHANNEL  ; 热压时间
D3526 CHANNEL  ; 4ST_A 热压时间（SV）
D3528 CHANNEL  ; 4ST_B 热压时间(SV)
D3530 CHANNEL  ; 预压时间下限
D3532 CHANNEL  ; 预压时间上限
D3534 CHANNEL  ; 4ST_A 热压时间下限（SV）
D3536 CHANNEL  ; 4ST_A 热压时间上限（SV）
D3540 CHANNEL  ; 上下温差下限
D3542 CHANNEL  ; 上下温差上限
D3544 CHANNEL  ; 侧压温度下限
D3546 CHANNEL  ; 侧压温度上限
D3554 CHANNEL  ; 4ST_B 热压时间下限（SV）
D3556 CHANNEL  ; 4ST_B热压时间上限（SV）
D3560 CHANNEL  ; 上压力保护值
D3562 CHANNEL  ; 侧压力保护值
D3570 CHANNEL  ; 4A动态预压时间
D3572 CHANNEL  ; 4B预压动态时间
D3580 CHANNEL  ; 一阶冷却时间
D3581 CHANNEL  ; 二阶冷却时间
D36 CHANNEL  ; 写入通道
D3600 CHANNEL  ; 4ST_A预压时间
D3601 CHANNEL  ; 4ST_A正压计时
D3602 CHANNEL  ; 4ST_A 热压时间
D3610 CHANNEL  ; 4ST_B预压时间
D3612 CHANNEL  ; 4ST_B 热压时间
D37 CHANNEL  ; 写入偏移
D38 CHANNEL  ; 写入偏移
D39 CHANNEL  ; 写入寄存器偏移
D4000 CHANNEL  ; A1当前使用下压板左边温度
D4003 CHANNEL  ; A2当前使用下压板左边温度
D4006 CHANNEL  ; A3当前使用下压板左边温度
D4009 CHANNEL  ; A4当前使用下压板左边温度
D4012 CHANNEL  ; A5当前使用下压板左边温度
D4020 CHANNEL  ; B1当前使用下压板左边温度
D4023 CHANNEL  ; B2当前使用下压板左边温度
D4026 CHANNEL  ; B3当前使用下压板左边温度
D4029 CHANNEL  ; B4当前使用下压板左边温度
D4032 CHANNEL  ; B5当前使用下压板左边温度
D4100 CHANNEL  ; A1上板左中温度和
D4101 CHANNEL  ; A1上板总温度
D4102 CHANNEL  ; A1上板平均温度
D4110 CHANNEL  ; A2上板中温度和
D4111 CHANNEL  ; A2上板总温度
D4112 CHANNEL  ; A2上板平均总温度
D4120 CHANNEL  ; A3上板左中温度和
D4121 CHANNEL  ; A3上板总温度
D4122 CHANNEL  ; A3上板平均温度
D4130 CHANNEL  ; A4上板左中温度和
D4131 CHANNEL  ; A4上板总温度
D4132 CHANNEL  ; A4上板平均总温度
D4140 CHANNEL  ; A5上板左中温度和
D4141 CHANNEL  ; A5上板总温度
D4142 CHANNEL  ; A5上板平均总温度
D4150 CHANNEL  ; A1下板左中温度和
D4151 CHANNEL  ; A1下板总温度
D4152 CHANNEL  ; A1下板平均温度
D4162 CHANNEL  ; A2下板平均总温度
D4172 CHANNEL  ; A3下板平均温度
D4182 CHANNEL  ; A4下板平均总温度
D4192 CHANNEL  ; A5下板平均总温度
D4200 CHANNEL  ; B1上板左中温度和
D4201 CHANNEL  ; B1上板总温度
D4202 CHANNEL  ; B1上板平均温度
D4210 CHANNEL  ; B2上板中温度和
D4211 CHANNEL  ; B2上板总温度
D4212 CHANNEL  ; B2上板平均总温度
D4220 CHANNEL  ; B3上板左中温度和
D4221 CHANNEL  ; B3上板总温度
D4222 CHANNEL  ; B3上板平均温度
D4230 CHANNEL  ; B4上板左中温度和
D4231 CHANNEL  ; B4上板总温度
D4232 CHANNEL  ; B4上板平均总温度
D4240 CHANNEL  ; B5上板左中温度和
D4241 CHANNEL  ; B5上板总温度
D4242 CHANNEL  ; B5上板平均总温度
D4250 CHANNEL  ; B1下板左中温度和
D4251 CHANNEL  ; B1下板总温度
D4252 CHANNEL  ; B1下板平均温度
D4262 CHANNEL  ; B2下板平均总温度
D4272 CHANNEL  ; B3下板平均温度
D4282 CHANNEL  ; B4下板平均总温度
D4292 CHANNEL  ; B5下板平均总温度
D6000 CHANNEL  ; 热压模组A上层压力
D6002 CHANNEL  ; 热压模组A下层压力
D6004 CHANNEL  ; 热压模组B上层压力
D6006 CHANNEL  ; 热压模组B下层压力
D6008 CHANNEL  ; 热压模组C上层压力
D6010 CHANNEL  ; 热压模组C下层压力
D6012 CHANNEL  ; A3上压力
D6014 CHANNEL  ; A3左压力
D6016 CHANNEL  ; A3右压力
D6018 CHANNEL  ; A4上压力
D6020 CHANNEL  ; A4左压力
D6022 CHANNEL  ; A4右压力
D6024 CHANNEL  ; A5上压力
D6026 CHANNEL  ; A5左压力
D6028 CHANNEL  ; A5右压力
D6030 CHANNEL  ; B1上压力
D6032 CHANNEL  ; B1左压力
D6034 CHANNEL  ; B1右压力
D6036 CHANNEL  ; B2上压力
D6038 CHANNEL  ; B2左压力
D6040 CHANNEL  ; B2右压力
D6042 CHANNEL  ; B3上压力
D6044 CHANNEL  ; B3左压力
D6046 CHANNEL  ; B3右压力
D6048 CHANNEL  ; B4上压力
D6050 CHANNEL  ; B4左压力
D6052 CHANNEL  ; B4右压力
D6054 CHANNEL  ; B5上压力
D6056 CHANNEL  ; B5左压力
D6058 CHANNEL  ; B5右压力
D6060 CHANNEL  ; 热压模组A上层转换倍率
D6062 CHANNEL  ; 热压模组A下层转换倍率
D6064 CHANNEL  ; 热压模组B上层转换倍率
D6066 CHANNEL  ; 热压模组B下层转换倍率
D6068 CHANNEL  ; 热压模组C上层转换倍率
D6070 CHANNEL  ; 热压模组C下层转换倍率
D6072 CHANNEL  ; A3上转换倍率
D6074 CHANNEL  ; A3左转换倍率
D6076 CHANNEL  ; A3右转换倍率
D6078 CHANNEL  ; A4上转换倍率
D6080 CHANNEL  ; A4左转换倍率
D6082 CHANNEL  ; A4右转换倍率
D6084 CHANNEL  ; A5上转换倍率
D6086 CHANNEL  ; A5左转换倍率
D6088 CHANNEL  ; A5右转换倍率
D6090 CHANNEL  ; B1上转换倍率
D6092 CHANNEL  ; B1左转换倍率
D6094 CHANNEL  ; B1右转换倍率
D6096 CHANNEL  ; B2上转换倍率
D6098 CHANNEL  ; B2左转换倍率
D6100 CHANNEL  ; B2右转换倍率
D6102 CHANNEL  ; B3上转换倍率
D6104 CHANNEL  ; B3左转换倍率
D6106 CHANNEL  ; B3右转换倍率
D6108 CHANNEL  ; B4上转换倍率
D6110 CHANNEL  ; B4左转换倍率
D6112 CHANNEL  ; B4右转换倍率
D6114 CHANNEL  ; B5上转换倍率
D6116 CHANNEL  ; B5左转换倍率
D6118 CHANNEL  ; B5右转换倍率
D6120 CHANNEL  ; 热压模组A上层补偿值
D6122 CHANNEL  ; 热压模组A下层补偿值
D6124 CHANNEL  ; 热压模组B上层补偿值
D6126 CHANNEL  ; 热压模组B下层补偿值
D6128 CHANNEL  ; 热压模组C上层补偿值
D6130 CHANNEL  ; 热压模组C下层补偿值
D6132 CHANNEL  ; A3上补偿值
D6134 CHANNEL  ; A3左补偿值
D6136 CHANNEL  ; A3右补偿值
D6138 CHANNEL  ; A4上补偿值
D6140 CHANNEL  ; A4左补偿值
D6142 CHANNEL  ; A4右补偿值
D6144 CHANNEL  ; A5上补偿值
D6146 CHANNEL  ; A5左补偿值
D6148 CHANNEL  ; A5右补偿值
D6150 CHANNEL  ; B1上补偿值
D6152 CHANNEL  ; B1左补偿值
D6154 CHANNEL  ; B1右补偿值
D6156 CHANNEL  ; B2上补偿值
D6158 CHANNEL  ; B2左补偿值
D6160 CHANNEL  ; B2右补偿值
D6162 CHANNEL  ; B3上补偿值
D6164 CHANNEL  ; B3左补偿值
D6166 CHANNEL  ; B3右补偿值
D6168 CHANNEL  ; B4上补偿值
D6170 CHANNEL  ; B4左补偿值
D6172 CHANNEL  ; B4右补偿值
D6174 CHANNEL  ; B5上补偿值
D6176 CHANNEL  ; B5左补偿值
D6178 CHANNEL  ; B5右补偿值
D6300 CHANNEL  ; 上压力调整下偏差
D6302 CHANNEL  ; 上压力调整上偏差
D6304 CHANNEL  ; 侧压力调整下偏差
D6306 CHANNEL  ; 侧压力调整上偏差
D6308 CHANNEL  ; 上压力调整变频值
D6310 CHANNEL  ; 上压力调整下限值
D6312 CHANNEL  ; 上压力调整上限值
D6314 CHANNEL  ; 侧压力调整下限值
D6316 CHANNEL  ; 侧压力调整上限值
D6318 CHANNEL  ; 侧压力调整变频值
D6320 CHANNEL  ; 上压力下限值
D6322 CHANNEL  ; 上压力上限值
D6324 CHANNEL  ; 侧压力下限值
D6326 CHANNEL  ; 侧压力上限值
D6328 CHANNEL  ; 侧压开始调整时的上压力阀值
D6330 CHANNEL  ; 上压力调整下限值
D6332 CHANNEL  ; 上压力调整下限
D6334 CHANNEL  ; 上压力下限值
D6350 CHANNEL  ; A工位上压参考选择（1.2.3.4.5）
D6352 CHANNEL  ; A工位上压调整参考
D6354 CHANNEL  ; 侧压快速调整量(正）
D6356 CHANNEL  ; 侧压快速调整量(负）
D6358 CHANNEL  ; 快速调整间隔（短整型）
D6360 CHANNEL  ; 侧压慢速调整量（正）
D6362 CHANNEL  ; 侧压慢速调整量（负）
D6364 CHANNEL  ; 慢速调整间隔（）
D6370 CHANNEL  ; B工位上压参考选择（1.2.3.4.5）
D6372 CHANNEL  ; B工位上压调整参考
D6374 CHANNEL  ; 正压快速调整量 +
D6376 CHANNEL  ; 正压快速调整量 -
D6378 CHANNEL  ; 正压快速调整频率
D6380 CHANNEL  ; 正压慢速调整量
D6382 CHANNEL  ; 正压慢速调整量-
D6384 CHANNEL  ; 正压慢速调整间隔
D6401 CHANNEL  ; A1比例阀
D6402 CHANNEL  ; A2比例阀
D6403 CHANNEL  ; A3比例阀
D6404 CHANNEL  ; A4比例阀
D6405 CHANNEL  ; B1比例阀
D6406 CHANNEL  ; B2比例阀
D6407 CHANNEL  ; B3比例阀
D6408 CHANNEL  ; B4比例阀
D6411 CHANNEL  ; A5比例阀
D6412 CHANNEL  ; B5比例阀
D6413 CHANNEL  ; 正压A转矩输出
D6414 CHANNEL  ; 侧压A1左转矩输出
D6415 CHANNEL  ; 侧压A1右转矩输出
D6416 CHANNEL  ; 侧压A2左转矩输出
D6417 CHANNEL  ; 侧压A2右转矩输出
D6418 CHANNEL  ; 侧压A3左转矩输出
D6421 CHANNEL  ; 侧压A3右转矩输出
D6422 CHANNEL  ; 侧压A4左转矩输出
D6423 CHANNEL  ; 侧压A4右转矩输出
D6424 CHANNEL  ; 侧压A5左转矩输出
D6425 CHANNEL  ; 侧压A5右转矩输出
D6426 CHANNEL  ; 正压B转矩输出
D6427 CHANNEL  ; 侧压B1左转矩输出
D6428 CHANNEL  ; 侧压B1右转矩输出
D6431 CHANNEL  ; 侧压B2左转矩输出
D6432 CHANNEL  ; 侧压B2右转矩输出
D6433 CHANNEL  ; 侧压B3左转矩输出
D6434 CHANNEL  ; 侧压B3右转矩输出
D6435 CHANNEL  ; 侧压B4左转矩输出
D6436 CHANNEL  ; 侧压B4右转矩输出
D6437 CHANNEL  ; 侧压B5左转矩输出
D6438 CHANNEL  ; 侧压B5右转矩输出
D6441 CHANNEL  ; A1比例阀重力设定
D6442 CHANNEL  ; A2比例阀重力设定
D6443 CHANNEL  ; A3比例阀重力设定
D6444 CHANNEL  ; A4比例阀重力设定
D6445 CHANNEL  ; B1比例阀重力设定
D6446 CHANNEL  ; B2比例阀重力设定
D6447 CHANNEL  ; B3比例阀重力设定
D6448 CHANNEL  ; B4比例阀重力设定
D6449 CHANNEL  ; A5比例阀重力设定
D6450 CHANNEL  ; B5比例阀重力设定
D6451 CHANNEL  ; A1比例阀顶升设定
D6452 CHANNEL  ; A2比例阀顶升设定
D6453 CHANNEL  ; A3比例阀顶升设定
D6454 CHANNEL  ; A4比例阀顶升设定
D6455 CHANNEL  ; B1比例阀顶升设定
D6456 CHANNEL  ; B2比例阀顶升设定
D6457 CHANNEL  ; B3比例阀顶升设定
D6458 CHANNEL  ; B4比例阀顶升设定
D6459 CHANNEL  ; A5比例阀顶升设定
D6460 CHANNEL  ; B5比例阀顶升设定
D7000 CHANNEL  ; 手/自动选择延时设置
D7001 CHANNEL  ; 启动按钮延时设置
D7002 CHANNEL  ; 停止按钮延时设置
D7003 CHANNEL  ; 复位按钮延时设置
D7004 CHANNEL  ; 前门磁延时设置
D7005 CHANNEL  ; 后门磁延时设置
D7006 CHANNEL  ; 左门磁延时设置
D7007 CHANNEL  ; 右门磁延时设置
D7008 CHANNEL  ; 气源压力开关延时设置
D7009 CHANNEL  ; 主急停按钮延时设置
D7010 CHANNEL  ; 移动屏急停延时设置
D7011 CHANNEL  ; 移动屏使用中延时设置
D7012 CHANNEL  ; 备用1延时设置
D7013 CHANNEL  ; 备用2延时设置
D7014 CHANNEL  ; 备用3延时设置
D7015 CHANNEL  ; 备用4延时设置
D7016 CHANNEL  ; 启动按钮1延时设置
D7017 CHANNEL  ; 启动按钮2延时设置
D7018 CHANNEL  ; 进出料安全光栅延时设置
D7019 CHANNEL  ; 进料定位上层前后松开位延时设置
D7020 CHANNEL  ; 进料定位上层前后夹紧位延时设置
D7021 CHANNEL  ; 进料定位下层前后松开位延时设置
D7022 CHANNEL  ; 进料定位下层前后夹紧位延时设置
D7023 CHANNEL  ; 进料定位上层左右松开位延时设置
D7024 CHANNEL  ; 进料定位上层左右夹紧位延时设置
D7025 CHANNEL  ; 进料定位下层左右松开位延时设置
D7026 CHANNEL  ; 进料定位下层左右夹紧位延时设置
D7027 CHANNEL  ; 进料定位平台上层待料位延时设置
D7028 CHANNEL  ; 进料定位平台上层出料位延时设置
D7029 CHANNEL  ; 进料定位平台下层待料位延时设置
D7030 CHANNEL  ; 进料定位平台下层出料位延时设置
D7031 CHANNEL  ; 进料定位上层有料感应延时设置
D7032 CHANNEL  ; 进料定位下层有料感应延时设置
D7033 CHANNEL  ; 出料定位上层前后松开位延时设置
D7034 CHANNEL  ; 出料定位上层前后夹紧位延时设置
D7035 CHANNEL  ; 出料定位下层前后松开位延时设置
D7036 CHANNEL  ; 出料定位下层前后夹紧位延时设置
D7037 CHANNEL  ; 出料定位上层左右松开位延时设置
D7038 CHANNEL  ; 出料定位上层左右夹紧位延时设置
D7039 CHANNEL  ; 出料定位下层左右松开位延时设置
D7040 CHANNEL  ; 出料定位下层左右夹紧位延时设置
D7041 CHANNEL  ; 出料定位平台上层接料位延时设置
D7042 CHANNEL  ; 出料定位平台上层出料位延时设置
D7043 CHANNEL  ; 出料定位平台下层接料位延时设置
D7044 CHANNEL  ; 出料定位平台下层出料位延时设置
D7045 CHANNEL  ; 出料定位上层有料感应延时设置
D7046 CHANNEL  ; 出料定位下层有料感应延时设置
D7047 CHANNEL  ; 备用5延时设置
D7048 CHANNEL  ; 进料夹爪张开位延时设置
D7049 CHANNEL  ; 进料夹爪夹紧位延时设置
D7050 CHANNEL  ; 进料爪上层左压紧上升位延时设置
D7051 CHANNEL  ; 进料爪上层右压紧上升位延时设置
D7052 CHANNEL  ; 进料爪下层左压紧上升位延时设置
D7053 CHANNEL  ; 进料爪下层右压紧上升位延时设置
D7054 CHANNEL  ; 进料爪上层中间压紧上升位延时设置
D7055 CHANNEL  ; 进料爪下层中间压紧上升位延时设置
D7056 CHANNEL  ; 进料夹爪上升位延时设置
D7057 CHANNEL  ; 进料夹爪下降位延时设置
D7058 CHANNEL  ; 进料爪上层有料感应延时设置
D7059 CHANNEL  ; 进料爪下层有料感应延时设置
D7060 CHANNEL  ; 出料夹爪张开位延时设置
D7061 CHANNEL  ; 出料夹爪夹紧位延时设置
D7062 CHANNEL  ; 出料爪上层左压紧上升位延时设置
D7063 CHANNEL  ; 出料爪上层右压紧上升位延时设置
D7064 CHANNEL  ; 出料爪下层左压紧上升位延时设置
D7065 CHANNEL  ; 出料爪下层右压紧上升位延时设置
D7066 CHANNEL  ; 出料夹爪上升位延时设置
D7067 CHANNEL  ; 出料夹爪下降位延时设置
D7068 CHANNEL  ; 出料爪上层有料感应延时设置
D7069 CHANNEL  ; 出料爪下层有料感应延时设置
D7070 CHANNEL  ; 备用6延时设置
D7071 CHANNEL  ; 备用7延时设置
D7072 CHANNEL  ; 热压A增压缸上升位延时设置
D7073 CHANNEL  ; 热压A增压缸下降位延时设置
D7074 CHANNEL  ; 热压A上层顶升气缸上升位延时设置
D7075 CHANNEL  ; 热压A上层顶升气缸下降位延时设置
D7076 CHANNEL  ; 热压A下层顶升气缸上升位延时设置
D7077 CHANNEL  ; 热压A下层顶升气缸下降位延时设置
D7078 CHANNEL  ; 热压A垫高气缸移出位延时设置
D7079 CHANNEL  ; 热压A垫高气缸热压位延时设置
D7080 CHANNEL  ; 热压A上层Hip测试气缸上升位延时设置
D7081 CHANNEL  ; 热压A上层Hip测试气缸下降位延时设置
D7082 CHANNEL  ; 热压A下层Hip测试气缸上升位延时设置
D7083 CHANNEL  ; 热压A下层Hip测试气缸下降位延时设置
D7084 CHANNEL  ; 热压A上层有料感应延时设置
D7085 CHANNEL  ; 热压A下层有料感应延时设置
D7086 CHANNEL  ; 热压A上层极耳检查输入延时设置
D7087 CHANNEL  ; 热压A下层极耳检查输入延时设置
D7088 CHANNEL  ; 热压B增压缸上升位延时设置
D7089 CHANNEL  ; 热压B增压缸下降位延时设置
D7090 CHANNEL  ; 热压B上层顶升气缸上升位延时设置
D7091 CHANNEL  ; 热压B上层顶升气缸下降位延时设置
D7092 CHANNEL  ; 热压B下层顶升气缸上升位延时设置
D7093 CHANNEL  ; 热压B下层顶升气缸下降位延时设置
D7094 CHANNEL  ; 热压B垫高气缸移出位延时设置
D7095 CHANNEL  ; 热压B垫高气缸热压位延时设置
D7096 CHANNEL  ; 热压B上层Hip测试气缸上升位延时设置
D7097 CHANNEL  ; 热压B上层Hip测试气缸下降位延时设置
D7098 CHANNEL  ; 热压B下层Hip测试气缸上升位延时设置
D7099 CHANNEL  ; 热压B下层Hip测试气缸下降位延时设置
D7100 CHANNEL  ; 热压B上层有料感应延时设置
D7101 CHANNEL  ; 热压B下层有料感应延时设置
D7102 CHANNEL  ; 热压B下层极耳检查输入延时设置
D7103 CHANNEL  ; 备用9延时设置
D7104 CHANNEL  ; 热压C增压缸上升位延时设置
D7105 CHANNEL  ; 热压C增压缸下降位延时设置
D7106 CHANNEL  ; 热压C上层顶升气缸上升位延时设置
D7107 CHANNEL  ; 热压C上层顶升气缸下降位延时设置
D7108 CHANNEL  ; 热压C下层顶升气缸上升位延时设置
D7109 CHANNEL  ; 热压C下层顶升气缸下降位延时设置
D7110 CHANNEL  ; 热压C垫高气缸移出位延时设置
D7111 CHANNEL  ; 热压C垫高气缸热压位延时设置
D7112 CHANNEL  ; 热压C上层Hip测试气缸上升位延时设置
D7113 CHANNEL  ; 热压C上层Hip测试气缸下降位延时设置
D7114 CHANNEL  ; 热压C下层Hip测试气缸上升位延时设置
